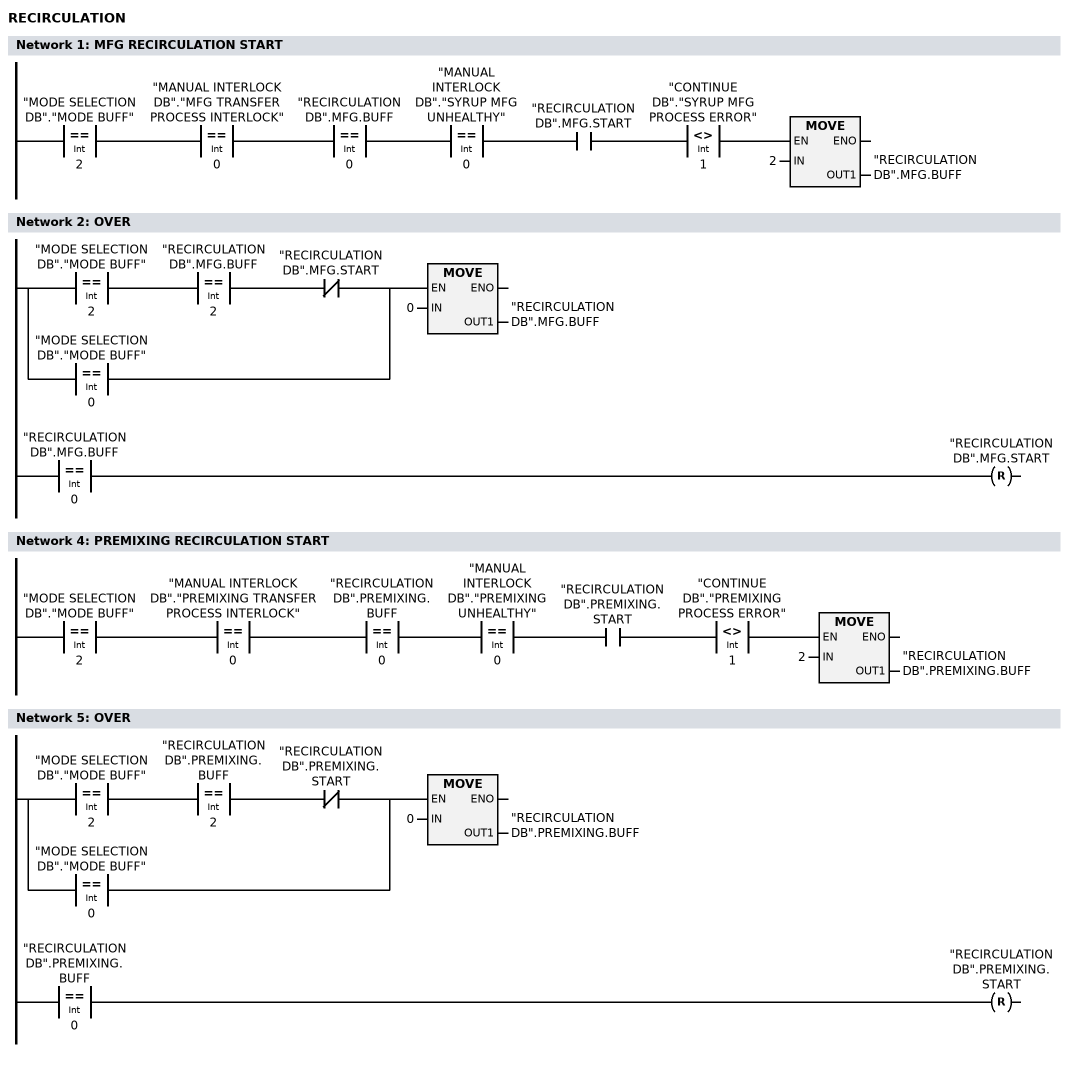
   RUNG wire#powerrail
      { S7_Templates := "SrcType := Int" } EQ_Contact(in1 := "MODE SELECTION DB"."MODE BUFF", in2 := 2)
      { S7_Templates := "SrcType := Int" } EQ_Contact(in1 := "MANUAL INTERLOCK DB"."MFG TRANSFER PROCESS INTERLOCK", in2 := 0)
      { S7_Templates := "SrcType := Int" } EQ_Contact(in1 := "RECIRCULATION DB".MFG.BUFF, in2 := 0)
      { S7_Templates := "SrcType := Int" } EQ_Contact(in1 := "MANUAL INTERLOCK DB"."SYRUP MFG UNHEALTHY", in2 := 0)
      Contact( "RECIRCULATION DB".MFG.START )
      { S7_Templates := "SrcType := Int" } NE_Contact(in1 := "CONTINUE DB"."SYRUP MFG PROCESS ERROR", in2 := 1)
      Move(in := 2, out1 => "RECIRCULATION DB".MFG.BUFF)
   END_RUNG
   // the same network as SCL:
   IF ("MODE SELECTION DB"."MODE BUFF" = 2) AND ("MANUAL INTERLOCK DB"."MFG TRANSFER PROCESS INTERLOCK" = 0) AND ("RECIRCULATION DB".MFG.BUFF = 0) AND ("MANUAL INTERLOCK DB"."SYRUP MFG UNHEALTHY" = 0) AND "RECIRCULATION DB".MFG.START AND ("CONTINUE DB"."SYRUP MFG PROCESS ERROR" <> 1) THEN
       "RECIRCULATION DB".MFG.BUFF := 2;
   END_IF;
END_REGION

REGION Network 2: OVER
   RUNG wire#powerrail
      { S7_Templates := "SrcType := Int" } EQ_Contact(in1 := "MODE SELECTION DB"."MODE BUFF", in2 := 2)
      { S7_Templates := "SrcType := Int" } EQ_Contact(in1 := "RECIRCULATION DB".MFG.BUFF, in2 := 2)
      I_Contact( "RECIRCULATION DB".MFG.START )
      wire#w1
      Move(in := 0, out1 => "RECIRCULATION DB".MFG.BUFF)
   END_RUNG
   RUNG wire#powerrail
      { S7_Templates := "SrcType := Int" } EQ_Contact(in1 := "MODE SELECTION DB"."MODE BUFF", in2 := 0)
   END_RUNG wire#w1
   RUNG wire#powerrail
      { S7_Templates := "SrcType := Int" } EQ_Contact(in1 := "RECIRCULATION DB".MFG.BUFF, in2 := 0)
      R_Coil( "RECIRCULATION DB".MFG.START )
   END_RUNG
   // the same network as SCL:
   IF (("MODE SELECTION DB"."MODE BUFF" = 2) AND ("RECIRCULATION DB".MFG.BUFF = 2) AND NOT "RECIRCULATION DB".MFG.START) OR ("MODE SELECTION DB"."MODE BUFF" = 0) THEN
       "RECIRCULATION DB".MFG.BUFF := 0;
   END_IF;
   IF "RECIRCULATION DB".MFG.BUFF = 0 THEN "RECIRCULATION DB".MFG.START := FALSE; END_IF;
END_REGION

REGION Network 4: PREMIXING RECIRCULATION START
   RUNG wire#powerrail
      { S7_Templates := "SrcType := Int" } EQ_Contact(in1 := "MODE SELECTION DB"."MODE BUFF", in2 := 2)
      { S7_Templates := "SrcType := Int" } EQ_Contact(in1 := "MANUAL INTERLOCK DB"."PREMIXING TRANSFER PROCESS INTERLOCK", in2 := 0)
      { S7_Templates := "SrcType := Int" } EQ_Contact(in1 := "RECIRCULATION DB".PREMIXING.BUFF, in2 := 0)
      { S7_Templates := "SrcType := Int" } EQ_Contact(in1 := "MANUAL INTERLOCK DB"."PREMIXING UNHEALTHY", in2 := 0)
      Contact( "RECIRCULATION DB".PREMIXING.START )
      { S7_Templates := "SrcType := Int" } NE_Contact(in1 := "CONTINUE DB"."PREMIXING PROCESS ERROR", in2 := 1)
      Move(in := 2, out1 => "RECIRCULATION DB".PREMIXING.BUFF)
   END_RUNG
   // the same network as SCL:
   IF ("MODE SELECTION DB"."MODE BUFF" = 2) AND ("MANUAL INTERLOCK DB"."PREMIXING TRANSFER PROCESS INTERLOCK" = 0) AND ("RECIRCULATION DB".PREMIXING.BUFF = 0) AND ("MANUAL INTERLOCK DB"."PREMIXING UNHEALTHY" = 0) AND "RECIRCULATION DB".PREMIXING.START AND ("CONTINUE DB"."PREMIXING PROCESS ERROR" <> 1) THEN
       "RECIRCULATION DB".PREMIXING.BUFF := 2;
   END_IF;
END_REGION

REGION Network 5: OVER
   RUNG wire#powerrail
      { S7_Templates := "SrcType := Int" } EQ_Contact(in1 := "MODE SELECTION DB"."MODE BUFF", in2 := 2)
      { S7_Templates := "SrcType := Int" } EQ_Contact(in1 := "RECIRCULATION DB".PREMIXING.BUFF, in2 := 2)
      I_Contact( "RECIRCULATION DB".PREMIXING.START )
      wire#w1
      Move(in := 0, out1 => "RECIRCULATION DB".PREMIXING.BUFF)
   END_RUNG
   RUNG wire#powerrail
      { S7_Templates := "SrcType := Int" } EQ_Contact(in1 := "MODE SELECTION DB"."MODE BUFF", in2 := 0)
   END_RUNG wire#w1
   RUNG wire#powerrail
      { S7_Templates := "SrcType := Int" } EQ_Contact(in1 := "RECIRCULATION DB".PREMIXING.BUFF, in2 := 0)
      R_Coil( "RECIRCULATION DB".PREMIXING.START )
   END_RUNG
   // the same network as SCL:
   IF (("MODE SELECTION DB"."MODE BUFF" = 2) AND ("RECIRCULATION DB".PREMIXING.BUFF = 2) AND NOT "RECIRCULATION DB".PREMIXING.START) OR ("MODE SELECTION DB"."MODE BUFF" = 0) THEN
       "RECIRCULATION DB".PREMIXING.BUFF := 0;
   END_IF;
   IF "RECIRCULATION DB".PREMIXING.BUFF = 0 THEN "RECIRCULATION DB".PREMIXING.START := FALSE; END_IF;
END_REGION
END_FUNCTION

FUNCTION "TEMP CUTOFF LOGIC" : Void   // FC11, LAD
{ S7_Optimized_Access := 'TRUE' }
// stored: SetENOAutomatically false
   VAR_TEMP   // added for the SCL form of the ladder/FBD networks
      _w1 : Bool;
      _w2 : Bool;
   END_VAR
BEGIN

REGION Network 1: MFG_TEMP. VALUE ///////////////////////////////////////////////////////////////
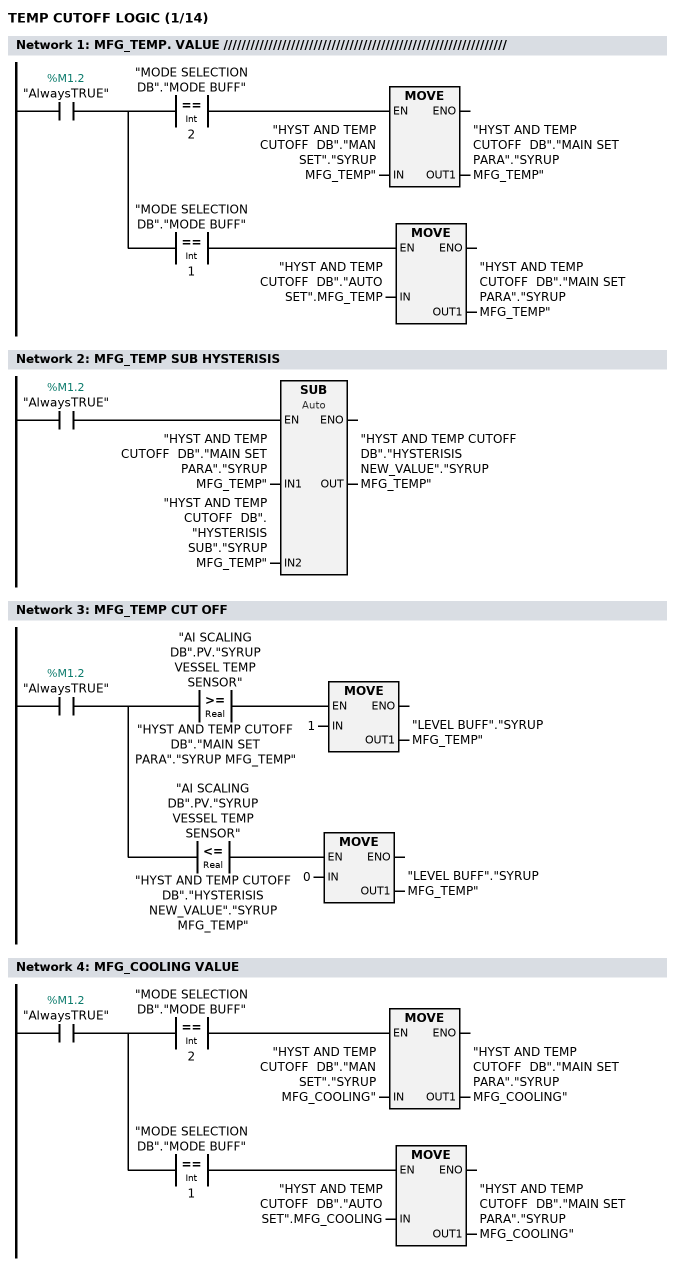
   RUNG wire#powerrail
      Contact( "AlwaysTRUE" )
      wire#w1
      { S7_Templates := "SrcType := Int" } EQ_Contact(in1 := "MODE SELECTION DB"."MODE BUFF", in2 := 2)
      Move(in := "HYST AND TEMP CUTOFF  DB"."MAN SET"."SYRUP MFG_TEMP", out1 => "HYST AND TEMP CUTOFF  DB"."MAIN SET PARA"."SYRUP MFG_TEMP")
   END_RUNG
   RUNG wire#w1
      { S7_Templates := "SrcType := Int" } EQ_Contact(in1 := "MODE SELECTION DB"."MODE BUFF", in2 := 1)
      Move(in := "HYST AND TEMP CUTOFF  DB"."AUTO SET".MFG_TEMP, out1 => "HYST AND TEMP CUTOFF  DB"."MAIN SET PARA"."SYRUP MFG_TEMP")
   END_RUNG
   // the same network as SCL:
   IF "AlwaysTRUE" AND ("MODE SELECTION DB"."MODE BUFF" = 2) THEN
       "HYST AND TEMP CUTOFF  DB"."MAIN SET PARA"."SYRUP MFG_TEMP" := "HYST AND TEMP CUTOFF  DB"."MAN SET"."SYRUP MFG_TEMP";
   END_IF;
   IF "AlwaysTRUE" AND ("MODE SELECTION DB"."MODE BUFF" = 1) THEN
       "HYST AND TEMP CUTOFF  DB"."MAIN SET PARA"."SYRUP MFG_TEMP" := "HYST AND TEMP CUTOFF  DB"."AUTO SET".MFG_TEMP;
   END_IF;
END_REGION

REGION Network 2: MFG_TEMP SUB HYSTERISIS
   RUNG wire#powerrail
      Contact( "AlwaysTRUE" )
      Sub(in1 := "HYST AND TEMP CUTOFF  DB"."MAIN SET PARA"."SYRUP MFG_TEMP", in2 := "HYST AND TEMP CUTOFF  DB"."HYSTERISIS SUB"."SYRUP MFG_TEMP", out => "HYST AND TEMP CUTOFF  DB"."HYSTERISIS NEW_VALUE"."SYRUP MFG_TEMP")
   END_RUNG
   // the same network as SCL:
   IF "AlwaysTRUE" THEN
       "HYST AND TEMP CUTOFF  DB"."HYSTERISIS NEW_VALUE"."SYRUP MFG_TEMP" := "HYST AND TEMP CUTOFF  DB"."MAIN SET PARA"."SYRUP MFG_TEMP" - "HYST AND TEMP CUTOFF  DB"."HYSTERISIS SUB"."SYRUP MFG_TEMP";
   END_IF;
END_REGION

REGION Network 3: MFG_TEMP CUT OFF
   RUNG wire#powerrail
      Contact( "AlwaysTRUE" )
      wire#w1
      { S7_Templates := "SrcType := Real" } GE_Contact(in1 := "AI SCALING DB".PV."SYRUP VESSEL TEMP SENSOR", in2 := "HYST AND TEMP CUTOFF  DB"."MAIN SET PARA"."SYRUP MFG_TEMP")
      Move(in := 1, out1 => "LEVEL BUFF"."SYRUP MFG_TEMP")
   END_RUNG
   RUNG wire#w1
      { S7_Templates := "SrcType := Real" } LE_Contact(in1 := "AI SCALING DB".PV."SYRUP VESSEL TEMP SENSOR", in2 := "HYST AND TEMP CUTOFF  DB"."HYSTERISIS NEW_VALUE"."SYRUP MFG_TEMP")
      Move(in := 0, out1 => "LEVEL BUFF"."SYRUP MFG_TEMP")
   END_RUNG
   // the same network as SCL:
   IF "AlwaysTRUE" AND ("AI SCALING DB".PV."SYRUP VESSEL TEMP SENSOR" >= "HYST AND TEMP CUTOFF  DB"."MAIN SET PARA"."SYRUP MFG_TEMP") THEN
       "LEVEL BUFF"."SYRUP MFG_TEMP" := 1;
   END_IF;
   IF "AlwaysTRUE" AND ("AI SCALING DB".PV."SYRUP VESSEL TEMP SENSOR" <= "HYST AND TEMP CUTOFF  DB"."HYSTERISIS NEW_VALUE"."SYRUP MFG_TEMP") THEN
       "LEVEL BUFF"."SYRUP MFG_TEMP" := 0;
   END_IF;
END_REGION

REGION Network 4: MFG_COOLING VALUE
   RUNG wire#powerrail
      Contact( "AlwaysTRUE" )
      wire#w1
      { S7_Templates := "SrcType := Int" } EQ_Contact(in1 := "MODE SELECTION DB"."MODE BUFF", in2 := 2)
      Move(in := "HYST AND TEMP CUTOFF  DB"."MAN SET"."SYRUP MFG_COOLING", out1 => "HYST AND TEMP CUTOFF  DB"."MAIN SET PARA"."SYRUP MFG_COOLING")
   END_RUNG
   RUNG wire#w1
      { S7_Templates := "SrcType := Int" } EQ_Contact(in1 := "MODE SELECTION DB"."MODE BUFF", in2 := 1)
      Move(in := "HYST AND TEMP CUTOFF  DB"."AUTO SET".MFG_COOLING, out1 => "HYST AND TEMP CUTOFF  DB"."MAIN SET PARA"."SYRUP MFG_COOLING")
   END_RUNG
   // the same network as SCL:
   IF "AlwaysTRUE" AND ("MODE SELECTION DB"."MODE BUFF" = 2) THEN
       "HYST AND TEMP CUTOFF  DB"."MAIN SET PARA"."SYRUP MFG_COOLING" := "HYST AND TEMP CUTOFF  DB"."MAN SET"."SYRUP MFG_COOLING";
   END_IF;
   IF "AlwaysTRUE" AND ("MODE SELECTION DB"."MODE BUFF" = 1) THEN
       "HYST AND TEMP CUTOFF  DB"."MAIN SET PARA"."SYRUP MFG_COOLING" := "HYST AND TEMP CUTOFF  DB"."AUTO SET".MFG_COOLING;
   END_IF;
END_REGION

REGION Network 5: MFG_COOLING SUB HYSTERISIS
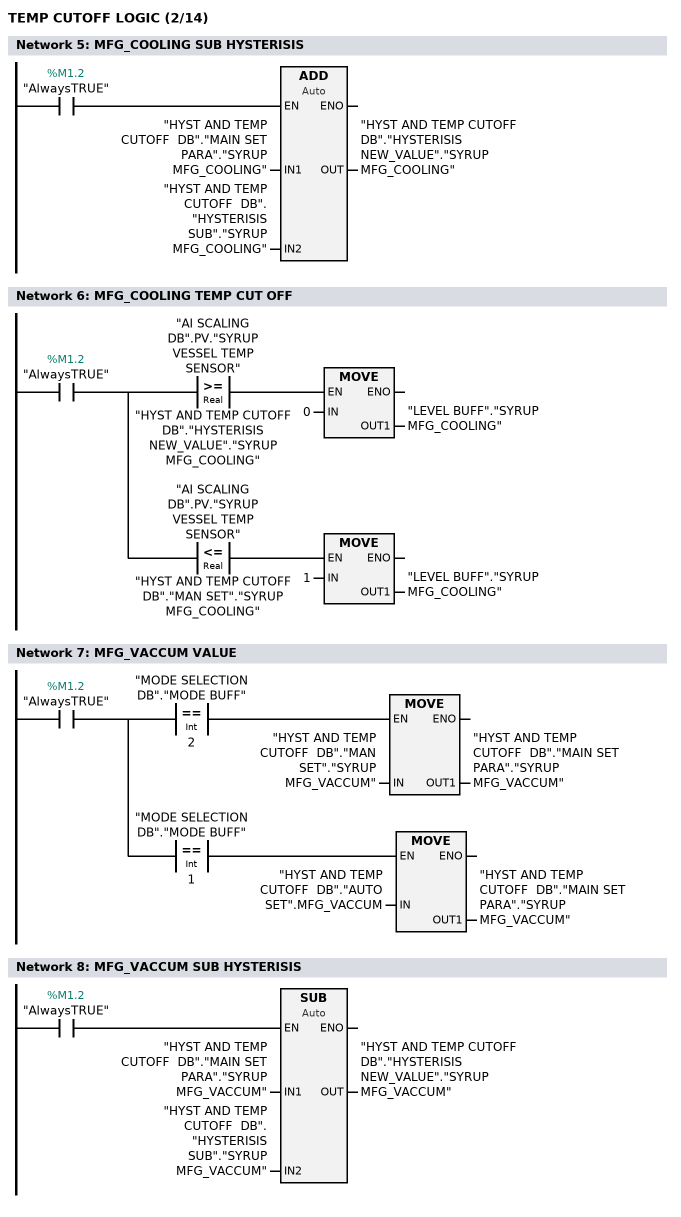
   RUNG wire#powerrail
      Contact( "AlwaysTRUE" )
      Add(in1 := "HYST AND TEMP CUTOFF  DB"."MAIN SET PARA"."SYRUP MFG_COOLING", in2 := "HYST AND TEMP CUTOFF  DB"."HYSTERISIS SUB"."SYRUP MFG_COOLING", out => "HYST AND TEMP CUTOFF  DB"."HYSTERISIS NEW_VALUE"."SYRUP MFG_COOLING")
   END_RUNG
   // the same network as SCL:
   IF "AlwaysTRUE" THEN
       "HYST AND TEMP CUTOFF  DB"."HYSTERISIS NEW_VALUE"."SYRUP MFG_COOLING" := "HYST AND TEMP CUTOFF  DB"."MAIN SET PARA"."SYRUP MFG_COOLING" + "HYST AND TEMP CUTOFF  DB"."HYSTERISIS SUB"."SYRUP MFG_COOLING";
   END_IF;
END_REGION

REGION Network 6: MFG_COOLING TEMP CUT OFF
   RUNG wire#powerrail
      Contact( "AlwaysTRUE" )
      wire#w1
      { S7_Templates := "SrcType := Real" } GE_Contact(in1 := "AI SCALING DB".PV."SYRUP VESSEL TEMP SENSOR", in2 := "HYST AND TEMP CUTOFF  DB"."HYSTERISIS NEW_VALUE"."SYRUP MFG_COOLING")
      Move(in := 0, out1 => "LEVEL BUFF"."SYRUP MFG_COOLING")
   END_RUNG
   RUNG wire#w1
      { S7_Templates := "SrcType := Real" } LE_Contact(in1 := "AI SCALING DB".PV."SYRUP VESSEL TEMP SENSOR", in2 := "HYST AND TEMP CUTOFF  DB"."MAN SET"."SYRUP MFG_COOLING")
      Move(in := 1, out1 => "LEVEL BUFF"."SYRUP MFG_COOLING")
   END_RUNG
   // the same network as SCL:
   IF "AlwaysTRUE" AND ("AI SCALING DB".PV."SYRUP VESSEL TEMP SENSOR" >= "HYST AND TEMP CUTOFF  DB"."HYSTERISIS NEW_VALUE"."SYRUP MFG_COOLING") THEN
       "LEVEL BUFF"."SYRUP MFG_COOLING" := 0;
   END_IF;
   IF "AlwaysTRUE" AND ("AI SCALING DB".PV."SYRUP VESSEL TEMP SENSOR" <= "HYST AND TEMP CUTOFF  DB"."MAN SET"."SYRUP MFG_COOLING") THEN
       "LEVEL BUFF"."SYRUP MFG_COOLING" := 1;
   END_IF;
END_REGION

REGION Network 7: MFG_VACCUM VALUE
   RUNG wire#powerrail
      Contact( "AlwaysTRUE" )
      wire#w1
      { S7_Templates := "SrcType := Int" } EQ_Contact(in1 := "MODE SELECTION DB"."MODE BUFF", in2 := 2)
      Move(in := "HYST AND TEMP CUTOFF  DB"."MAN SET"."SYRUP MFG_VACCUM", out1 => "HYST AND TEMP CUTOFF  DB"."MAIN SET PARA"."SYRUP MFG_VACCUM")
   END_RUNG
   RUNG wire#w1
      { S7_Templates := "SrcType := Int" } EQ_Contact(in1 := "MODE SELECTION DB"."MODE BUFF", in2 := 1)
      Move(in := "HYST AND TEMP CUTOFF  DB"."AUTO SET".MFG_VACCUM, out1 => "HYST AND TEMP CUTOFF  DB"."MAIN SET PARA"."SYRUP MFG_VACCUM")
   END_RUNG
   // the same network as SCL:
   IF "AlwaysTRUE" AND ("MODE SELECTION DB"."MODE BUFF" = 2) THEN
       "HYST AND TEMP CUTOFF  DB"."MAIN SET PARA"."SYRUP MFG_VACCUM" := "HYST AND TEMP CUTOFF  DB"."MAN SET"."SYRUP MFG_VACCUM";
   END_IF;
   IF "AlwaysTRUE" AND ("MODE SELECTION DB"."MODE BUFF" = 1) THEN
       "HYST AND TEMP CUTOFF  DB"."MAIN SET PARA"."SYRUP MFG_VACCUM" := "HYST AND TEMP CUTOFF  DB"."AUTO SET".MFG_VACCUM;
   END_IF;
END_REGION

REGION Network 8: MFG_VACCUM SUB HYSTERISIS
   RUNG wire#powerrail
      Contact( "AlwaysTRUE" )
      Sub(in1 := "HYST AND TEMP CUTOFF  DB"."MAIN SET PARA"."SYRUP MFG_VACCUM", in2 := "HYST AND TEMP CUTOFF  DB"."HYSTERISIS SUB"."SYRUP MFG_VACCUM", out => "HYST AND TEMP CUTOFF  DB"."HYSTERISIS NEW_VALUE"."SYRUP MFG_VACCUM")
   END_RUNG
   // the same network as SCL:
   IF "AlwaysTRUE" THEN
       "HYST AND TEMP CUTOFF  DB"."HYSTERISIS NEW_VALUE"."SYRUP MFG_VACCUM" := "HYST AND TEMP CUTOFF  DB"."MAIN SET PARA"."SYRUP MFG_VACCUM" - "HYST AND TEMP CUTOFF  DB"."HYSTERISIS SUB"."SYRUP MFG_VACCUM";
   END_IF;
END_REGION

REGION Network 9: MFG_VACCUM CUT OFF
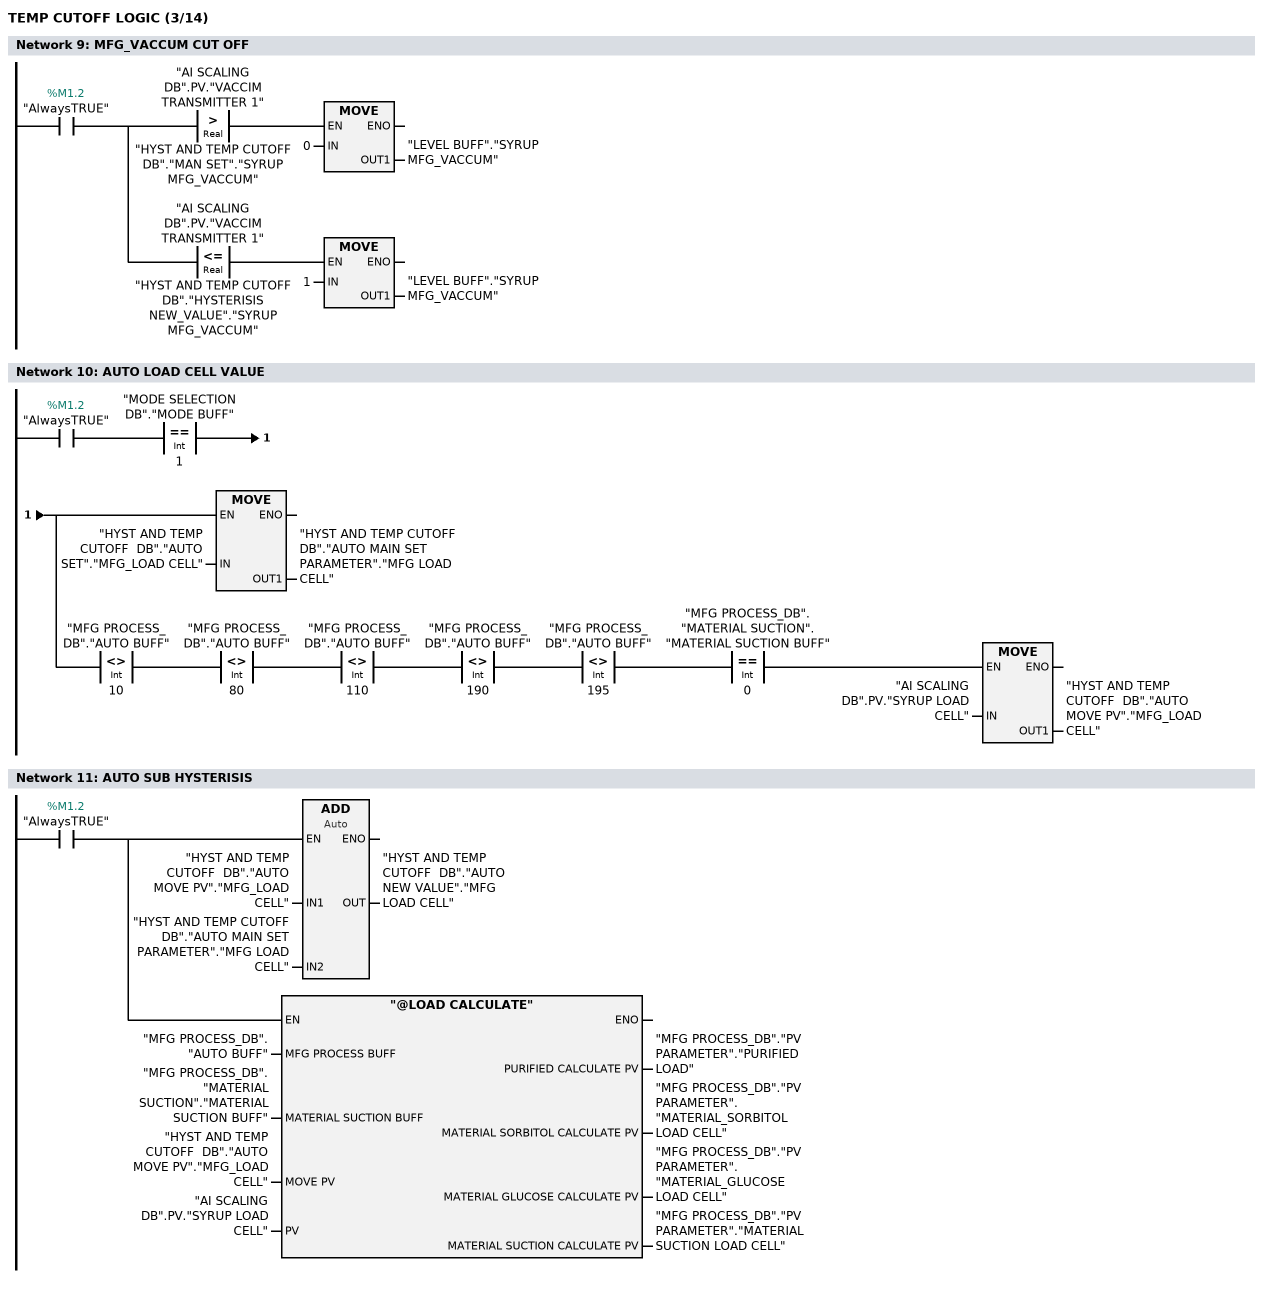
   RUNG wire#powerrail
      Contact( "AlwaysTRUE" )
      wire#w1
      { S7_Templates := "SrcType := Real" } GT_Contact(in1 := "AI SCALING DB".PV."VACCIM TRANSMITTER 1", in2 := "HYST AND TEMP CUTOFF  DB"."MAN SET"."SYRUP MFG_VACCUM")
      Move(in := 0, out1 => "LEVEL BUFF"."SYRUP MFG_VACCUM")
   END_RUNG
   RUNG wire#w1
      { S7_Templates := "SrcType := Real" } LE_Contact(in1 := "AI SCALING DB".PV."VACCIM TRANSMITTER 1", in2 := "HYST AND TEMP CUTOFF  DB"."HYSTERISIS NEW_VALUE"."SYRUP MFG_VACCUM")
      Move(in := 1, out1 => "LEVEL BUFF"."SYRUP MFG_VACCUM")
   END_RUNG
   // the same network as SCL:
   IF "AlwaysTRUE" AND ("AI SCALING DB".PV."VACCIM TRANSMITTER 1" > "HYST AND TEMP CUTOFF  DB"."MAN SET"."SYRUP MFG_VACCUM") THEN
       "LEVEL BUFF"."SYRUP MFG_VACCUM" := 0;
   END_IF;
   IF "AlwaysTRUE" AND ("AI SCALING DB".PV."VACCIM TRANSMITTER 1" <= "HYST AND TEMP CUTOFF  DB"."HYSTERISIS NEW_VALUE"."SYRUP MFG_VACCUM") THEN
       "LEVEL BUFF"."SYRUP MFG_VACCUM" := 1;
   END_IF;
END_REGION

REGION Network 10: AUTO LOAD CELL VALUE
   RUNG wire#powerrail
      Contact( "AlwaysTRUE" )
      { S7_Templates := "SrcType := Int" } EQ_Contact(in1 := "MODE SELECTION DB"."MODE BUFF", in2 := 1)
      wire#w1
      Move(in := "HYST AND TEMP CUTOFF  DB"."AUTO SET"."MFG_LOAD CELL", out1 => "HYST AND TEMP CUTOFF  DB"."AUTO MAIN SET PARAMETER"."MFG LOAD CELL")
   END_RUNG
   RUNG wire#w1
      { S7_Templates := "SrcType := Int" } NE_Contact(in1 := "MFG PROCESS_DB"."AUTO BUFF", in2 := 10)
      { S7_Templates := "SrcType := Int" } NE_Contact(in1 := "MFG PROCESS_DB"."AUTO BUFF", in2 := 80)
      { S7_Templates := "SrcType := Int" } NE_Contact(in1 := "MFG PROCESS_DB"."AUTO BUFF", in2 := 110)
      { S7_Templates := "SrcType := Int" } NE_Contact(in1 := "MFG PROCESS_DB"."AUTO BUFF", in2 := 190)
      { S7_Templates := "SrcType := Int" } NE_Contact(in1 := "MFG PROCESS_DB"."AUTO BUFF", in2 := 195)
      { S7_Templates := "SrcType := Int" } EQ_Contact(in1 := "MFG PROCESS_DB"."MATERIAL SUCTION"."MATERIAL SUCTION BUFF", in2 := 0)
      Move(in := "AI SCALING DB".PV."SYRUP LOAD CELL", out1 => "HYST AND TEMP CUTOFF  DB"."AUTO MOVE PV"."MFG_LOAD CELL")
   END_RUNG
   // the same network as SCL:
   #_w1 := "AlwaysTRUE" AND ("MODE SELECTION DB"."MODE BUFF" = 1);
   IF #_w1 THEN
       "HYST AND TEMP CUTOFF  DB"."AUTO MAIN SET PARAMETER"."MFG LOAD CELL" := "HYST AND TEMP CUTOFF  DB"."AUTO SET"."MFG_LOAD CELL";
   END_IF;
   IF #_w1 AND ("MFG PROCESS_DB"."AUTO BUFF" <> 10) AND ("MFG PROCESS_DB"."AUTO BUFF" <> 80) AND ("MFG PROCESS_DB"."AUTO BUFF" <> 110) AND ("MFG PROCESS_DB"."AUTO BUFF" <> 190) AND ("MFG PROCESS_DB"."AUTO BUFF" <> 195) AND ("MFG PROCESS_DB"."MATERIAL SUCTION"."MATERIAL SUCTION BUFF" = 0) THEN
       "HYST AND TEMP CUTOFF  DB"."AUTO MOVE PV"."MFG_LOAD CELL" := "AI SCALING DB".PV."SYRUP LOAD CELL";
   END_IF;
END_REGION

REGION Network 11: AUTO SUB HYSTERISIS
   RUNG wire#powerrail
      Contact( "AlwaysTRUE" )
      wire#w1
      Add(in1 := "HYST AND TEMP CUTOFF  DB"."AUTO MOVE PV"."MFG_LOAD CELL", in2 := "HYST AND TEMP CUTOFF  DB"."AUTO MAIN SET PARAMETER"."MFG LOAD CELL", out => "HYST AND TEMP CUTOFF  DB"."AUTO NEW VALUE"."MFG LOAD CELL")
   END_RUNG
   RUNG wire#w1
      "@LOAD CALCULATE"("MFG PROCESS BUFF" := "MFG PROCESS_DB"."AUTO BUFF", "MATERIAL SUCTION BUFF" := "MFG PROCESS_DB"."MATERIAL SUCTION"."MATERIAL SUCTION BUFF", "MOVE PV" := "HYST AND TEMP CUTOFF  DB"."AUTO MOVE PV"."MFG_LOAD CELL", PV := "AI SCALING DB".PV."SYRUP LOAD CELL", "PURIFIED CALCULATE PV" => "MFG PROCESS_DB"."PV PARAMETER"."PURIFIED LOAD", "MATERIAL SORBITOL CALCULATE PV" => "MFG PROCESS_DB"."PV PARAMETER"."MATERIAL_SORBITOL LOAD CELL", "MATERIAL GLUCOSE CALCULATE PV" => "MFG PROCESS_DB"."PV PARAMETER"."MATERIAL_GLUCOSE LOAD CELL", "MATERIAL SUCTION CALCULATE PV" => "MFG PROCESS_DB"."PV PARAMETER"."MATERIAL SUCTION LOAD CELL")
   END_RUNG
   // the same network as SCL:
   IF "AlwaysTRUE" THEN
       "HYST AND TEMP CUTOFF  DB"."AUTO NEW VALUE"."MFG LOAD CELL" := "HYST AND TEMP CUTOFF  DB"."AUTO MOVE PV"."MFG_LOAD CELL" + "HYST AND TEMP CUTOFF  DB"."AUTO MAIN SET PARAMETER"."MFG LOAD CELL";
       "@LOAD CALCULATE"("MFG PROCESS BUFF" := "MFG PROCESS_DB"."AUTO BUFF",
                         "MATERIAL SUCTION BUFF" := "MFG PROCESS_DB"."MATERIAL SUCTION"."MATERIAL SUCTION BUFF",
                         "MOVE PV" := "HYST AND TEMP CUTOFF  DB"."AUTO MOVE PV"."MFG_LOAD CELL",
                         PV := "AI SCALING DB".PV."SYRUP LOAD CELL",
                         "PURIFIED CALCULATE PV" => "MFG PROCESS_DB"."PV PARAMETER"."PURIFIED LOAD",
                         "MATERIAL SORBITOL CALCULATE PV" => "MFG PROCESS_DB"."PV PARAMETER"."MATERIAL_SORBITOL LOAD CELL",
                         "MATERIAL GLUCOSE CALCULATE PV" => "MFG PROCESS_DB"."PV PARAMETER"."MATERIAL_GLUCOSE LOAD CELL",
                         "MATERIAL SUCTION CALCULATE PV" => "MFG PROCESS_DB"."PV PARAMETER"."MATERIAL SUCTION LOAD CELL");
   END_IF;
END_REGION

REGION Network 12: AUTO LOAD CELL CUT OFF
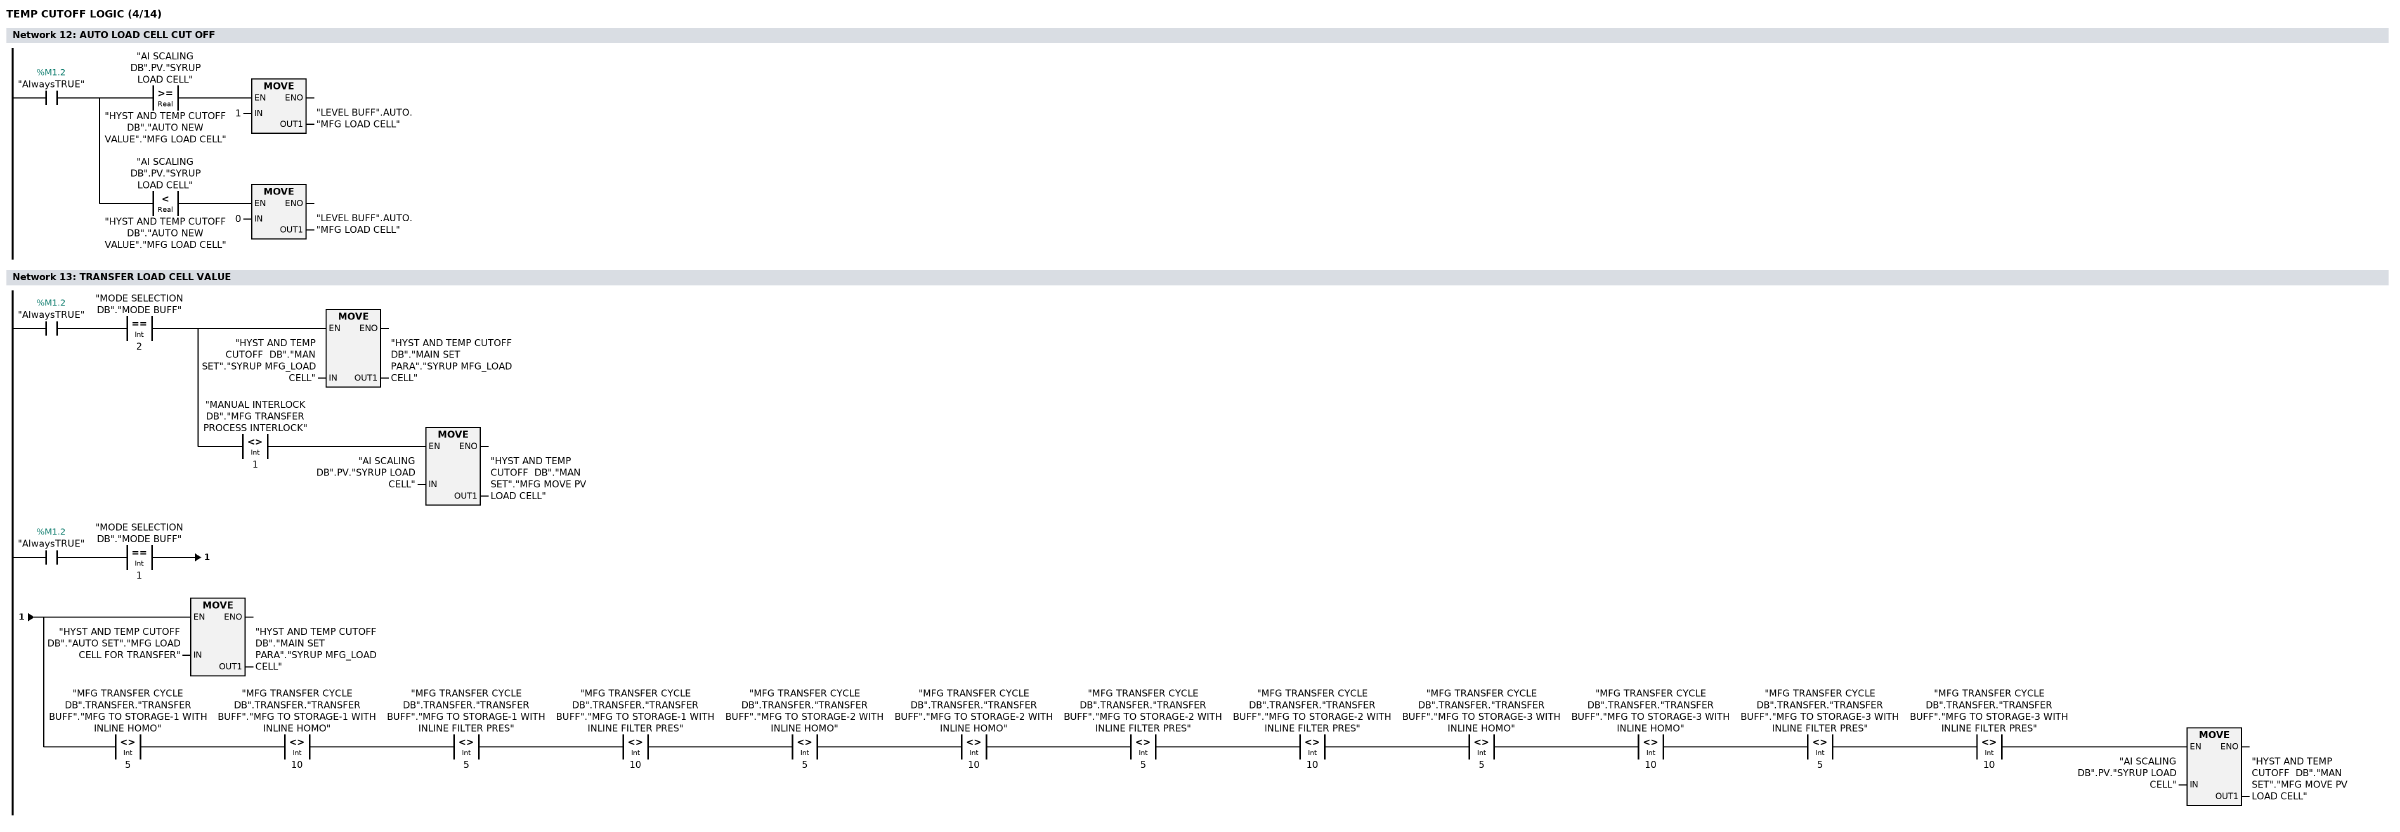
   RUNG wire#powerrail
      Contact( "AlwaysTRUE" )
      wire#w1
      { S7_Templates := "SrcType := Real" } GE_Contact(in1 := "AI SCALING DB".PV."SYRUP LOAD CELL", in2 := "HYST AND TEMP CUTOFF  DB"."AUTO NEW VALUE"."MFG LOAD CELL")
      Move(in := 1, out1 => "LEVEL BUFF".AUTO."MFG LOAD CELL")
   END_RUNG
   RUNG wire#w1
      { S7_Templates := "SrcType := Real" } LT_Contact(in1 := "AI SCALING DB".PV."SYRUP LOAD CELL", in2 := "HYST AND TEMP CUTOFF  DB"."AUTO NEW VALUE"."MFG LOAD CELL")
      Move(in := 0, out1 => "LEVEL BUFF".AUTO."MFG LOAD CELL")
   END_RUNG
   // the same network as SCL:
   IF "AlwaysTRUE" AND ("AI SCALING DB".PV."SYRUP LOAD CELL" >= "HYST AND TEMP CUTOFF  DB"."AUTO NEW VALUE"."MFG LOAD CELL") THEN
       "LEVEL BUFF".AUTO."MFG LOAD CELL" := 1;
   END_IF;
   IF "AlwaysTRUE" AND ("AI SCALING DB".PV."SYRUP LOAD CELL" < "HYST AND TEMP CUTOFF  DB"."AUTO NEW VALUE"."MFG LOAD CELL") THEN
       "LEVEL BUFF".AUTO."MFG LOAD CELL" := 0;
   END_IF;
END_REGION

REGION Network 13: TRANSFER LOAD CELL VALUE
   RUNG wire#powerrail
      Contact( "AlwaysTRUE" )
      { S7_Templates := "SrcType := Int" } EQ_Contact(in1 := "MODE SELECTION DB"."MODE BUFF", in2 := 2)
      wire#w1
      Move(in := "HYST AND TEMP CUTOFF  DB"."MAN SET"."SYRUP MFG_LOAD CELL", out1 => "HYST AND TEMP CUTOFF  DB"."MAIN SET PARA"."SYRUP MFG_LOAD CELL")
   END_RUNG
   RUNG wire#w1
      { S7_Templates := "SrcType := Int" } NE_Contact(in1 := "MANUAL INTERLOCK DB"."MFG TRANSFER PROCESS INTERLOCK", in2 := 1)
      Move(in := "AI SCALING DB".PV."SYRUP LOAD CELL", out1 => "HYST AND TEMP CUTOFF  DB"."MAN SET"."MFG MOVE PV LOAD CELL")
   END_RUNG
   RUNG wire#powerrail
      Contact( "AlwaysTRUE" )
      { S7_Templates := "SrcType := Int" } EQ_Contact(in1 := "MODE SELECTION DB"."MODE BUFF", in2 := 1)
      wire#w2
      Move(in := "HYST AND TEMP CUTOFF  DB"."AUTO SET"."MFG LOAD CELL FOR TRANSFER", out1 => "HYST AND TEMP CUTOFF  DB"."MAIN SET PARA"."SYRUP MFG_LOAD CELL")
   END_RUNG
   RUNG wire#w2
      { S7_Templates := "SrcType := Int" } NE_Contact(in1 := "MFG TRANSFER CYCLE DB".TRANSFER."TRANSFER BUFF"."MFG TO STORAGE-1 WITH INLINE HOMO", in2 := 5)
      { S7_Templates := "SrcType := Int" } NE_Contact(in1 := "MFG TRANSFER CYCLE DB".TRANSFER."TRANSFER BUFF"."MFG TO STORAGE-1 WITH INLINE HOMO", in2 := 10)
      { S7_Templates := "SrcType := Int" } NE_Contact(in1 := "MFG TRANSFER CYCLE DB".TRANSFER."TRANSFER BUFF"."MFG TO STORAGE-1 WITH INLINE FILTER PRES", in2 := 5)
      { S7_Templates := "SrcType := Int" } NE_Contact(in1 := "MFG TRANSFER CYCLE DB".TRANSFER."TRANSFER BUFF"."MFG TO STORAGE-1 WITH INLINE FILTER PRES", in2 := 10)
      { S7_Templates := "SrcType := Int" } NE_Contact(in1 := "MFG TRANSFER CYCLE DB".TRANSFER."TRANSFER BUFF"."MFG TO STORAGE-2 WITH INLINE HOMO", in2 := 5)
      { S7_Templates := "SrcType := Int" } NE_Contact(in1 := "MFG TRANSFER CYCLE DB".TRANSFER."TRANSFER BUFF"."MFG TO STORAGE-2 WITH INLINE HOMO", in2 := 10)
      { S7_Templates := "SrcType := Int" } NE_Contact(in1 := "MFG TRANSFER CYCLE DB".TRANSFER."TRANSFER BUFF"."MFG TO STORAGE-2 WITH INLINE FILTER PRES", in2 := 5)
      { S7_Templates := "SrcType := Int" } NE_Contact(in1 := "MFG TRANSFER CYCLE DB".TRANSFER."TRANSFER BUFF"."MFG TO STORAGE-2 WITH INLINE FILTER PRES", in2 := 10)
      { S7_Templates := "SrcType := Int" } NE_Contact(in1 := "MFG TRANSFER CYCLE DB".TRANSFER."TRANSFER BUFF"."MFG TO STORAGE-3 WITH INLINE HOMO", in2 := 5)
      { S7_Templates := "SrcType := Int" } NE_Contact(in1 := "MFG TRANSFER CYCLE DB".TRANSFER."TRANSFER BUFF"."MFG TO STORAGE-3 WITH INLINE HOMO", in2 := 10)
      { S7_Templates := "SrcType := Int" } NE_Contact(in1 := "MFG TRANSFER CYCLE DB".TRANSFER."TRANSFER BUFF"."MFG TO STORAGE-3 WITH INLINE FILTER PRES", in2 := 5)
      { S7_Templates := "SrcType := Int" } NE_Contact(in1 := "MFG TRANSFER CYCLE DB".TRANSFER."TRANSFER BUFF"."MFG TO STORAGE-3 WITH INLINE FILTER PRES", in2 := 10)
      Move(in := "AI SCALING DB".PV."SYRUP LOAD CELL", out1 => "HYST AND TEMP CUTOFF  DB"."MAN SET"."MFG MOVE PV LOAD CELL")
   END_RUNG
   // the same network as SCL:
   #_w1 := "AlwaysTRUE" AND ("MODE SELECTION DB"."MODE BUFF" = 2);
   IF #_w1 THEN
       "HYST AND TEMP CUTOFF  DB"."MAIN SET PARA"."SYRUP MFG_LOAD CELL" := "HYST AND TEMP CUTOFF  DB"."MAN SET"."SYRUP MFG_LOAD CELL";
   END_IF;
   IF #_w1 AND ("MANUAL INTERLOCK DB"."MFG TRANSFER PROCESS INTERLOCK" <> 1) THEN
       "HYST AND TEMP CUTOFF  DB"."MAN SET"."MFG MOVE PV LOAD CELL" := "AI SCALING DB".PV."SYRUP LOAD CELL";
   END_IF;
   #_w2 := "AlwaysTRUE" AND ("MODE SELECTION DB"."MODE BUFF" = 1);
   IF #_w2 THEN
       "HYST AND TEMP CUTOFF  DB"."MAIN SET PARA"."SYRUP MFG_LOAD CELL" := "HYST AND TEMP CUTOFF  DB"."AUTO SET"."MFG LOAD CELL FOR TRANSFER";
   END_IF;
   IF #_w2 AND ("MFG TRANSFER CYCLE DB".TRANSFER."TRANSFER BUFF"."MFG TO STORAGE-1 WITH INLINE HOMO" <> 5) AND ("MFG TRANSFER CYCLE DB".TRANSFER."TRANSFER BUFF"."MFG TO STORAGE-1 WITH INLINE HOMO" <> 10) AND ("MFG TRANSFER CYCLE DB".TRANSFER."TRANSFER BUFF"."MFG TO STORAGE-1 WITH INLINE FILTER PRES" <> 5) AND ("MFG TRANSFER CYCLE DB".TRANSFER."TRANSFER BUFF"."MFG TO STORAGE-1 WITH INLINE FILTER PRES" <> 10) AND ("MFG TRANSFER CYCLE DB".TRANSFER."TRANSFER BUFF"."MFG TO STORAGE-2 WITH INLINE HOMO" <> 5) AND ("MFG TRANSFER CYCLE DB".TRANSFER."TRANSFER BUFF"."MFG TO STORAGE-2 WITH INLINE HOMO" <> 10) AND ("MFG TRANSFER CYCLE DB".TRANSFER."TRANSFER BUFF"."MFG TO STORAGE-2 WITH INLINE FILTER PRES" <> 5) AND ("MFG TRANSFER CYCLE DB".TRANSFER."TRANSFER BUFF"."MFG TO STORAGE-2 WITH INLINE FILTER PRES" <> 10) AND ("MFG TRANSFER CYCLE DB".TRANSFER."TRANSFER BUFF"."MFG TO STORAGE-3 WITH INLINE HOMO" <> 5) AND ("MFG TRANSFER CYCLE DB".TRANSFER."TRANSFER BUFF"."MFG TO STORAGE-3 WITH INLINE HOMO" <> 10) AND ("MFG TRANSFER CYCLE DB".TRANSFER."TRANSFER BUFF"."MFG TO STORAGE-3 WITH INLINE FILTER PRES" <> 5) AND ("MFG TRANSFER CYCLE DB".TRANSFER."TRANSFER BUFF"."MFG TO STORAGE-3 WITH INLINE FILTER PRES" <> 10) THEN
       "HYST AND TEMP CUTOFF  DB"."MAN SET"."MFG MOVE PV LOAD CELL" := "AI SCALING DB".PV."SYRUP LOAD CELL";
   END_IF;
END_REGION

REGION Network 14: TRANSFER CALCULATE
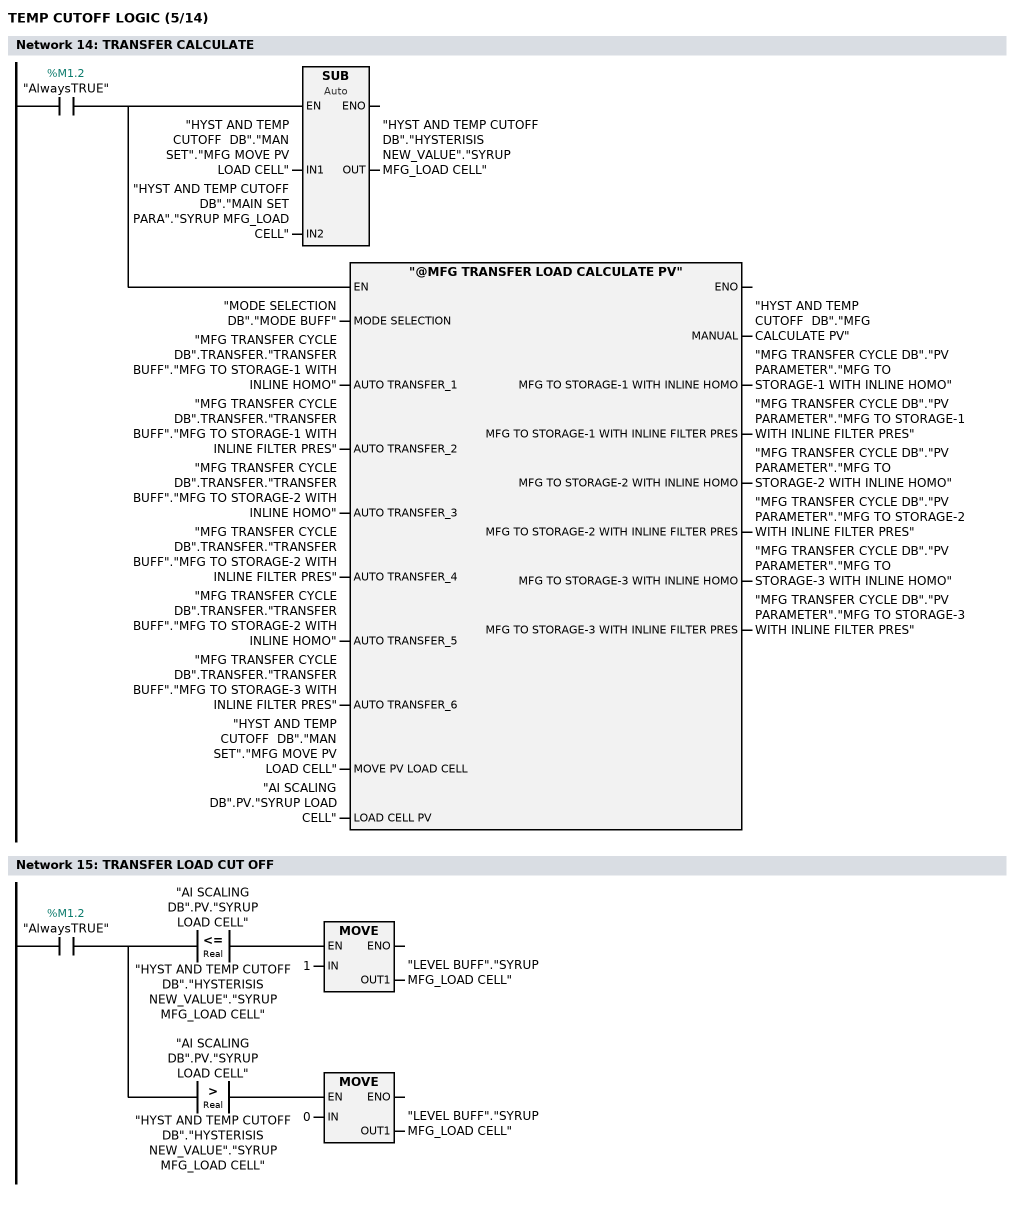
   RUNG wire#powerrail
      Contact( "AlwaysTRUE" )
      wire#w1
      Sub(in1 := "HYST AND TEMP CUTOFF  DB"."MAN SET"."MFG MOVE PV LOAD CELL", in2 := "HYST AND TEMP CUTOFF  DB"."MAIN SET PARA"."SYRUP MFG_LOAD CELL", out => "HYST AND TEMP CUTOFF  DB"."HYSTERISIS NEW_VALUE"."SYRUP MFG_LOAD CELL")
   END_RUNG
   RUNG wire#w1
      "@MFG TRANSFER LOAD CALCULATE PV"("MODE SELECTION" := "MODE SELECTION DB"."MODE BUFF", "AUTO TRANSFER_1" := "MFG TRANSFER CYCLE DB".TRANSFER."TRANSFER BUFF"."MFG TO STORAGE-1 WITH INLINE HOMO", "AUTO TRANSFER_2" := "MFG TRANSFER CYCLE DB".TRANSFER."TRANSFER BUFF"."MFG TO STORAGE-1 WITH INLINE FILTER PRES", "AUTO TRANSFER_3" := "MFG TRANSFER CYCLE DB".TRANSFER."TRANSFER BUFF"."MFG TO STORAGE-2 WITH INLINE HOMO", "AUTO TRANSFER_4" := "MFG TRANSFER CYCLE DB".TRANSFER."TRANSFER BUFF"."MFG TO STORAGE-2 WITH INLINE FILTER PRES", "AUTO TRANSFER_5" := "MFG TRANSFER CYCLE DB".TRANSFER."TRANSFER BUFF"."MFG TO STORAGE-2 WITH INLINE HOMO", "AUTO TRANSFER_6" := "MFG TRANSFER CYCLE DB".TRANSFER."TRANSFER BUFF"."MFG TO STORAGE-3 WITH INLINE FILTER PRES", "MOVE PV LOAD CELL" := "HYST AND TEMP CUTOFF  DB"."MAN SET"."MFG MOVE PV LOAD CELL", "LOAD CELL PV" := "AI SCALING DB".PV."SYRUP LOAD CELL", MANUAL => "HYST AND TEMP CUTOFF  DB"."MFG CALCULATE PV", "MFG TO STORAGE-1 WITH INLINE HOMO" => "MFG TRANSFER CYCLE DB"."PV PARAMETER"."MFG TO STORAGE-1 WITH INLINE HOMO", "MFG TO STORAGE-1 WITH INLINE FILTER PRES" => "MFG TRANSFER CYCLE DB"."PV PARAMETER"."MFG TO STORAGE-1 WITH INLINE FILTER PRES", "MFG TO STORAGE-2 WITH INLINE HOMO" => "MFG TRANSFER CYCLE DB"."PV PARAMETER"."MFG TO STORAGE-2 WITH INLINE HOMO", "MFG TO STORAGE-2 WITH INLINE FILTER PRES" => "MFG TRANSFER CYCLE DB"."PV PARAMETER"."MFG TO STORAGE-2 WITH INLINE FILTER PRES", "MFG TO STORAGE-3 WITH INLINE HOMO" => "MFG TRANSFER CYCLE DB"."PV PARAMETER"."MFG TO STORAGE-3 WITH INLINE HOMO", "MFG TO STORAGE-3 WITH INLINE FILTER PRES" => "MFG TRANSFER CYCLE DB"."PV PARAMETER"."MFG TO STORAGE-3 WITH INLINE FILTER PRES")
   END_RUNG
   // the same network as SCL:
   IF "AlwaysTRUE" THEN
       "HYST AND TEMP CUTOFF  DB"."HYSTERISIS NEW_VALUE"."SYRUP MFG_LOAD CELL" := "HYST AND TEMP CUTOFF  DB"."MAN SET"."MFG MOVE PV LOAD CELL" - "HYST AND TEMP CUTOFF  DB"."MAIN SET PARA"."SYRUP MFG_LOAD CELL";
       "@MFG TRANSFER LOAD CALCULATE PV"("MODE SELECTION" := "MODE SELECTION DB"."MODE BUFF",
                               "AUTO TRANSFER_1" := "MFG TRANSFER CYCLE DB".TRANSFER."TRANSFER BUFF"."MFG TO STORAGE-1 WITH INLINE HOMO",
                               "AUTO TRANSFER_2" := "MFG TRANSFER CYCLE DB".TRANSFER."TRANSFER BUFF"."MFG TO STORAGE-1 WITH INLINE FILTER PRES",
                               "AUTO TRANSFER_3" := "MFG TRANSFER CYCLE DB".TRANSFER."TRANSFER BUFF"."MFG TO STORAGE-2 WITH INLINE HOMO",
                               "AUTO TRANSFER_4" := "MFG TRANSFER CYCLE DB".TRANSFER."TRANSFER BUFF"."MFG TO STORAGE-2 WITH INLINE FILTER PRES",
                               "AUTO TRANSFER_5" := "MFG TRANSFER CYCLE DB".TRANSFER."TRANSFER BUFF"."MFG TO STORAGE-2 WITH INLINE HOMO",
                               "AUTO TRANSFER_6" := "MFG TRANSFER CYCLE DB".TRANSFER."TRANSFER BUFF"."MFG TO STORAGE-3 WITH INLINE FILTER PRES",
                               "MOVE PV LOAD CELL" := "HYST AND TEMP CUTOFF  DB"."MAN SET"."MFG MOVE PV LOAD CELL",
                               "LOAD CELL PV" := "AI SCALING DB".PV."SYRUP LOAD CELL",
                               MANUAL => "HYST AND TEMP CUTOFF  DB"."MFG CALCULATE PV",
                               "MFG TO STORAGE-1 WITH INLINE HOMO" => "MFG TRANSFER CYCLE DB"."PV PARAMETER"."MFG TO STORAGE-1 WITH INLINE HOMO",
                               "MFG TO STORAGE-1 WITH INLINE FILTER PRES" => "MFG TRANSFER CYCLE DB"."PV PARAMETER"."MFG TO STORAGE-1 WITH INLINE FILTER PRES",
                               "MFG TO STORAGE-2 WITH INLINE HOMO" => "MFG TRANSFER CYCLE DB"."PV PARAMETER"."MFG TO STORAGE-2 WITH INLINE HOMO",
                               "MFG TO STORAGE-2 WITH INLINE FILTER PRES" => "MFG TRANSFER CYCLE DB"."PV PARAMETER"."MFG TO STORAGE-2 WITH INLINE FILTER PRES",
                               "MFG TO STORAGE-3 WITH INLINE HOMO" => "MFG TRANSFER CYCLE DB"."PV PARAMETER"."MFG TO STORAGE-3 WITH INLINE HOMO",
                               "MFG TO STORAGE-3 WITH INLINE FILTER PRES" => "MFG TRANSFER CYCLE DB"."PV PARAMETER"."MFG TO STORAGE-3 WITH INLINE FILTER PRES");
   END_IF;
END_REGION

REGION Network 15: TRANSFER LOAD CUT OFF
   RUNG wire#powerrail
      Contact( "AlwaysTRUE" )
      wire#w1
      { S7_Templates := "SrcType := Real" } LE_Contact(in1 := "AI SCALING DB".PV."SYRUP LOAD CELL", in2 := "HYST AND TEMP CUTOFF  DB"."HYSTERISIS NEW_VALUE"."SYRUP MFG_LOAD CELL")
      Move(in := 1, out1 => "LEVEL BUFF"."SYRUP MFG_LOAD CELL")
   END_RUNG
   RUNG wire#w1
      { S7_Templates := "SrcType := Real" } GT_Contact(in1 := "AI SCALING DB".PV."SYRUP LOAD CELL", in2 := "HYST AND TEMP CUTOFF  DB"."HYSTERISIS NEW_VALUE"."SYRUP MFG_LOAD CELL")
      Move(in := 0, out1 => "LEVEL BUFF"."SYRUP MFG_LOAD CELL")
   END_RUNG
   // the same network as SCL:
   IF "AlwaysTRUE" AND ("AI SCALING DB".PV."SYRUP LOAD CELL" <= "HYST AND TEMP CUTOFF  DB"."HYSTERISIS NEW_VALUE"."SYRUP MFG_LOAD CELL") THEN
       "LEVEL BUFF"."SYRUP MFG_LOAD CELL" := 1;
   END_IF;
   IF "AlwaysTRUE" AND ("AI SCALING DB".PV."SYRUP LOAD CELL" > "HYST AND TEMP CUTOFF  DB"."HYSTERISIS NEW_VALUE"."SYRUP MFG_LOAD CELL") THEN
       "LEVEL BUFF"."SYRUP MFG_LOAD CELL" := 0;
   END_IF;
END_REGION

REGION Network 17: MFG TEMP MIN_MAX BUFF
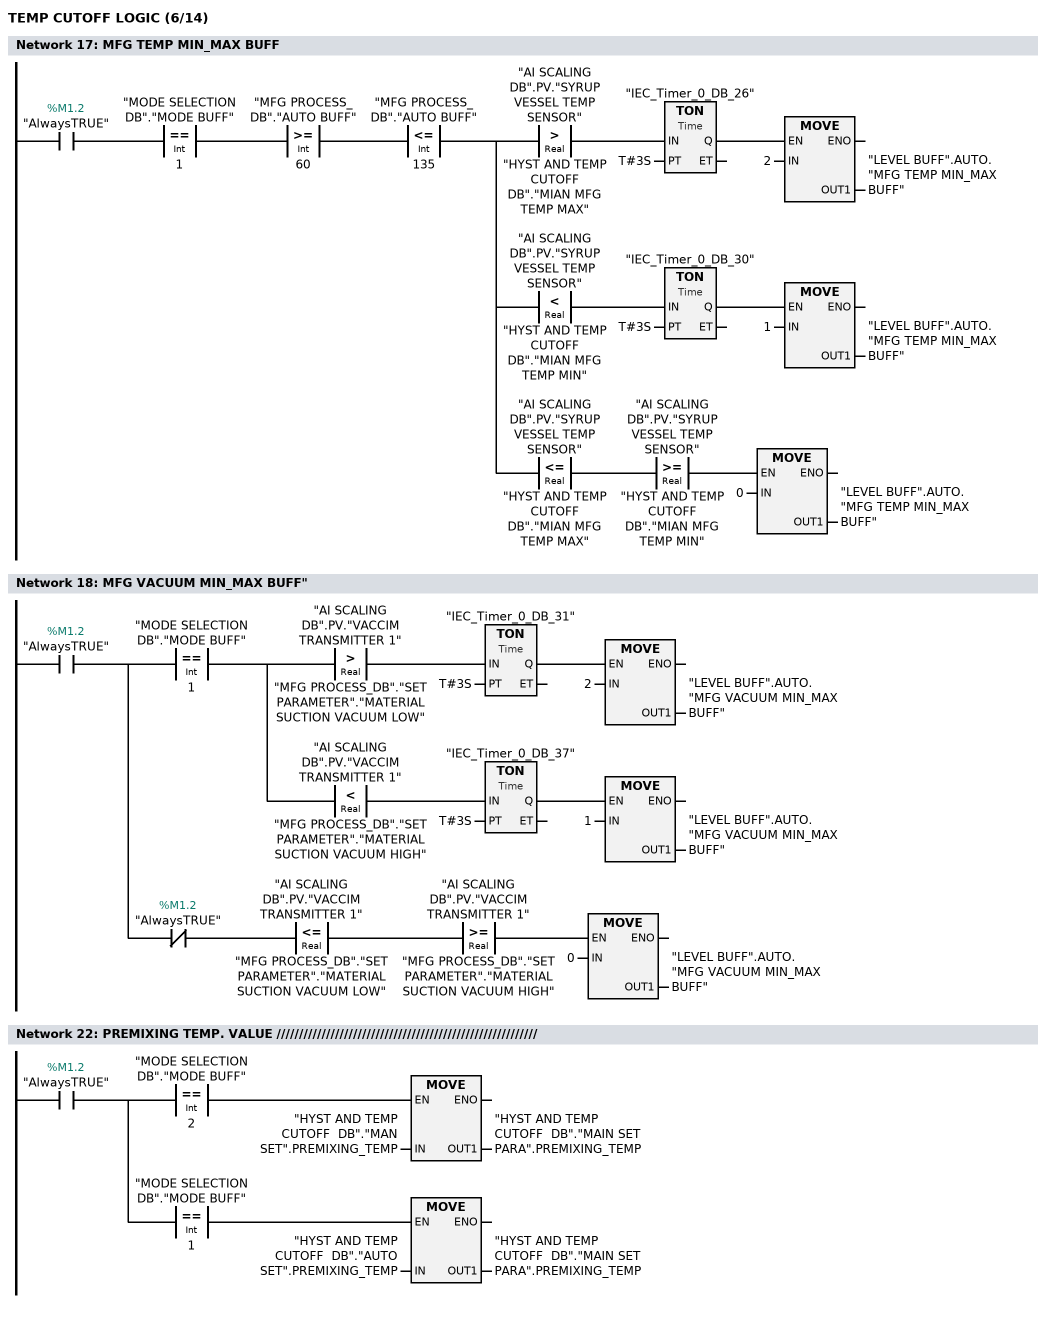
   RUNG wire#powerrail
      Contact( "AlwaysTRUE" )
      { S7_Templates := "SrcType := Int" } EQ_Contact(in1 := "MODE SELECTION DB"."MODE BUFF", in2 := 1)
      { S7_Templates := "SrcType := Int" } GE_Contact(in1 := "MFG PROCESS_DB"."AUTO BUFF", in2 := 60)
      { S7_Templates := "SrcType := Int" } LE_Contact(in1 := "MFG PROCESS_DB"."AUTO BUFF", in2 := 135)
      wire#w1
      { S7_Templates := "SrcType := Real" } GT_Contact(in1 := "AI SCALING DB".PV."SYRUP VESSEL TEMP SENSOR", in2 := "HYST AND TEMP CUTOFF  DB"."MIAN MFG TEMP MAX")
      { S7_Templates := "time_type := Time" } "IEC_Timer_0_DB_26".TON(pt := T#3S, et =>)
      Move(in := 2, out1 => "LEVEL BUFF".AUTO."MFG TEMP MIN_MAX BUFF")
   END_RUNG
   RUNG wire#w1
      { S7_Templates := "SrcType := Real" } LT_Contact(in1 := "AI SCALING DB".PV."SYRUP VESSEL TEMP SENSOR", in2 := "HYST AND TEMP CUTOFF  DB"."MIAN MFG TEMP MIN")
      { S7_Templates := "time_type := Time" } "IEC_Timer_0_DB_30".TON(pt := T#3S, et =>)
      Move(in := 1, out1 => "LEVEL BUFF".AUTO."MFG TEMP MIN_MAX BUFF")
   END_RUNG
   RUNG wire#w1
      { S7_Templates := "SrcType := Real" } LE_Contact(in1 := "AI SCALING DB".PV."SYRUP VESSEL TEMP SENSOR", in2 := "HYST AND TEMP CUTOFF  DB"."MIAN MFG TEMP MAX")
      { S7_Templates := "SrcType := Real" } GE_Contact(in1 := "AI SCALING DB".PV."SYRUP VESSEL TEMP SENSOR", in2 := "HYST AND TEMP CUTOFF  DB"."MIAN MFG TEMP MIN")
      Move(in := 0, out1 => "LEVEL BUFF".AUTO."MFG TEMP MIN_MAX BUFF")
   END_RUNG
   // the same network as SCL:
   #_w1 := "AlwaysTRUE" AND ("MODE SELECTION DB"."MODE BUFF" = 1) AND ("MFG PROCESS_DB"."AUTO BUFF" >= 60) AND ("MFG PROCESS_DB"."AUTO BUFF" <= 135);
   "IEC_Timer_0_DB_26".TON(IN := #_w1 AND ("AI SCALING DB".PV."SYRUP VESSEL TEMP SENSOR" > "HYST AND TEMP CUTOFF  DB"."MIAN MFG TEMP MAX"),
                           PT := T#3S);
   IF "IEC_Timer_0_DB_26".Q THEN "LEVEL BUFF".AUTO."MFG TEMP MIN_MAX BUFF" := 2; END_IF;
   "IEC_Timer_0_DB_30".TON(IN := #_w1 AND ("AI SCALING DB".PV."SYRUP VESSEL TEMP SENSOR" < "HYST AND TEMP CUTOFF  DB"."MIAN MFG TEMP MIN"),
                           PT := T#3S);
   IF "IEC_Timer_0_DB_30".Q THEN "LEVEL BUFF".AUTO."MFG TEMP MIN_MAX BUFF" := 1; END_IF;
   IF #_w1 AND ("AI SCALING DB".PV."SYRUP VESSEL TEMP SENSOR" <= "HYST AND TEMP CUTOFF  DB"."MIAN MFG TEMP MAX") AND ("AI SCALING DB".PV."SYRUP VESSEL TEMP SENSOR" >= "HYST AND TEMP CUTOFF  DB"."MIAN MFG TEMP MIN") THEN
       "LEVEL BUFF".AUTO."MFG TEMP MIN_MAX BUFF" := 0;
   END_IF;
END_REGION

REGION Network 18: MFG VACUUM MIN_MAX BUFF"
   RUNG wire#powerrail
      Contact( "AlwaysTRUE" )
      wire#w1
      { S7_Templates := "SrcType := Int" } EQ_Contact(in1 := "MODE SELECTION DB"."MODE BUFF", in2 := 1)
      wire#w2
      { S7_Templates := "SrcType := Real" } GT_Contact(in1 := "AI SCALING DB".PV."VACCIM TRANSMITTER 1", in2 := "MFG PROCESS_DB"."SET PARAMETER"."MATERIAL SUCTION VACUUM LOW")
      { S7_Templates := "time_type := Time" } "IEC_Timer_0_DB_31".TON(pt := T#3S, et =>)
      Move(in := 2, out1 => "LEVEL BUFF".AUTO."MFG VACUUM MIN_MAX BUFF")
   END_RUNG
   RUNG wire#w2
      { S7_Templates := "SrcType := Real" } LT_Contact(in1 := "AI SCALING DB".PV."VACCIM TRANSMITTER 1", in2 := "MFG PROCESS_DB"."SET PARAMETER"."MATERIAL SUCTION VACUUM HIGH")
      { S7_Templates := "time_type := Time" } "IEC_Timer_0_DB_37".TON(pt := T#3S, et =>)
      Move(in := 1, out1 => "LEVEL BUFF".AUTO."MFG VACUUM MIN_MAX BUFF")
   END_RUNG
   RUNG wire#w1
      I_Contact( "AlwaysTRUE" )
      { S7_Templates := "SrcType := Real" } LE_Contact(in1 := "AI SCALING DB".PV."VACCIM TRANSMITTER 1", in2 := "MFG PROCESS_DB"."SET PARAMETER"."MATERIAL SUCTION VACUUM LOW")
      { S7_Templates := "SrcType := Real" } GE_Contact(in1 := "AI SCALING DB".PV."VACCIM TRANSMITTER 1", in2 := "MFG PROCESS_DB"."SET PARAMETER"."MATERIAL SUCTION VACUUM HIGH")
      Move(in := 0, out1 => "LEVEL BUFF".AUTO."MFG VACUUM MIN_MAX BUFF")
   END_RUNG
   // the same network as SCL:
   #_w1 := "AlwaysTRUE" AND ("MODE SELECTION DB"."MODE BUFF" = 1);
   "IEC_Timer_0_DB_31".TON(IN := #_w1 AND ("AI SCALING DB".PV."VACCIM TRANSMITTER 1" > "MFG PROCESS_DB"."SET PARAMETER"."MATERIAL SUCTION VACUUM LOW"),
                           PT := T#3S);
   IF "IEC_Timer_0_DB_31".Q THEN "LEVEL BUFF".AUTO."MFG VACUUM MIN_MAX BUFF" := 2; END_IF;
   "IEC_Timer_0_DB_37".TON(IN := #_w1 AND ("AI SCALING DB".PV."VACCIM TRANSMITTER 1" < "MFG PROCESS_DB"."SET PARAMETER"."MATERIAL SUCTION VACUUM HIGH"),
                           PT := T#3S);
   IF "IEC_Timer_0_DB_37".Q THEN "LEVEL BUFF".AUTO."MFG VACUUM MIN_MAX BUFF" := 1; END_IF;
   IF "AlwaysTRUE" AND NOT "AlwaysTRUE" AND ("AI SCALING DB".PV."VACCIM TRANSMITTER 1" <= "MFG PROCESS_DB"."SET PARAMETER"."MATERIAL SUCTION VACUUM LOW") AND ("AI SCALING DB".PV."VACCIM TRANSMITTER 1" >= "MFG PROCESS_DB"."SET PARAMETER"."MATERIAL SUCTION VACUUM HIGH") THEN
       "LEVEL BUFF".AUTO."MFG VACUUM MIN_MAX BUFF" := 0;
   END_IF;
END_REGION

REGION Network 22: PREMIXING TEMP. VALUE //////////////////////////////////////////////////////////
   RUNG wire#powerrail
      Contact( "AlwaysTRUE" )
      wire#w1
      { S7_Templates := "SrcType := Int" } EQ_Contact(in1 := "MODE SELECTION DB"."MODE BUFF", in2 := 2)
      Move(in := "HYST AND TEMP CUTOFF  DB"."MAN SET".PREMIXING_TEMP, out1 => "HYST AND TEMP CUTOFF  DB"."MAIN SET PARA".PREMIXING_TEMP)
   END_RUNG
   RUNG wire#w1
      { S7_Templates := "SrcType := Int" } EQ_Contact(in1 := "MODE SELECTION DB"."MODE BUFF", in2 := 1)
      Move(in := "HYST AND TEMP CUTOFF  DB"."AUTO SET".PREMIXING_TEMP, out1 => "HYST AND TEMP CUTOFF  DB"."MAIN SET PARA".PREMIXING_TEMP)
   END_RUNG
   // the same network as SCL:
   IF "AlwaysTRUE" AND ("MODE SELECTION DB"."MODE BUFF" = 2) THEN
       "HYST AND TEMP CUTOFF  DB"."MAIN SET PARA".PREMIXING_TEMP := "HYST AND TEMP CUTOFF  DB"."MAN SET".PREMIXING_TEMP;
   END_IF;
   IF "AlwaysTRUE" AND ("MODE SELECTION DB"."MODE BUFF" = 1) THEN
       "HYST AND TEMP CUTOFF  DB"."MAIN SET PARA".PREMIXING_TEMP := "HYST AND TEMP CUTOFF  DB"."AUTO SET".PREMIXING_TEMP;
   END_IF;
END_REGION

REGION Network 23: SUB HYSTERISIS
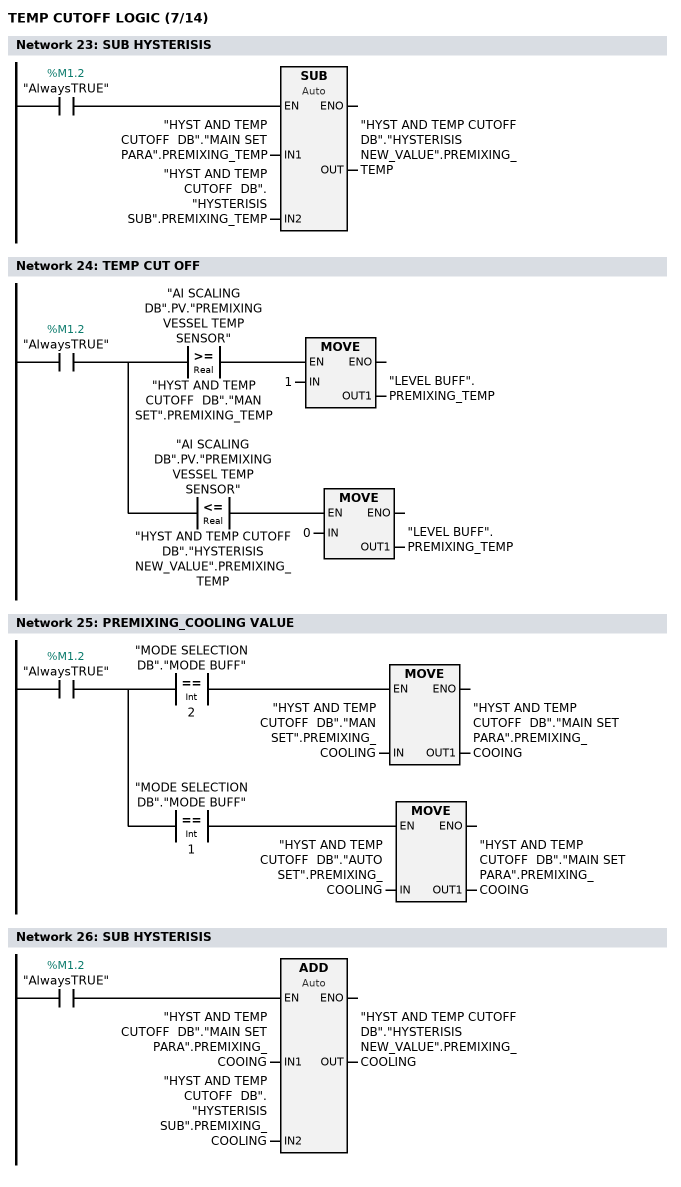
   RUNG wire#powerrail
      Contact( "AlwaysTRUE" )
      Sub(in1 := "HYST AND TEMP CUTOFF  DB"."MAIN SET PARA".PREMIXING_TEMP, in2 := "HYST AND TEMP CUTOFF  DB"."HYSTERISIS SUB".PREMIXING_TEMP, out => "HYST AND TEMP CUTOFF  DB"."HYSTERISIS NEW_VALUE".PREMIXING_TEMP)
   END_RUNG
   // the same network as SCL:
   IF "AlwaysTRUE" THEN
       "HYST AND TEMP CUTOFF  DB"."HYSTERISIS NEW_VALUE".PREMIXING_TEMP := "HYST AND TEMP CUTOFF  DB"."MAIN SET PARA".PREMIXING_TEMP - "HYST AND TEMP CUTOFF  DB"."HYSTERISIS SUB".PREMIXING_TEMP;
   END_IF;
END_REGION

REGION Network 24: TEMP CUT OFF
   RUNG wire#powerrail
      Contact( "AlwaysTRUE" )
      wire#w1
      { S7_Templates := "SrcType := Real" } GE_Contact(in1 := "AI SCALING DB".PV."PREMIXING VESSEL TEMP SENSOR", in2 := "HYST AND TEMP CUTOFF  DB"."MAN SET".PREMIXING_TEMP)
      Move(in := 1, out1 => "LEVEL BUFF".PREMIXING_TEMP)
   END_RUNG
   RUNG wire#w1
      { S7_Templates := "SrcType := Real" } LE_Contact(in1 := "AI SCALING DB".PV."PREMIXING VESSEL TEMP SENSOR", in2 := "HYST AND TEMP CUTOFF  DB"."HYSTERISIS NEW_VALUE".PREMIXING_TEMP)
      Move(in := 0, out1 => "LEVEL BUFF".PREMIXING_TEMP)
   END_RUNG
   // the same network as SCL:
   IF "AlwaysTRUE" AND ("AI SCALING DB".PV."PREMIXING VESSEL TEMP SENSOR" >= "HYST AND TEMP CUTOFF  DB"."MAN SET".PREMIXING_TEMP) THEN
       "LEVEL BUFF".PREMIXING_TEMP := 1;
   END_IF;
   IF "AlwaysTRUE" AND ("AI SCALING DB".PV."PREMIXING VESSEL TEMP SENSOR" <= "HYST AND TEMP CUTOFF  DB"."HYSTERISIS NEW_VALUE".PREMIXING_TEMP) THEN
       "LEVEL BUFF".PREMIXING_TEMP := 0;
   END_IF;
END_REGION

REGION Network 25: PREMIXING_COOLING VALUE
   RUNG wire#powerrail
      Contact( "AlwaysTRUE" )
      wire#w1
      { S7_Templates := "SrcType := Int" } EQ_Contact(in1 := "MODE SELECTION DB"."MODE BUFF", in2 := 2)
      Move(in := "HYST AND TEMP CUTOFF  DB"."MAN SET".PREMIXING_COOLING, out1 => "HYST AND TEMP CUTOFF  DB"."MAIN SET PARA".PREMIXING_COOING)
   END_RUNG
   RUNG wire#w1
      { S7_Templates := "SrcType := Int" } EQ_Contact(in1 := "MODE SELECTION DB"."MODE BUFF", in2 := 1)
      Move(in := "HYST AND TEMP CUTOFF  DB"."AUTO SET".PREMIXING_COOLING, out1 => "HYST AND TEMP CUTOFF  DB"."MAIN SET PARA".PREMIXING_COOING)
   END_RUNG
   // the same network as SCL:
   IF "AlwaysTRUE" AND ("MODE SELECTION DB"."MODE BUFF" = 2) THEN
       "HYST AND TEMP CUTOFF  DB"."MAIN SET PARA".PREMIXING_COOING := "HYST AND TEMP CUTOFF  DB"."MAN SET".PREMIXING_COOLING;
   END_IF;
   IF "AlwaysTRUE" AND ("MODE SELECTION DB"."MODE BUFF" = 1) THEN
       "HYST AND TEMP CUTOFF  DB"."MAIN SET PARA".PREMIXING_COOING := "HYST AND TEMP CUTOFF  DB"."AUTO SET".PREMIXING_COOLING;
   END_IF;
END_REGION

REGION Network 26: SUB HYSTERISIS
   RUNG wire#powerrail
      Contact( "AlwaysTRUE" )
      Add(in1 := "HYST AND TEMP CUTOFF  DB"."MAIN SET PARA".PREMIXING_COOING, in2 := "HYST AND TEMP CUTOFF  DB"."HYSTERISIS SUB".PREMIXING_COOLING, out => "HYST AND TEMP CUTOFF  DB"."HYSTERISIS NEW_VALUE".PREMIXING_COOLING)
   END_RUNG
   // the same network as SCL:
   IF "AlwaysTRUE" THEN
       "HYST AND TEMP CUTOFF  DB"."HYSTERISIS NEW_VALUE".PREMIXING_COOLING := "HYST AND TEMP CUTOFF  DB"."MAIN SET PARA".PREMIXING_COOING + "HYST AND TEMP CUTOFF  DB"."HYSTERISIS SUB".PREMIXING_COOLING;
   END_IF;
END_REGION

REGION Network 27: TEMP CUT OFF
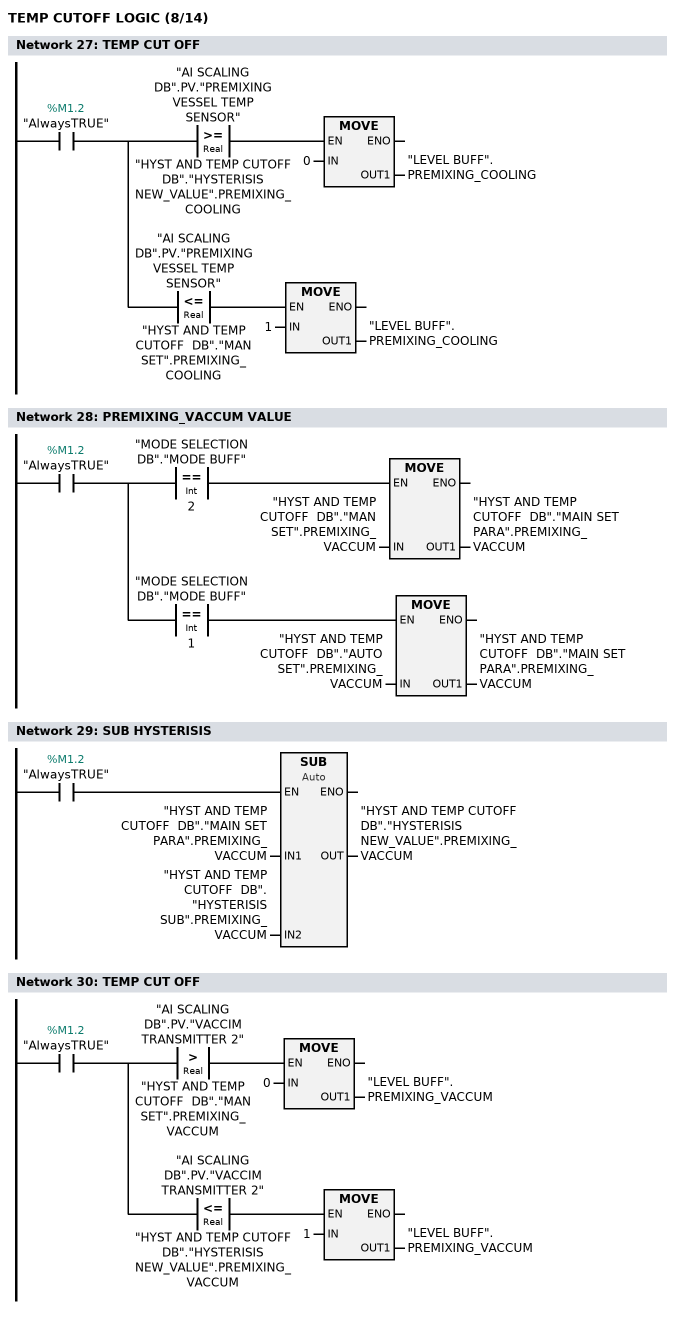
   RUNG wire#powerrail
      Contact( "AlwaysTRUE" )
      wire#w1
      { S7_Templates := "SrcType := Real" } GE_Contact(in1 := "AI SCALING DB".PV."PREMIXING VESSEL TEMP SENSOR", in2 := "HYST AND TEMP CUTOFF  DB"."HYSTERISIS NEW_VALUE".PREMIXING_COOLING)
      Move(in := 0, out1 => "LEVEL BUFF".PREMIXING_COOLING)
   END_RUNG
   RUNG wire#w1
      { S7_Templates := "SrcType := Real" } LE_Contact(in1 := "AI SCALING DB".PV."PREMIXING VESSEL TEMP SENSOR", in2 := "HYST AND TEMP CUTOFF  DB"."MAN SET".PREMIXING_COOLING)
      Move(in := 1, out1 => "LEVEL BUFF".PREMIXING_COOLING)
   END_RUNG
   // the same network as SCL:
   IF "AlwaysTRUE" AND ("AI SCALING DB".PV."PREMIXING VESSEL TEMP SENSOR" >= "HYST AND TEMP CUTOFF  DB"."HYSTERISIS NEW_VALUE".PREMIXING_COOLING) THEN
       "LEVEL BUFF".PREMIXING_COOLING := 0;
   END_IF;
   IF "AlwaysTRUE" AND ("AI SCALING DB".PV."PREMIXING VESSEL TEMP SENSOR" <= "HYST AND TEMP CUTOFF  DB"."MAN SET".PREMIXING_COOLING) THEN
       "LEVEL BUFF".PREMIXING_COOLING := 1;
   END_IF;
END_REGION

REGION Network 28: PREMIXING_VACCUM VALUE
   RUNG wire#powerrail
      Contact( "AlwaysTRUE" )
      wire#w1
      { S7_Templates := "SrcType := Int" } EQ_Contact(in1 := "MODE SELECTION DB"."MODE BUFF", in2 := 2)
      Move(in := "HYST AND TEMP CUTOFF  DB"."MAN SET".PREMIXING_VACCUM, out1 => "HYST AND TEMP CUTOFF  DB"."MAIN SET PARA".PREMIXING_VACCUM)
   END_RUNG
   RUNG wire#w1
      { S7_Templates := "SrcType := Int" } EQ_Contact(in1 := "MODE SELECTION DB"."MODE BUFF", in2 := 1)
      Move(in := "HYST AND TEMP CUTOFF  DB"."AUTO SET".PREMIXING_VACCUM, out1 => "HYST AND TEMP CUTOFF  DB"."MAIN SET PARA".PREMIXING_VACCUM)
   END_RUNG
   // the same network as SCL:
   IF "AlwaysTRUE" AND ("MODE SELECTION DB"."MODE BUFF" = 2) THEN
       "HYST AND TEMP CUTOFF  DB"."MAIN SET PARA".PREMIXING_VACCUM := "HYST AND TEMP CUTOFF  DB"."MAN SET".PREMIXING_VACCUM;
   END_IF;
   IF "AlwaysTRUE" AND ("MODE SELECTION DB"."MODE BUFF" = 1) THEN
       "HYST AND TEMP CUTOFF  DB"."MAIN SET PARA".PREMIXING_VACCUM := "HYST AND TEMP CUTOFF  DB"."AUTO SET".PREMIXING_VACCUM;
   END_IF;
END_REGION

REGION Network 29: SUB HYSTERISIS
   RUNG wire#powerrail
      Contact( "AlwaysTRUE" )
      Sub(in1 := "HYST AND TEMP CUTOFF  DB"."MAIN SET PARA".PREMIXING_VACCUM, in2 := "HYST AND TEMP CUTOFF  DB"."HYSTERISIS SUB".PREMIXING_VACCUM, out => "HYST AND TEMP CUTOFF  DB"."HYSTERISIS NEW_VALUE".PREMIXING_VACCUM)
   END_RUNG
   // the same network as SCL:
   IF "AlwaysTRUE" THEN
       "HYST AND TEMP CUTOFF  DB"."HYSTERISIS NEW_VALUE".PREMIXING_VACCUM := "HYST AND TEMP CUTOFF  DB"."MAIN SET PARA".PREMIXING_VACCUM - "HYST AND TEMP CUTOFF  DB"."HYSTERISIS SUB".PREMIXING_VACCUM;
   END_IF;
END_REGION

REGION Network 30: TEMP CUT OFF
   RUNG wire#powerrail
      Contact( "AlwaysTRUE" )
      wire#w1
      { S7_Templates := "SrcType := Real" } GT_Contact(in1 := "AI SCALING DB".PV."VACCIM TRANSMITTER 2", in2 := "HYST AND TEMP CUTOFF  DB"."MAN SET".PREMIXING_VACCUM)
      Move(in := 0, out1 => "LEVEL BUFF".PREMIXING_VACCUM)
   END_RUNG
   RUNG wire#w1
      { S7_Templates := "SrcType := Real" } LE_Contact(in1 := "AI SCALING DB".PV."VACCIM TRANSMITTER 2", in2 := "HYST AND TEMP CUTOFF  DB"."HYSTERISIS NEW_VALUE".PREMIXING_VACCUM)
      Move(in := 1, out1 => "LEVEL BUFF".PREMIXING_VACCUM)
   END_RUNG
   // the same network as SCL:
   IF "AlwaysTRUE" AND ("AI SCALING DB".PV."VACCIM TRANSMITTER 2" > "HYST AND TEMP CUTOFF  DB"."MAN SET".PREMIXING_VACCUM) THEN
       "LEVEL BUFF".PREMIXING_VACCUM := 0;
   END_IF;
   IF "AlwaysTRUE" AND ("AI SCALING DB".PV."VACCIM TRANSMITTER 2" <= "HYST AND TEMP CUTOFF  DB"."HYSTERISIS NEW_VALUE".PREMIXING_VACCUM) THEN
       "LEVEL BUFF".PREMIXING_VACCUM := 1;
   END_IF;
END_REGION

REGION Network 31: AUTO PREMIXING_LOAD CELL VALUE
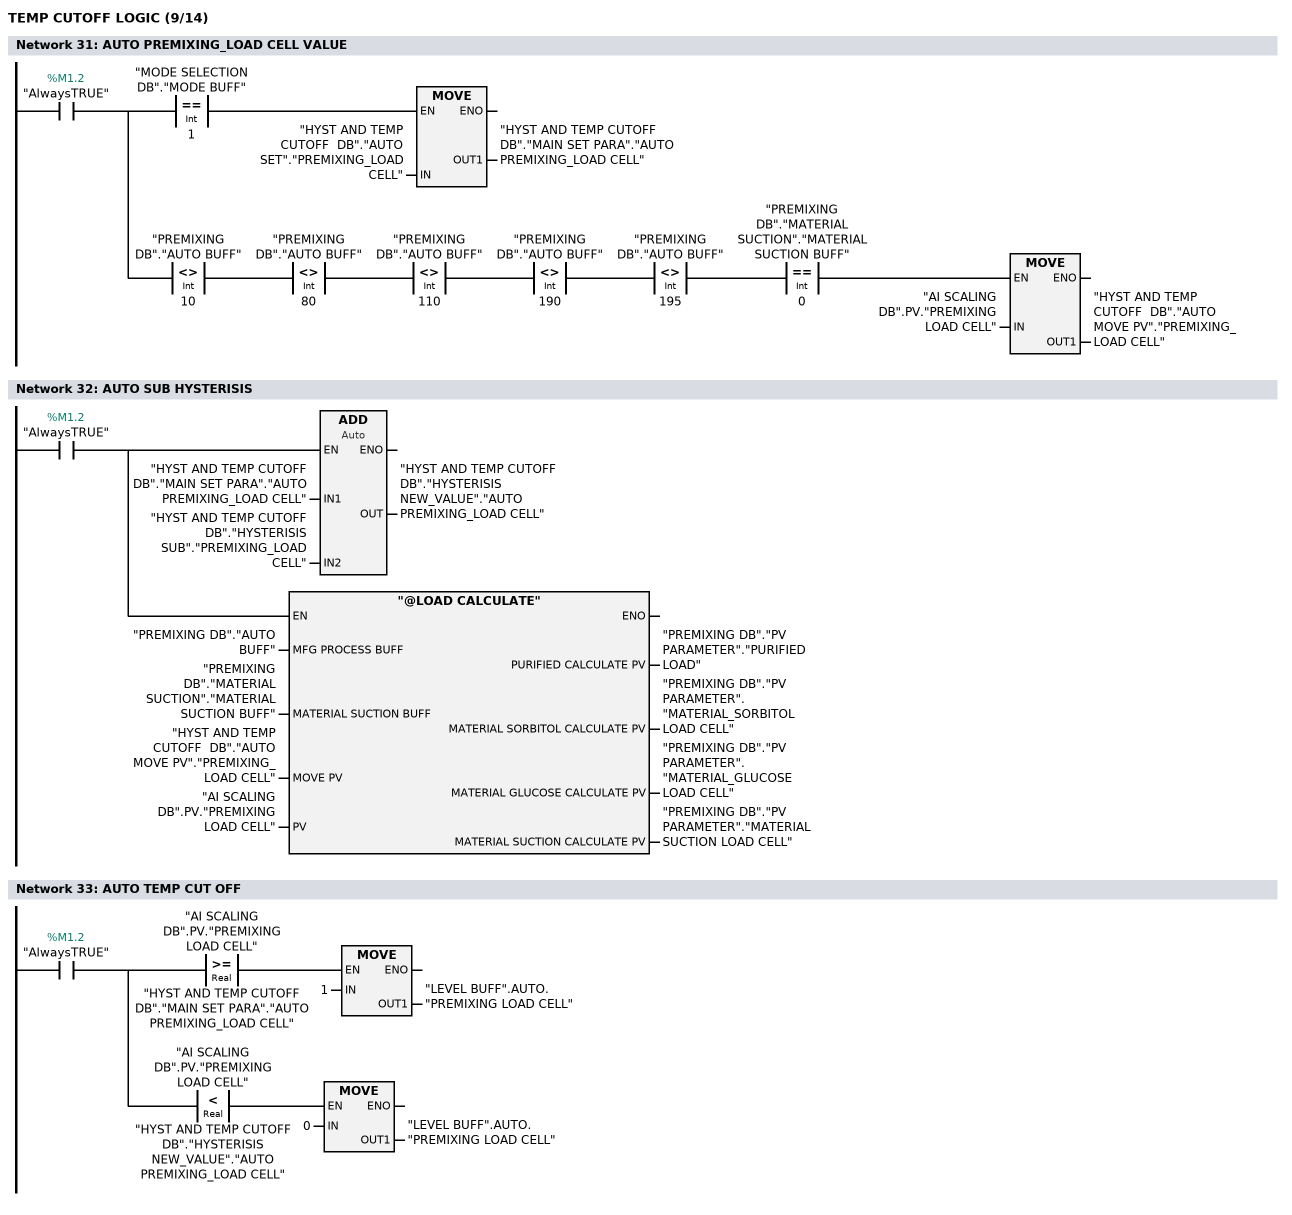
   RUNG wire#powerrail
      Contact( "AlwaysTRUE" )
      wire#w1
      { S7_Templates := "SrcType := Int" } EQ_Contact(in1 := "MODE SELECTION DB"."MODE BUFF", in2 := 1)
      Move(in := "HYST AND TEMP CUTOFF  DB"."AUTO SET"."PREMIXING_LOAD CELL", out1 => "HYST AND TEMP CUTOFF  DB"."MAIN SET PARA"."AUTO PREMIXING_LOAD CELL")
   END_RUNG
   RUNG wire#w1
      { S7_Templates := "SrcType := Int" } NE_Contact(in1 := "PREMIXING DB"."AUTO BUFF", in2 := 10)
      { S7_Templates := "SrcType := Int" } NE_Contact(in1 := "PREMIXING DB"."AUTO BUFF", in2 := 80)
      { S7_Templates := "SrcType := Int" } NE_Contact(in1 := "PREMIXING DB"."AUTO BUFF", in2 := 110)
      { S7_Templates := "SrcType := Int" } NE_Contact(in1 := "PREMIXING DB"."AUTO BUFF", in2 := 190)
      { S7_Templates := "SrcType := Int" } NE_Contact(in1 := "PREMIXING DB"."AUTO BUFF", in2 := 195)
      { S7_Templates := "SrcType := Int" } EQ_Contact(in1 := "PREMIXING DB"."MATERIAL SUCTION"."MATERIAL SUCTION BUFF", in2 := 0)
      Move(in := "AI SCALING DB".PV."PREMIXING LOAD CELL", out1 => "HYST AND TEMP CUTOFF  DB"."AUTO MOVE PV"."PREMIXING_LOAD CELL")
   END_RUNG
   // the same network as SCL:
   IF "AlwaysTRUE" AND ("MODE SELECTION DB"."MODE BUFF" = 1) THEN
       "HYST AND TEMP CUTOFF  DB"."MAIN SET PARA"."AUTO PREMIXING_LOAD CELL" := "HYST AND TEMP CUTOFF  DB"."AUTO SET"."PREMIXING_LOAD CELL";
   END_IF;
   IF "AlwaysTRUE" AND ("PREMIXING DB"."AUTO BUFF" <> 10) AND ("PREMIXING DB"."AUTO BUFF" <> 80) AND ("PREMIXING DB"."AUTO BUFF" <> 110) AND ("PREMIXING DB"."AUTO BUFF" <> 190) AND ("PREMIXING DB"."AUTO BUFF" <> 195) AND ("PREMIXING DB"."MATERIAL SUCTION"."MATERIAL SUCTION BUFF" = 0) THEN
       "HYST AND TEMP CUTOFF  DB"."AUTO MOVE PV"."PREMIXING_LOAD CELL" := "AI SCALING DB".PV."PREMIXING LOAD CELL";
   END_IF;
END_REGION

REGION Network 32: AUTO SUB HYSTERISIS
   RUNG wire#powerrail
      Contact( "AlwaysTRUE" )
      wire#w1
      Add(in1 := "HYST AND TEMP CUTOFF  DB"."MAIN SET PARA"."AUTO PREMIXING_LOAD CELL", in2 := "HYST AND TEMP CUTOFF  DB"."HYSTERISIS SUB"."PREMIXING_LOAD CELL", out => "HYST AND TEMP CUTOFF  DB"."HYSTERISIS NEW_VALUE"."AUTO PREMIXING_LOAD CELL")
   END_RUNG
   RUNG wire#w1
      "@LOAD CALCULATE"("MFG PROCESS BUFF" := "PREMIXING DB"."AUTO BUFF", "MATERIAL SUCTION BUFF" := "PREMIXING DB"."MATERIAL SUCTION"."MATERIAL SUCTION BUFF", "MOVE PV" := "HYST AND TEMP CUTOFF  DB"."AUTO MOVE PV"."PREMIXING_LOAD CELL", PV := "AI SCALING DB".PV."PREMIXING LOAD CELL", "PURIFIED CALCULATE PV" => "PREMIXING DB"."PV PARAMETER"."PURIFIED LOAD", "MATERIAL SORBITOL CALCULATE PV" => "PREMIXING DB"."PV PARAMETER"."MATERIAL_SORBITOL LOAD CELL", "MATERIAL GLUCOSE CALCULATE PV" => "PREMIXING DB"."PV PARAMETER"."MATERIAL_GLUCOSE LOAD CELL", "MATERIAL SUCTION CALCULATE PV" => "PREMIXING DB"."PV PARAMETER"."MATERIAL SUCTION LOAD CELL")
   END_RUNG
   // the same network as SCL:
   IF "AlwaysTRUE" THEN
       "HYST AND TEMP CUTOFF  DB"."HYSTERISIS NEW_VALUE"."AUTO PREMIXING_LOAD CELL" := "HYST AND TEMP CUTOFF  DB"."MAIN SET PARA"."AUTO PREMIXING_LOAD CELL" + "HYST AND TEMP CUTOFF  DB"."HYSTERISIS SUB"."PREMIXING_LOAD CELL";
       "@LOAD CALCULATE"("MFG PROCESS BUFF" := "PREMIXING DB"."AUTO BUFF",
                         "MATERIAL SUCTION BUFF" := "PREMIXING DB"."MATERIAL SUCTION"."MATERIAL SUCTION BUFF",
                         "MOVE PV" := "HYST AND TEMP CUTOFF  DB"."AUTO MOVE PV"."PREMIXING_LOAD CELL",
                         PV := "AI SCALING DB".PV."PREMIXING LOAD CELL",
                         "PURIFIED CALCULATE PV" => "PREMIXING DB"."PV PARAMETER"."PURIFIED LOAD",
                         "MATERIAL SORBITOL CALCULATE PV" => "PREMIXING DB"."PV PARAMETER"."MATERIAL_SORBITOL LOAD CELL",
                         "MATERIAL GLUCOSE CALCULATE PV" => "PREMIXING DB"."PV PARAMETER"."MATERIAL_GLUCOSE LOAD CELL",
                         "MATERIAL SUCTION CALCULATE PV" => "PREMIXING DB"."PV PARAMETER"."MATERIAL SUCTION LOAD CELL");
   END_IF;
END_REGION

REGION Network 33: AUTO TEMP CUT OFF
   RUNG wire#powerrail
      Contact( "AlwaysTRUE" )
      wire#w1
      { S7_Templates := "SrcType := Real" } GE_Contact(in1 := "AI SCALING DB".PV."PREMIXING LOAD CELL", in2 := "HYST AND TEMP CUTOFF  DB"."MAIN SET PARA"."AUTO PREMIXING_LOAD CELL")
      Move(in := 1, out1 => "LEVEL BUFF".AUTO."PREMIXING LOAD CELL")
   END_RUNG
   RUNG wire#w1
      { S7_Templates := "SrcType := Real" } LT_Contact(in1 := "AI SCALING DB".PV."PREMIXING LOAD CELL", in2 := "HYST AND TEMP CUTOFF  DB"."HYSTERISIS NEW_VALUE"."AUTO PREMIXING_LOAD CELL")
      Move(in := 0, out1 => "LEVEL BUFF".AUTO."PREMIXING LOAD CELL")
   END_RUNG
   // the same network as SCL:
   IF "AlwaysTRUE" AND ("AI SCALING DB".PV."PREMIXING LOAD CELL" >= "HYST AND TEMP CUTOFF  DB"."MAIN SET PARA"."AUTO PREMIXING_LOAD CELL") THEN
       "LEVEL BUFF".AUTO."PREMIXING LOAD CELL" := 1;
   END_IF;
   IF "AlwaysTRUE" AND ("AI SCALING DB".PV."PREMIXING LOAD CELL" < "HYST AND TEMP CUTOFF  DB"."HYSTERISIS NEW_VALUE"."AUTO PREMIXING_LOAD CELL") THEN
       "LEVEL BUFF".AUTO."PREMIXING LOAD CELL" := 0;
   END_IF;
END_REGION

REGION Network 34: TRANSFER PREMIXING_LOAD CELL
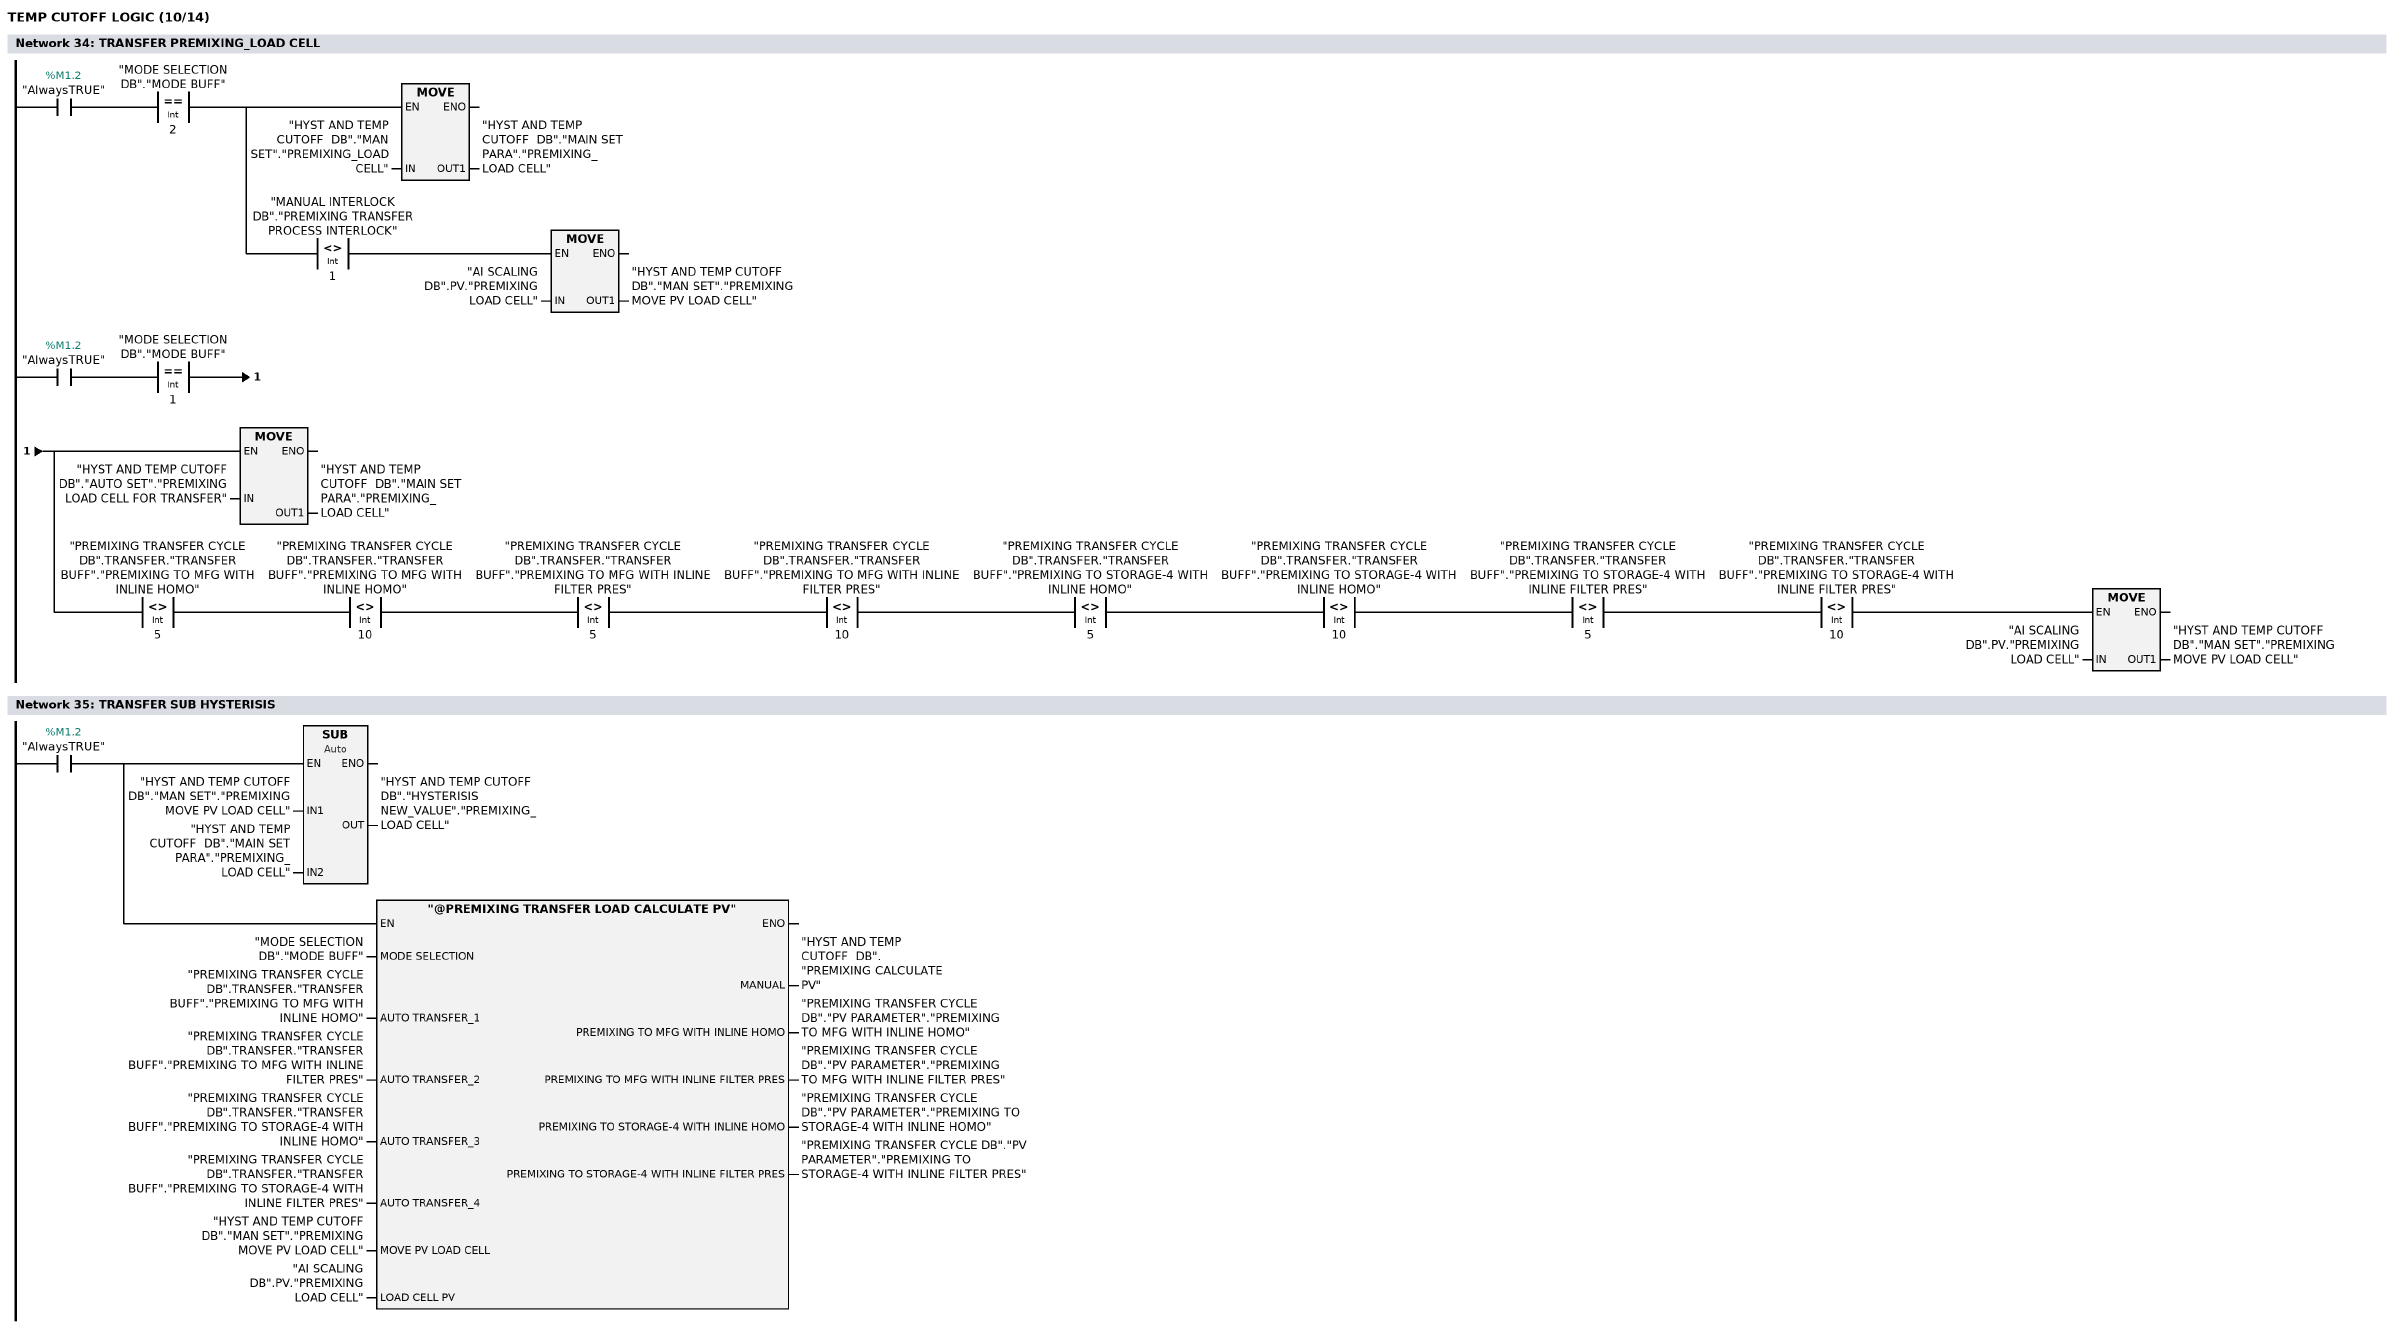
   RUNG wire#powerrail
      Contact( "AlwaysTRUE" )
      { S7_Templates := "SrcType := Int" } EQ_Contact(in1 := "MODE SELECTION DB"."MODE BUFF", in2 := 2)
      wire#w1
      Move(in := "HYST AND TEMP CUTOFF  DB"."MAN SET"."PREMIXING_LOAD CELL", out1 => "HYST AND TEMP CUTOFF  DB"."MAIN SET PARA"."PREMIXING_LOAD CELL")
   END_RUNG
   RUNG wire#w1
      { S7_Templates := "SrcType := Int" } NE_Contact(in1 := "MANUAL INTERLOCK DB"."PREMIXING TRANSFER PROCESS INTERLOCK", in2 := 1)
      Move(in := "AI SCALING DB".PV."PREMIXING LOAD CELL", out1 => "HYST AND TEMP CUTOFF  DB"."MAN SET"."PREMIXING MOVE PV LOAD CELL")
   END_RUNG
   RUNG wire#powerrail
      Contact( "AlwaysTRUE" )
      { S7_Templates := "SrcType := Int" } EQ_Contact(in1 := "MODE SELECTION DB"."MODE BUFF", in2 := 1)
      wire#w2
      Move(in := "HYST AND TEMP CUTOFF  DB"."AUTO SET"."PREMIXING LOAD CELL FOR TRANSFER", out1 => "HYST AND TEMP CUTOFF  DB"."MAIN SET PARA"."PREMIXING_LOAD CELL")
   END_RUNG
   RUNG wire#w2
      { S7_Templates := "SrcType := Int" } NE_Contact(in1 := "PREMIXING TRANSFER CYCLE DB".TRANSFER."TRANSFER BUFF"."PREMIXING TO MFG WITH INLINE HOMO", in2 := 5)
      { S7_Templates := "SrcType := Int" } NE_Contact(in1 := "PREMIXING TRANSFER CYCLE DB".TRANSFER."TRANSFER BUFF"."PREMIXING TO MFG WITH INLINE HOMO", in2 := 10)
      { S7_Templates := "SrcType := Int" } NE_Contact(in1 := "PREMIXING TRANSFER CYCLE DB".TRANSFER."TRANSFER BUFF"."PREMIXING TO MFG WITH INLINE FILTER PRES", in2 := 5)
      { S7_Templates := "SrcType := Int" } NE_Contact(in1 := "PREMIXING TRANSFER CYCLE DB".TRANSFER."TRANSFER BUFF"."PREMIXING TO MFG WITH INLINE FILTER PRES", in2 := 10)
      { S7_Templates := "SrcType := Int" } NE_Contact(in1 := "PREMIXING TRANSFER CYCLE DB".TRANSFER."TRANSFER BUFF"."PREMIXING TO STORAGE-4 WITH INLINE HOMO", in2 := 5)
      { S7_Templates := "SrcType := Int" } NE_Contact(in1 := "PREMIXING TRANSFER CYCLE DB".TRANSFER."TRANSFER BUFF"."PREMIXING TO STORAGE-4 WITH INLINE HOMO", in2 := 10)
      { S7_Templates := "SrcType := Int" } NE_Contact(in1 := "PREMIXING TRANSFER CYCLE DB".TRANSFER."TRANSFER BUFF"."PREMIXING TO STORAGE-4 WITH INLINE FILTER PRES", in2 := 5)
      { S7_Templates := "SrcType := Int" } NE_Contact(in1 := "PREMIXING TRANSFER CYCLE DB".TRANSFER."TRANSFER BUFF"."PREMIXING TO STORAGE-4 WITH INLINE FILTER PRES", in2 := 10)
      Move(in := "AI SCALING DB".PV."PREMIXING LOAD CELL", out1 => "HYST AND TEMP CUTOFF  DB"."MAN SET"."PREMIXING MOVE PV LOAD CELL")
   END_RUNG
   // the same network as SCL:
   #_w1 := "AlwaysTRUE" AND ("MODE SELECTION DB"."MODE BUFF" = 2);
   IF #_w1 THEN
       "HYST AND TEMP CUTOFF  DB"."MAIN SET PARA"."PREMIXING_LOAD CELL" := "HYST AND TEMP CUTOFF  DB"."MAN SET"."PREMIXING_LOAD CELL";
   END_IF;
   IF #_w1 AND ("MANUAL INTERLOCK DB"."PREMIXING TRANSFER PROCESS INTERLOCK" <> 1) THEN
       "HYST AND TEMP CUTOFF  DB"."MAN SET"."PREMIXING MOVE PV LOAD CELL" := "AI SCALING DB".PV."PREMIXING LOAD CELL";
   END_IF;
   #_w2 := "AlwaysTRUE" AND ("MODE SELECTION DB"."MODE BUFF" = 1);
   IF #_w2 THEN
       "HYST AND TEMP CUTOFF  DB"."MAIN SET PARA"."PREMIXING_LOAD CELL" := "HYST AND TEMP CUTOFF  DB"."AUTO SET"."PREMIXING LOAD CELL FOR TRANSFER";
   END_IF;
   IF #_w2 AND ("PREMIXING TRANSFER CYCLE DB".TRANSFER."TRANSFER BUFF"."PREMIXING TO MFG WITH INLINE HOMO" <> 5) AND ("PREMIXING TRANSFER CYCLE DB".TRANSFER."TRANSFER BUFF"."PREMIXING TO MFG WITH INLINE HOMO" <> 10) AND ("PREMIXING TRANSFER CYCLE DB".TRANSFER."TRANSFER BUFF"."PREMIXING TO MFG WITH INLINE FILTER PRES" <> 5) AND ("PREMIXING TRANSFER CYCLE DB".TRANSFER."TRANSFER BUFF"."PREMIXING TO MFG WITH INLINE FILTER PRES" <> 10) AND ("PREMIXING TRANSFER CYCLE DB".TRANSFER."TRANSFER BUFF"."PREMIXING TO STORAGE-4 WITH INLINE HOMO" <> 5) AND ("PREMIXING TRANSFER CYCLE DB".TRANSFER."TRANSFER BUFF"."PREMIXING TO STORAGE-4 WITH INLINE HOMO" <> 10) AND ("PREMIXING TRANSFER CYCLE DB".TRANSFER."TRANSFER BUFF"."PREMIXING TO STORAGE-4 WITH INLINE FILTER PRES" <> 5) AND ("PREMIXING TRANSFER CYCLE DB".TRANSFER."TRANSFER BUFF"."PREMIXING TO STORAGE-4 WITH INLINE FILTER PRES" <> 10) THEN
       "HYST AND TEMP CUTOFF  DB"."MAN SET"."PREMIXING MOVE PV LOAD CELL" := "AI SCALING DB".PV."PREMIXING LOAD CELL";
   END_IF;
END_REGION

REGION Network 35: TRANSFER SUB HYSTERISIS
   RUNG wire#powerrail
      Contact( "AlwaysTRUE" )
      wire#w1
      Sub(in1 := "HYST AND TEMP CUTOFF  DB"."MAN SET"."PREMIXING MOVE PV LOAD CELL", in2 := "HYST AND TEMP CUTOFF  DB"."MAIN SET PARA"."PREMIXING_LOAD CELL", out => "HYST AND TEMP CUTOFF  DB"."HYSTERISIS NEW_VALUE"."PREMIXING_LOAD CELL")
   END_RUNG
   RUNG wire#w1
      "@PREMIXING TRANSFER LOAD CALCULATE PV"("MODE SELECTION" := "MODE SELECTION DB"."MODE BUFF", "AUTO TRANSFER_1" := "PREMIXING TRANSFER CYCLE DB".TRANSFER."TRANSFER BUFF"."PREMIXING TO MFG WITH INLINE HOMO", "AUTO TRANSFER_2" := "PREMIXING TRANSFER CYCLE DB".TRANSFER."TRANSFER BUFF"."PREMIXING TO MFG WITH INLINE FILTER PRES", "AUTO TRANSFER_3" := "PREMIXING TRANSFER CYCLE DB".TRANSFER."TRANSFER BUFF"."PREMIXING TO STORAGE-4 WITH INLINE HOMO", "AUTO TRANSFER_4" := "PREMIXING TRANSFER CYCLE DB".TRANSFER."TRANSFER BUFF"."PREMIXING TO STORAGE-4 WITH INLINE FILTER PRES", "MOVE PV LOAD CELL" := "HYST AND TEMP CUTOFF  DB"."MAN SET"."PREMIXING MOVE PV LOAD CELL", "LOAD CELL PV" := "AI SCALING DB".PV."PREMIXING LOAD CELL", MANUAL => "HYST AND TEMP CUTOFF  DB"."PREMIXING CALCULATE PV", "PREMIXING TO MFG WITH INLINE HOMO" => "PREMIXING TRANSFER CYCLE DB"."PV PARAMETER"."PREMIXING TO MFG WITH INLINE HOMO", "PREMIXING TO MFG WITH INLINE FILTER PRES" => "PREMIXING TRANSFER CYCLE DB"."PV PARAMETER"."PREMIXING TO MFG WITH INLINE FILTER PRES", "PREMIXING TO STORAGE-4 WITH INLINE HOMO" => "PREMIXING TRANSFER CYCLE DB"."PV PARAMETER"."PREMIXING TO STORAGE-4 WITH INLINE HOMO", "PREMIXING TO STORAGE-4 WITH INLINE FILTER PRES" => "PREMIXING TRANSFER CYCLE DB"."PV PARAMETER"."PREMIXING TO STORAGE-4 WITH INLINE FILTER PRES")
   END_RUNG
   // the same network as SCL:
   IF "AlwaysTRUE" THEN
       "HYST AND TEMP CUTOFF  DB"."HYSTERISIS NEW_VALUE"."PREMIXING_LOAD CELL" := "HYST AND TEMP CUTOFF  DB"."MAN SET"."PREMIXING MOVE PV LOAD CELL" - "HYST AND TEMP CUTOFF  DB"."MAIN SET PARA"."PREMIXING_LOAD CELL";
       "@PREMIXING TRANSFER LOAD CALCULATE PV"("MODE SELECTION" := "MODE SELECTION DB"."MODE BUFF",
                               "AUTO TRANSFER_1" := "PREMIXING TRANSFER CYCLE DB".TRANSFER."TRANSFER BUFF"."PREMIXING TO MFG WITH INLINE HOMO",
                               "AUTO TRANSFER_2" := "PREMIXING TRANSFER CYCLE DB".TRANSFER."TRANSFER BUFF"."PREMIXING TO MFG WITH INLINE FILTER PRES",
                               "AUTO TRANSFER_3" := "PREMIXING TRANSFER CYCLE DB".TRANSFER."TRANSFER BUFF"."PREMIXING TO STORAGE-4 WITH INLINE HOMO",
                               "AUTO TRANSFER_4" := "PREMIXING TRANSFER CYCLE DB".TRANSFER."TRANSFER BUFF"."PREMIXING TO STORAGE-4 WITH INLINE FILTER PRES",
                               "MOVE PV LOAD CELL" := "HYST AND TEMP CUTOFF  DB"."MAN SET"."PREMIXING MOVE PV LOAD CELL",
                               "LOAD CELL PV" := "AI SCALING DB".PV."PREMIXING LOAD CELL",
                               MANUAL => "HYST AND TEMP CUTOFF  DB"."PREMIXING CALCULATE PV",
                               "PREMIXING TO MFG WITH INLINE HOMO" => "PREMIXING TRANSFER CYCLE DB"."PV PARAMETER"."PREMIXING TO MFG WITH INLINE HOMO",
                               "PREMIXING TO MFG WITH INLINE FILTER PRES" => "PREMIXING TRANSFER CYCLE DB"."PV PARAMETER"."PREMIXING TO MFG WITH INLINE FILTER PRES",
                               "PREMIXING TO STORAGE-4 WITH INLINE HOMO" => "PREMIXING TRANSFER CYCLE DB"."PV PARAMETER"."PREMIXING TO STORAGE-4 WITH INLINE HOMO",
                               "PREMIXING TO STORAGE-4 WITH INLINE FILTER PRES" => "PREMIXING TRANSFER CYCLE DB"."PV PARAMETER"."PREMIXING TO STORAGE-4 WITH INLINE FILTER PRES");
   END_IF;
END_REGION

REGION Network 36: TRANSFER TEMP CUT OFF
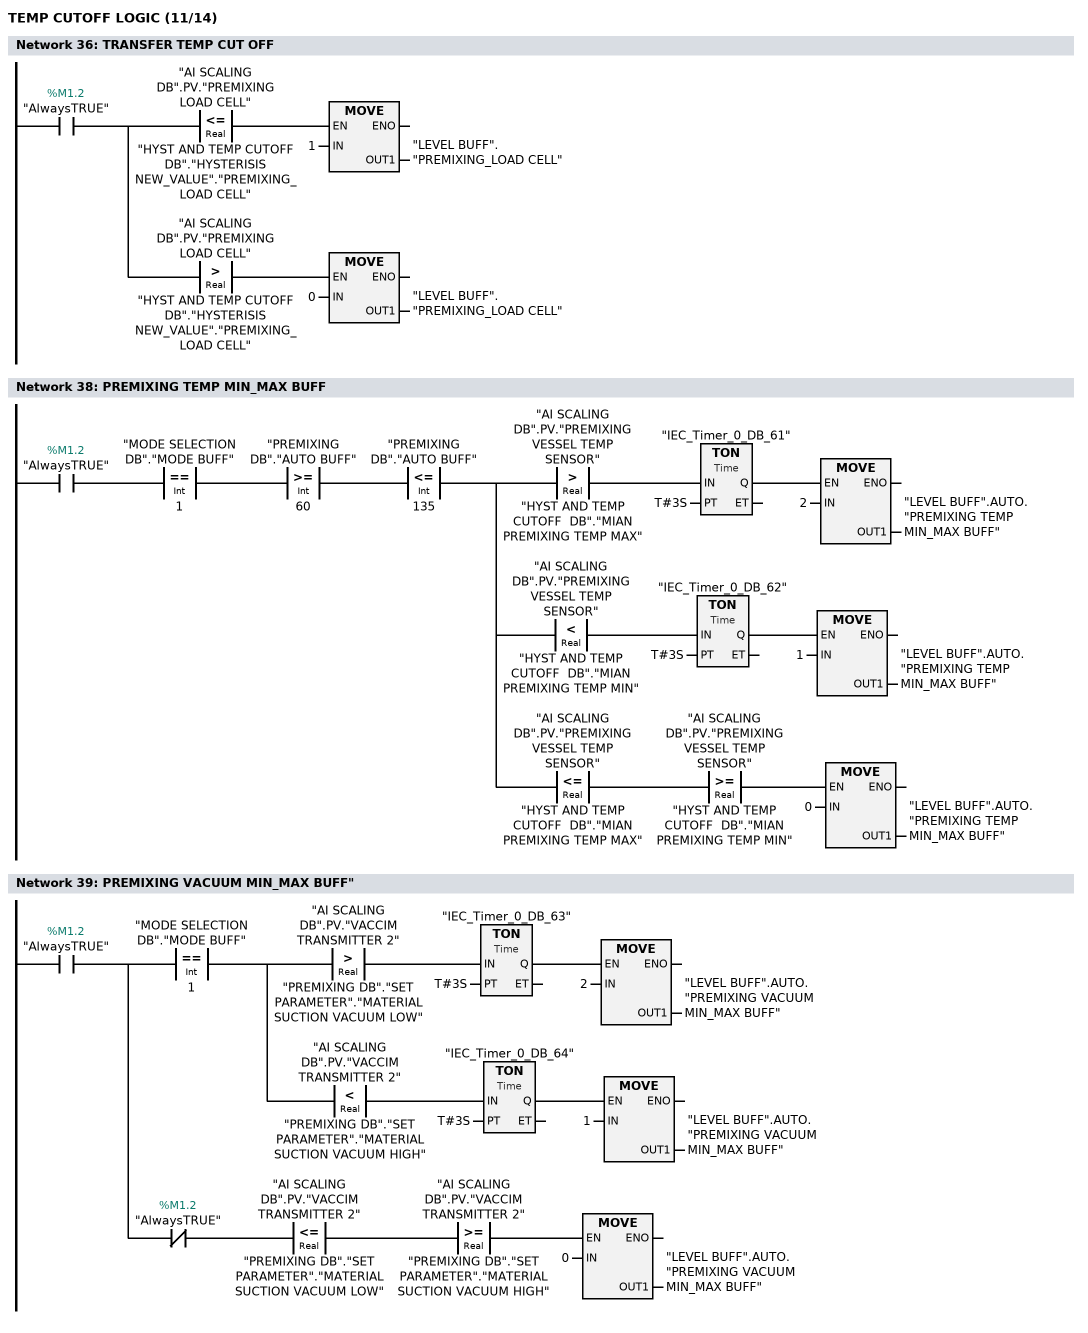
   RUNG wire#powerrail
      Contact( "AlwaysTRUE" )
      wire#w1
      { S7_Templates := "SrcType := Real" } LE_Contact(in1 := "AI SCALING DB".PV."PREMIXING LOAD CELL", in2 := "HYST AND TEMP CUTOFF  DB"."HYSTERISIS NEW_VALUE"."PREMIXING_LOAD CELL")
      Move(in := 1, out1 => "LEVEL BUFF"."PREMIXING_LOAD CELL")
   END_RUNG
   RUNG wire#w1
      { S7_Templates := "SrcType := Real" } GT_Contact(in1 := "AI SCALING DB".PV."PREMIXING LOAD CELL", in2 := "HYST AND TEMP CUTOFF  DB"."HYSTERISIS NEW_VALUE"."PREMIXING_LOAD CELL")
      Move(in := 0, out1 => "LEVEL BUFF"."PREMIXING_LOAD CELL")
   END_RUNG
   // the same network as SCL:
   IF "AlwaysTRUE" AND ("AI SCALING DB".PV."PREMIXING LOAD CELL" <= "HYST AND TEMP CUTOFF  DB"."HYSTERISIS NEW_VALUE"."PREMIXING_LOAD CELL") THEN
       "LEVEL BUFF"."PREMIXING_LOAD CELL" := 1;
   END_IF;
   IF "AlwaysTRUE" AND ("AI SCALING DB".PV."PREMIXING LOAD CELL" > "HYST AND TEMP CUTOFF  DB"."HYSTERISIS NEW_VALUE"."PREMIXING_LOAD CELL") THEN
       "LEVEL BUFF"."PREMIXING_LOAD CELL" := 0;
   END_IF;
END_REGION

REGION Network 38: PREMIXING TEMP MIN_MAX BUFF
   RUNG wire#powerrail
      Contact( "AlwaysTRUE" )
      { S7_Templates := "SrcType := Int" } EQ_Contact(in1 := "MODE SELECTION DB"."MODE BUFF", in2 := 1)
      { S7_Templates := "SrcType := Int" } GE_Contact(in1 := "PREMIXING DB"."AUTO BUFF", in2 := 60)
      { S7_Templates := "SrcType := Int" } LE_Contact(in1 := "PREMIXING DB"."AUTO BUFF", in2 := 135)
      wire#w1
      { S7_Templates := "SrcType := Real" } GT_Contact(in1 := "AI SCALING DB".PV."PREMIXING VESSEL TEMP SENSOR", in2 := "HYST AND TEMP CUTOFF  DB"."MIAN PREMIXING TEMP MAX")
      { S7_Templates := "time_type := Time" } "IEC_Timer_0_DB_61".TON(pt := T#3S, et =>)
      Move(in := 2, out1 => "LEVEL BUFF".AUTO."PREMIXING TEMP MIN_MAX BUFF")
   END_RUNG
   RUNG wire#w1
      { S7_Templates := "SrcType := Real" } LT_Contact(in1 := "AI SCALING DB".PV."PREMIXING VESSEL TEMP SENSOR", in2 := "HYST AND TEMP CUTOFF  DB"."MIAN PREMIXING TEMP MIN")
      { S7_Templates := "time_type := Time" } "IEC_Timer_0_DB_62".TON(pt := T#3S, et =>)
      Move(in := 1, out1 => "LEVEL BUFF".AUTO."PREMIXING TEMP MIN_MAX BUFF")
   END_RUNG
   RUNG wire#w1
      { S7_Templates := "SrcType := Real" } LE_Contact(in1 := "AI SCALING DB".PV."PREMIXING VESSEL TEMP SENSOR", in2 := "HYST AND TEMP CUTOFF  DB"."MIAN PREMIXING TEMP MAX")
      { S7_Templates := "SrcType := Real" } GE_Contact(in1 := "AI SCALING DB".PV."PREMIXING VESSEL TEMP SENSOR", in2 := "HYST AND TEMP CUTOFF  DB"."MIAN PREMIXING TEMP MIN")
      Move(in := 0, out1 => "LEVEL BUFF".AUTO."PREMIXING TEMP MIN_MAX BUFF")
   END_RUNG
   // the same network as SCL:
   #_w1 := "AlwaysTRUE" AND ("MODE SELECTION DB"."MODE BUFF" = 1) AND ("PREMIXING DB"."AUTO BUFF" >= 60) AND ("PREMIXING DB"."AUTO BUFF" <= 135);
   "IEC_Timer_0_DB_61".TON(IN := #_w1 AND ("AI SCALING DB".PV."PREMIXING VESSEL TEMP SENSOR" > "HYST AND TEMP CUTOFF  DB"."MIAN PREMIXING TEMP MAX"),
                           PT := T#3S);
   IF "IEC_Timer_0_DB_61".Q THEN "LEVEL BUFF".AUTO."PREMIXING TEMP MIN_MAX BUFF" := 2; END_IF;
   "IEC_Timer_0_DB_62".TON(IN := #_w1 AND ("AI SCALING DB".PV."PREMIXING VESSEL TEMP SENSOR" < "HYST AND TEMP CUTOFF  DB"."MIAN PREMIXING TEMP MIN"),
                           PT := T#3S);
   IF "IEC_Timer_0_DB_62".Q THEN "LEVEL BUFF".AUTO."PREMIXING TEMP MIN_MAX BUFF" := 1; END_IF;
   IF #_w1 AND ("AI SCALING DB".PV."PREMIXING VESSEL TEMP SENSOR" <= "HYST AND TEMP CUTOFF  DB"."MIAN PREMIXING TEMP MAX") AND ("AI SCALING DB".PV."PREMIXING VESSEL TEMP SENSOR" >= "HYST AND TEMP CUTOFF  DB"."MIAN PREMIXING TEMP MIN") THEN
       "LEVEL BUFF".AUTO."PREMIXING TEMP MIN_MAX BUFF" := 0;
   END_IF;
END_REGION

REGION Network 39: PREMIXING VACUUM MIN_MAX BUFF"
   RUNG wire#powerrail
      Contact( "AlwaysTRUE" )
      wire#w1
      { S7_Templates := "SrcType := Int" } EQ_Contact(in1 := "MODE SELECTION DB"."MODE BUFF", in2 := 1)
      wire#w2
      { S7_Templates := "SrcType := Real" } GT_Contact(in1 := "AI SCALING DB".PV."VACCIM TRANSMITTER 2", in2 := "PREMIXING DB"."SET PARAMETER"."MATERIAL SUCTION VACUUM LOW")
      { S7_Templates := "time_type := Time" } "IEC_Timer_0_DB_63".TON(pt := T#3S, et =>)
      Move(in := 2, out1 => "LEVEL BUFF".AUTO."PREMIXING VACUUM MIN_MAX BUFF")
   END_RUNG
   RUNG wire#w2
      { S7_Templates := "SrcType := Real" } LT_Contact(in1 := "AI SCALING DB".PV."VACCIM TRANSMITTER 2", in2 := "PREMIXING DB"."SET PARAMETER"."MATERIAL SUCTION VACUUM HIGH")
      { S7_Templates := "time_type := Time" } "IEC_Timer_0_DB_64".TON(pt := T#3S, et =>)
      Move(in := 1, out1 => "LEVEL BUFF".AUTO."PREMIXING VACUUM MIN_MAX BUFF")
   END_RUNG
   RUNG wire#w1
      I_Contact( "AlwaysTRUE" )
      { S7_Templates := "SrcType := Real" } LE_Contact(in1 := "AI SCALING DB".PV."VACCIM TRANSMITTER 2", in2 := "PREMIXING DB"."SET PARAMETER"."MATERIAL SUCTION VACUUM LOW")
      { S7_Templates := "SrcType := Real" } GE_Contact(in1 := "AI SCALING DB".PV."VACCIM TRANSMITTER 2", in2 := "PREMIXING DB"."SET PARAMETER"."MATERIAL SUCTION VACUUM HIGH")
      Move(in := 0, out1 => "LEVEL BUFF".AUTO."PREMIXING VACUUM MIN_MAX BUFF")
   END_RUNG
   // the same network as SCL:
   #_w1 := "AlwaysTRUE" AND ("MODE SELECTION DB"."MODE BUFF" = 1);
   "IEC_Timer_0_DB_63".TON(IN := #_w1 AND ("AI SCALING DB".PV."VACCIM TRANSMITTER 2" > "PREMIXING DB"."SET PARAMETER"."MATERIAL SUCTION VACUUM LOW"),
                           PT := T#3S);
   IF "IEC_Timer_0_DB_63".Q THEN "LEVEL BUFF".AUTO."PREMIXING VACUUM MIN_MAX BUFF" := 2; END_IF;
   "IEC_Timer_0_DB_64".TON(IN := #_w1 AND ("AI SCALING DB".PV."VACCIM TRANSMITTER 2" < "PREMIXING DB"."SET PARAMETER"."MATERIAL SUCTION VACUUM HIGH"),
                           PT := T#3S);
   IF "IEC_Timer_0_DB_64".Q THEN "LEVEL BUFF".AUTO."PREMIXING VACUUM MIN_MAX BUFF" := 1; END_IF;
   IF "AlwaysTRUE" AND NOT "AlwaysTRUE" AND ("AI SCALING DB".PV."VACCIM TRANSMITTER 2" <= "PREMIXING DB"."SET PARAMETER"."MATERIAL SUCTION VACUUM LOW") AND ("AI SCALING DB".PV."VACCIM TRANSMITTER 2" >= "PREMIXING DB"."SET PARAMETER"."MATERIAL SUCTION VACUUM HIGH") THEN
       "LEVEL BUFF".AUTO."PREMIXING VACUUM MIN_MAX BUFF" := 0;
   END_IF;
END_REGION

REGION Network 43: SUGAR TEMP. VALUE ///////////////////////////////////////////////////////////
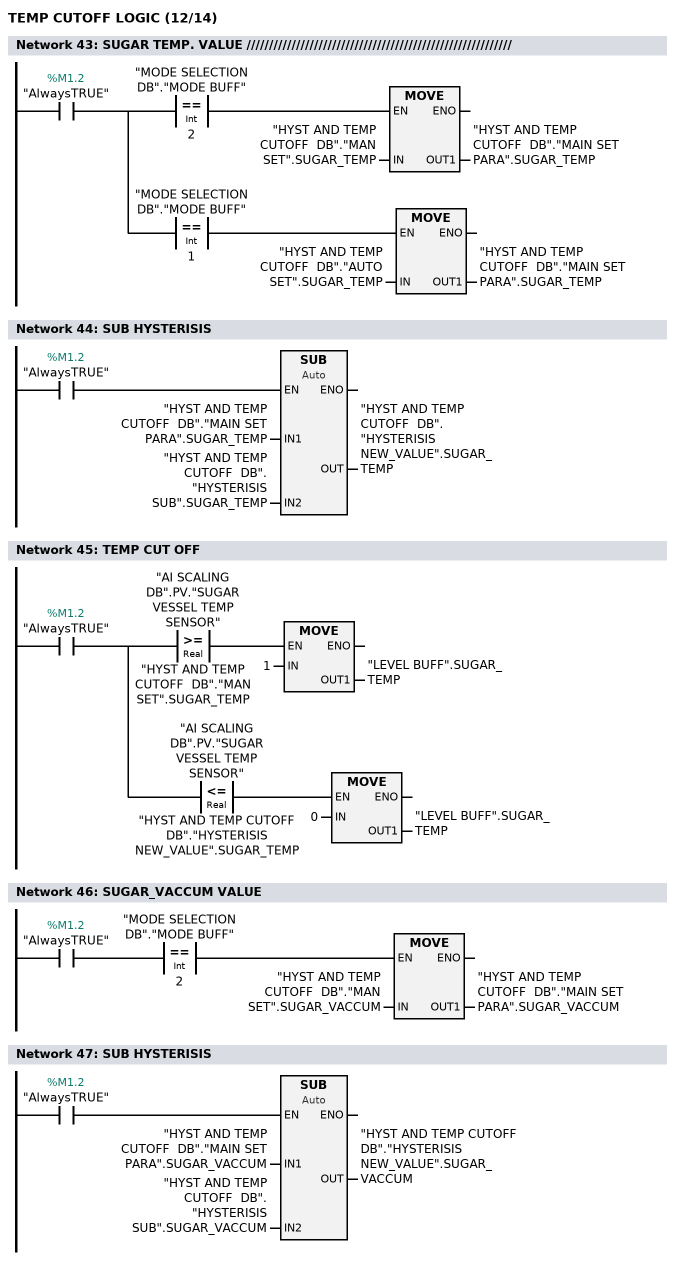
   RUNG wire#powerrail
      Contact( "AlwaysTRUE" )
      wire#w1
      { S7_Templates := "SrcType := Int" } EQ_Contact(in1 := "MODE SELECTION DB"."MODE BUFF", in2 := 2)
      Move(in := "HYST AND TEMP CUTOFF  DB"."MAN SET".SUGAR_TEMP, out1 => "HYST AND TEMP CUTOFF  DB"."MAIN SET PARA".SUGAR_TEMP)
   END_RUNG
   RUNG wire#w1
      { S7_Templates := "SrcType := Int" } EQ_Contact(in1 := "MODE SELECTION DB"."MODE BUFF", in2 := 1)
      Move(in := "HYST AND TEMP CUTOFF  DB"."AUTO SET".SUGAR_TEMP, out1 => "HYST AND TEMP CUTOFF  DB"."MAIN SET PARA".SUGAR_TEMP)
   END_RUNG
   // the same network as SCL:
   IF "AlwaysTRUE" AND ("MODE SELECTION DB"."MODE BUFF" = 2) THEN
       "HYST AND TEMP CUTOFF  DB"."MAIN SET PARA".SUGAR_TEMP := "HYST AND TEMP CUTOFF  DB"."MAN SET".SUGAR_TEMP;
   END_IF;
   IF "AlwaysTRUE" AND ("MODE SELECTION DB"."MODE BUFF" = 1) THEN
       "HYST AND TEMP CUTOFF  DB"."MAIN SET PARA".SUGAR_TEMP := "HYST AND TEMP CUTOFF  DB"."AUTO SET".SUGAR_TEMP;
   END_IF;
END_REGION

REGION Network 44: SUB HYSTERISIS
   RUNG wire#powerrail
      Contact( "AlwaysTRUE" )
      Sub(in1 := "HYST AND TEMP CUTOFF  DB"."MAIN SET PARA".SUGAR_TEMP, in2 := "HYST AND TEMP CUTOFF  DB"."HYSTERISIS SUB".SUGAR_TEMP, out => "HYST AND TEMP CUTOFF  DB"."HYSTERISIS NEW_VALUE".SUGAR_TEMP)
   END_RUNG
   // the same network as SCL:
   IF "AlwaysTRUE" THEN
       "HYST AND TEMP CUTOFF  DB"."HYSTERISIS NEW_VALUE".SUGAR_TEMP := "HYST AND TEMP CUTOFF  DB"."MAIN SET PARA".SUGAR_TEMP - "HYST AND TEMP CUTOFF  DB"."HYSTERISIS SUB".SUGAR_TEMP;
   END_IF;
END_REGION

REGION Network 45: TEMP CUT OFF
   RUNG wire#powerrail
      Contact( "AlwaysTRUE" )
      wire#w1
      { S7_Templates := "SrcType := Real" } GE_Contact(in1 := "AI SCALING DB".PV."SUGAR VESSEL TEMP SENSOR", in2 := "HYST AND TEMP CUTOFF  DB"."MAN SET".SUGAR_TEMP)
      Move(in := 1, out1 => "LEVEL BUFF".SUGAR_TEMP)
   END_RUNG
   RUNG wire#w1
      { S7_Templates := "SrcType := Real" } LE_Contact(in1 := "AI SCALING DB".PV."SUGAR VESSEL TEMP SENSOR", in2 := "HYST AND TEMP CUTOFF  DB"."HYSTERISIS NEW_VALUE".SUGAR_TEMP)
      Move(in := 0, out1 => "LEVEL BUFF".SUGAR_TEMP)
   END_RUNG
   // the same network as SCL:
   IF "AlwaysTRUE" AND ("AI SCALING DB".PV."SUGAR VESSEL TEMP SENSOR" >= "HYST AND TEMP CUTOFF  DB"."MAN SET".SUGAR_TEMP) THEN
       "LEVEL BUFF".SUGAR_TEMP := 1;
   END_IF;
   IF "AlwaysTRUE" AND ("AI SCALING DB".PV."SUGAR VESSEL TEMP SENSOR" <= "HYST AND TEMP CUTOFF  DB"."HYSTERISIS NEW_VALUE".SUGAR_TEMP) THEN
       "LEVEL BUFF".SUGAR_TEMP := 0;
   END_IF;
END_REGION

REGION Network 46: SUGAR_VACCUM VALUE
   RUNG wire#powerrail
      Contact( "AlwaysTRUE" )
      { S7_Templates := "SrcType := Int" } EQ_Contact(in1 := "MODE SELECTION DB"."MODE BUFF", in2 := 2)
      Move(in := "HYST AND TEMP CUTOFF  DB"."MAN SET".SUGAR_VACCUM, out1 => "HYST AND TEMP CUTOFF  DB"."MAIN SET PARA".SUGAR_VACCUM)
   END_RUNG
   // the same network as SCL:
   IF "AlwaysTRUE" AND ("MODE SELECTION DB"."MODE BUFF" = 2) THEN
       "HYST AND TEMP CUTOFF  DB"."MAIN SET PARA".SUGAR_VACCUM := "HYST AND TEMP CUTOFF  DB"."MAN SET".SUGAR_VACCUM;
   END_IF;
END_REGION

REGION Network 47: SUB HYSTERISIS
   RUNG wire#powerrail
      Contact( "AlwaysTRUE" )
      Sub(in1 := "HYST AND TEMP CUTOFF  DB"."MAIN SET PARA".SUGAR_VACCUM, in2 := "HYST AND TEMP CUTOFF  DB"."HYSTERISIS SUB".SUGAR_VACCUM, out => "HYST AND TEMP CUTOFF  DB"."HYSTERISIS NEW_VALUE".SUGAR_VACCUM)
   END_RUNG
   // the same network as SCL:
   IF "AlwaysTRUE" THEN
       "HYST AND TEMP CUTOFF  DB"."HYSTERISIS NEW_VALUE".SUGAR_VACCUM := "HYST AND TEMP CUTOFF  DB"."MAIN SET PARA".SUGAR_VACCUM - "HYST AND TEMP CUTOFF  DB"."HYSTERISIS SUB".SUGAR_VACCUM;
   END_IF;
END_REGION

REGION Network 48: VACCUM CUT OFF
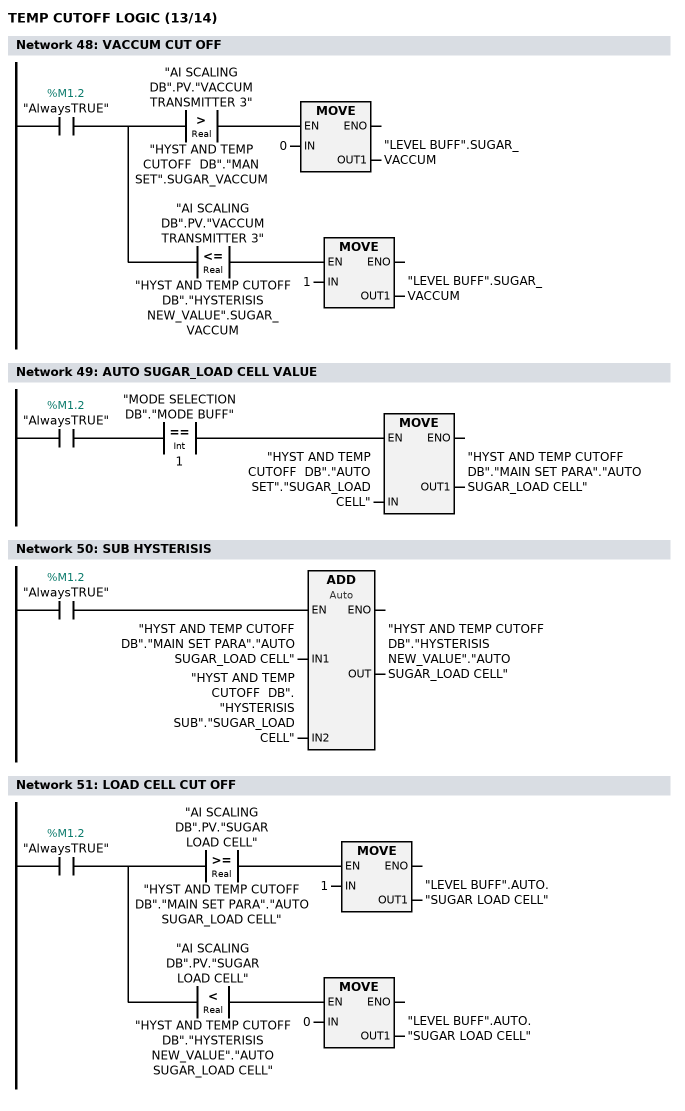
   RUNG wire#powerrail
      Contact( "AlwaysTRUE" )
      wire#w1
      { S7_Templates := "SrcType := Real" } GT_Contact(in1 := "AI SCALING DB".PV."VACCUM TRANSMITTER 3", in2 := "HYST AND TEMP CUTOFF  DB"."MAN SET".SUGAR_VACCUM)
      Move(in := 0, out1 => "LEVEL BUFF".SUGAR_VACCUM)
   END_RUNG
   RUNG wire#w1
      { S7_Templates := "SrcType := Real" } LE_Contact(in1 := "AI SCALING DB".PV."VACCUM TRANSMITTER 3", in2 := "HYST AND TEMP CUTOFF  DB"."HYSTERISIS NEW_VALUE".SUGAR_VACCUM)
      Move(in := 1, out1 => "LEVEL BUFF".SUGAR_VACCUM)
   END_RUNG
   // the same network as SCL:
   IF "AlwaysTRUE" AND ("AI SCALING DB".PV."VACCUM TRANSMITTER 3" > "HYST AND TEMP CUTOFF  DB"."MAN SET".SUGAR_VACCUM) THEN
       "LEVEL BUFF".SUGAR_VACCUM := 0;
   END_IF;
   IF "AlwaysTRUE" AND ("AI SCALING DB".PV."VACCUM TRANSMITTER 3" <= "HYST AND TEMP CUTOFF  DB"."HYSTERISIS NEW_VALUE".SUGAR_VACCUM) THEN
       "LEVEL BUFF".SUGAR_VACCUM := 1;
   END_IF;
END_REGION

REGION Network 49: AUTO SUGAR_LOAD CELL VALUE
   RUNG wire#powerrail
      Contact( "AlwaysTRUE" )
      { S7_Templates := "SrcType := Int" } EQ_Contact(in1 := "MODE SELECTION DB"."MODE BUFF", in2 := 1)
      Move(in := "HYST AND TEMP CUTOFF  DB"."AUTO SET"."SUGAR_LOAD CELL", out1 => "HYST AND TEMP CUTOFF  DB"."MAIN SET PARA"."AUTO SUGAR_LOAD CELL")
   END_RUNG
   // the same network as SCL:
   IF "AlwaysTRUE" AND ("MODE SELECTION DB"."MODE BUFF" = 1) THEN
       "HYST AND TEMP CUTOFF  DB"."MAIN SET PARA"."AUTO SUGAR_LOAD CELL" := "HYST AND TEMP CUTOFF  DB"."AUTO SET"."SUGAR_LOAD CELL";
   END_IF;
END_REGION

REGION Network 50: SUB HYSTERISIS
   RUNG wire#powerrail
      Contact( "AlwaysTRUE" )
      Add(in1 := "HYST AND TEMP CUTOFF  DB"."MAIN SET PARA"."AUTO SUGAR_LOAD CELL", in2 := "HYST AND TEMP CUTOFF  DB"."HYSTERISIS SUB"."SUGAR_LOAD CELL", out => "HYST AND TEMP CUTOFF  DB"."HYSTERISIS NEW_VALUE"."AUTO SUGAR_LOAD CELL")
   END_RUNG
   // the same network as SCL:
   IF "AlwaysTRUE" THEN
       "HYST AND TEMP CUTOFF  DB"."HYSTERISIS NEW_VALUE"."AUTO SUGAR_LOAD CELL" := "HYST AND TEMP CUTOFF  DB"."MAIN SET PARA"."AUTO SUGAR_LOAD CELL" + "HYST AND TEMP CUTOFF  DB"."HYSTERISIS SUB"."SUGAR_LOAD CELL";
   END_IF;
END_REGION

REGION Network 51: LOAD CELL CUT OFF
   RUNG wire#powerrail
      Contact( "AlwaysTRUE" )
      wire#w1
      { S7_Templates := "SrcType := Real" } GE_Contact(in1 := "AI SCALING DB".PV."SUGAR LOAD CELL", in2 := "HYST AND TEMP CUTOFF  DB"."MAIN SET PARA"."AUTO SUGAR_LOAD CELL")
      Move(in := 1, out1 => "LEVEL BUFF".AUTO."SUGAR LOAD CELL")
   END_RUNG
   RUNG wire#w1
      { S7_Templates := "SrcType := Real" } LT_Contact(in1 := "AI SCALING DB".PV."SUGAR LOAD CELL", in2 := "HYST AND TEMP CUTOFF  DB"."HYSTERISIS NEW_VALUE"."AUTO SUGAR_LOAD CELL")
      Move(in := 0, out1 => "LEVEL BUFF".AUTO."SUGAR LOAD CELL")
   END_RUNG
   // the same network as SCL:
   IF "AlwaysTRUE" AND ("AI SCALING DB".PV."SUGAR LOAD CELL" >= "HYST AND TEMP CUTOFF  DB"."MAIN SET PARA"."AUTO SUGAR_LOAD CELL") THEN
       "LEVEL BUFF".AUTO."SUGAR LOAD CELL" := 1;
   END_IF;
   IF "AlwaysTRUE" AND ("AI SCALING DB".PV."SUGAR LOAD CELL" < "HYST AND TEMP CUTOFF  DB"."HYSTERISIS NEW_VALUE"."AUTO SUGAR_LOAD CELL") THEN
       "LEVEL BUFF".AUTO."SUGAR LOAD CELL" := 0;
   END_IF;
END_REGION

REGION Network 53: SUGAR_LOAD CELL VALUE ONLY TRANSFER
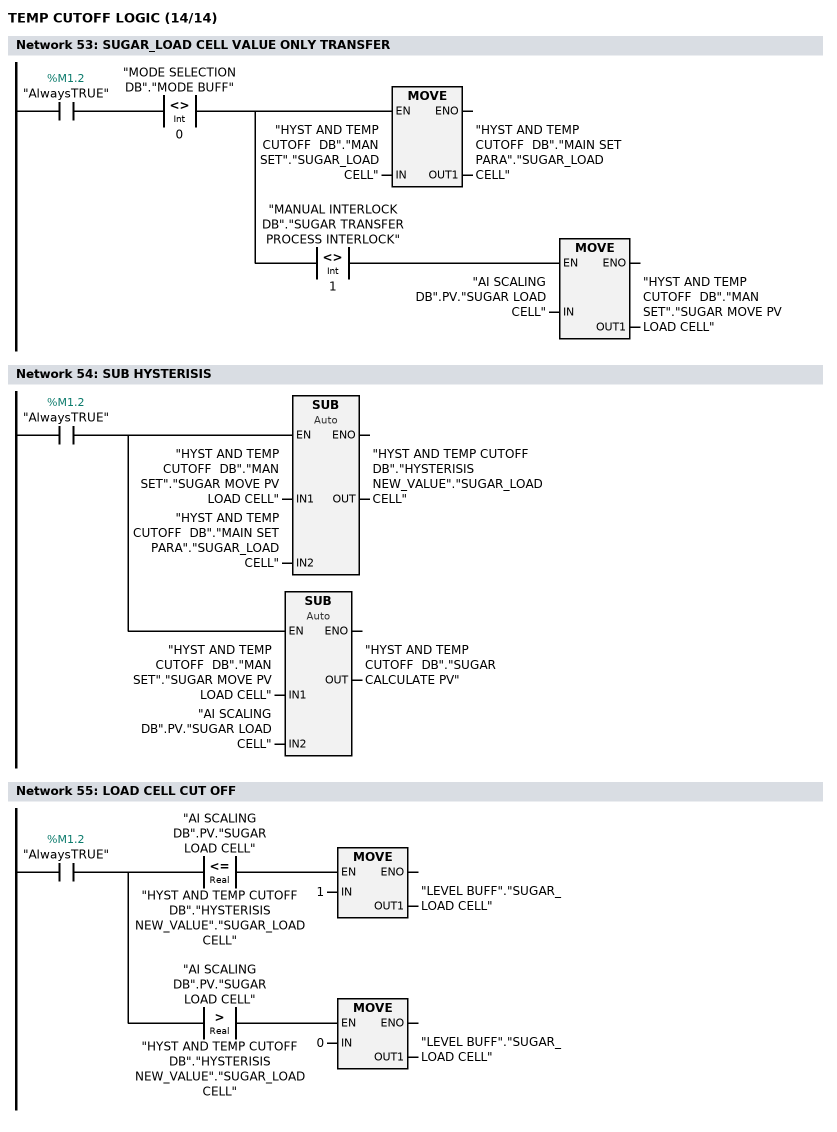
   RUNG wire#powerrail
      Contact( "AlwaysTRUE" )
      { S7_Templates := "SrcType := Int" } NE_Contact(in1 := "MODE SELECTION DB"."MODE BUFF", in2 := 0)
      wire#w1
      Move(in := "HYST AND TEMP CUTOFF  DB"."MAN SET"."SUGAR_LOAD CELL", out1 => "HYST AND TEMP CUTOFF  DB"."MAIN SET PARA"."SUGAR_LOAD CELL")
   END_RUNG
   RUNG wire#w1
      { S7_Templates := "SrcType := Int" } NE_Contact(in1 := "MANUAL INTERLOCK DB"."SUGAR TRANSFER PROCESS INTERLOCK", in2 := 1)
      Move(in := "AI SCALING DB".PV."SUGAR LOAD CELL", out1 => "HYST AND TEMP CUTOFF  DB"."MAN SET"."SUGAR MOVE PV LOAD CELL")
   END_RUNG
   // the same network as SCL:
   #_w1 := "AlwaysTRUE" AND ("MODE SELECTION DB"."MODE BUFF" <> 0);
   IF #_w1 THEN
       "HYST AND TEMP CUTOFF  DB"."MAIN SET PARA"."SUGAR_LOAD CELL" := "HYST AND TEMP CUTOFF  DB"."MAN SET"."SUGAR_LOAD CELL";
   END_IF;
   IF #_w1 AND ("MANUAL INTERLOCK DB"."SUGAR TRANSFER PROCESS INTERLOCK" <> 1) THEN
       "HYST AND TEMP CUTOFF  DB"."MAN SET"."SUGAR MOVE PV LOAD CELL" := "AI SCALING DB".PV."SUGAR LOAD CELL";
   END_IF;
END_REGION

REGION Network 54: SUB HYSTERISIS
   RUNG wire#powerrail
      Contact( "AlwaysTRUE" )
      wire#w1
      Sub(in1 := "HYST AND TEMP CUTOFF  DB"."MAN SET"."SUGAR MOVE PV LOAD CELL", in2 := "HYST AND TEMP CUTOFF  DB"."MAIN SET PARA"."SUGAR_LOAD CELL", out => "HYST AND TEMP CUTOFF  DB"."HYSTERISIS NEW_VALUE"."SUGAR_LOAD CELL")
   END_RUNG
   RUNG wire#w1
      Sub(in1 := "HYST AND TEMP CUTOFF  DB"."MAN SET"."SUGAR MOVE PV LOAD CELL", in2 := "AI SCALING DB".PV."SUGAR LOAD CELL", out => "HYST AND TEMP CUTOFF  DB"."SUGAR CALCULATE PV")
   END_RUNG
   // the same network as SCL:
   IF "AlwaysTRUE" THEN
       "HYST AND TEMP CUTOFF  DB"."HYSTERISIS NEW_VALUE"."SUGAR_LOAD CELL" := "HYST AND TEMP CUTOFF  DB"."MAN SET"."SUGAR MOVE PV LOAD CELL" - "HYST AND TEMP CUTOFF  DB"."MAIN SET PARA"."SUGAR_LOAD CELL";
       "HYST AND TEMP CUTOFF  DB"."SUGAR CALCULATE PV" := "HYST AND TEMP CUTOFF  DB"."MAN SET"."SUGAR MOVE PV LOAD CELL" - "AI SCALING DB".PV."SUGAR LOAD CELL";
   END_IF;
END_REGION

REGION Network 55: LOAD CELL CUT OFF
   RUNG wire#powerrail
      Contact( "AlwaysTRUE" )
      wire#w1
      { S7_Templates := "SrcType := Real" } LE_Contact(in1 := "AI SCALING DB".PV."SUGAR LOAD CELL", in2 := "HYST AND TEMP CUTOFF  DB"."HYSTERISIS NEW_VALUE"."SUGAR_LOAD CELL")
      Move(in := 1, out1 => "LEVEL BUFF"."SUGAR_LOAD CELL")
   END_RUNG
   RUNG wire#w1
      { S7_Templates := "SrcType := Real" } GT_Contact(in1 := "AI SCALING DB".PV."SUGAR LOAD CELL", in2 := "HYST AND TEMP CUTOFF  DB"."HYSTERISIS NEW_VALUE"."SUGAR_LOAD CELL")
      Move(in := 0, out1 => "LEVEL BUFF"."SUGAR_LOAD CELL")
   END_RUNG
   // the same network as SCL:
   IF "AlwaysTRUE" AND ("AI SCALING DB".PV."SUGAR LOAD CELL" <= "HYST AND TEMP CUTOFF  DB"."HYSTERISIS NEW_VALUE"."SUGAR_LOAD CELL") THEN
       "LEVEL BUFF"."SUGAR_LOAD CELL" := 1;
   END_IF;
   IF "AlwaysTRUE" AND ("AI SCALING DB".PV."SUGAR LOAD CELL" > "HYST AND TEMP CUTOFF  DB"."HYSTERISIS NEW_VALUE"."SUGAR_LOAD CELL") THEN
       "LEVEL BUFF"."SUGAR_LOAD CELL" := 0;
   END_IF;
END_REGION
END_FUNCTION

FUNCTION "@LOAD CALCULATE" : Void   // FC20, LAD
{ S7_Optimized_Access := 'TRUE' }
// stored: SetENOAutomatically false
   VAR_INPUT
      "MFG PROCESS BUFF" : Int;
      "MATERIAL SUCTION BUFF" : Int;
      "MOVE PV" : Real;
      PV : Real;
   END_VAR
   VAR_OUTPUT
      "PURIFIED CALCULATE PV" : Real;
      "MATERIAL SORBITOL CALCULATE PV" : Real;
      "MATERIAL GLUCOSE CALCULATE PV" : Real;
      "MATERIAL SUCTION CALCULATE PV" : Real;
   END_VAR
BEGIN

REGION Network 1
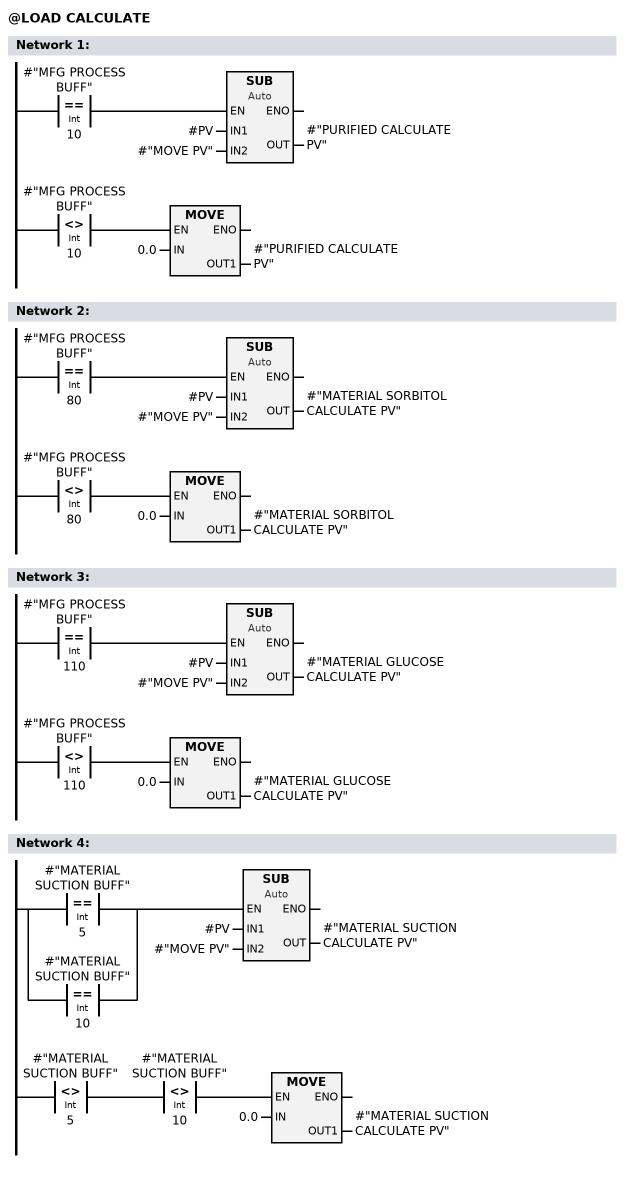
   RUNG wire#powerrail
      { S7_Templates := "SrcType := Int" } EQ_Contact(in1 := #"MFG PROCESS BUFF", in2 := 10)
      Sub(in1 := #PV, in2 := #"MOVE PV", out => #"PURIFIED CALCULATE PV")
   END_RUNG
   RUNG wire#powerrail
      { S7_Templates := "SrcType := Int" } NE_Contact(in1 := #"MFG PROCESS BUFF", in2 := 10)
      Move(in := 0.0, out1 => #"PURIFIED CALCULATE PV")
   END_RUNG
   // the same network as SCL:
   IF #"MFG PROCESS BUFF" = 10 THEN #"PURIFIED CALCULATE PV" := #PV - #"MOVE PV"; END_IF;
   IF #"MFG PROCESS BUFF" <> 10 THEN #"PURIFIED CALCULATE PV" := 0.0; END_IF;
END_REGION

REGION Network 2
   RUNG wire#powerrail
      { S7_Templates := "SrcType := Int" } EQ_Contact(in1 := #"MFG PROCESS BUFF", in2 := 80)
      Sub(in1 := #PV, in2 := #"MOVE PV", out => #"MATERIAL SORBITOL CALCULATE PV")
   END_RUNG
   RUNG wire#powerrail
      { S7_Templates := "SrcType := Int" } NE_Contact(in1 := #"MFG PROCESS BUFF", in2 := 80)
      Move(in := 0.0, out1 => #"MATERIAL SORBITOL CALCULATE PV")
   END_RUNG
   // the same network as SCL:
   IF #"MFG PROCESS BUFF" = 80 THEN #"MATERIAL SORBITOL CALCULATE PV" := #PV - #"MOVE PV"; END_IF;
   IF #"MFG PROCESS BUFF" <> 80 THEN #"MATERIAL SORBITOL CALCULATE PV" := 0.0; END_IF;
END_REGION

REGION Network 3
   RUNG wire#powerrail
      { S7_Templates := "SrcType := Int" } EQ_Contact(in1 := #"MFG PROCESS BUFF", in2 := 110)
      Sub(in1 := #PV, in2 := #"MOVE PV", out => #"MATERIAL GLUCOSE CALCULATE PV")
   END_RUNG
   RUNG wire#powerrail
      { S7_Templates := "SrcType := Int" } NE_Contact(in1 := #"MFG PROCESS BUFF", in2 := 110)
      Move(in := 0.0, out1 => #"MATERIAL GLUCOSE CALCULATE PV")
   END_RUNG
   // the same network as SCL:
   IF #"MFG PROCESS BUFF" = 110 THEN #"MATERIAL GLUCOSE CALCULATE PV" := #PV - #"MOVE PV"; END_IF;
   IF #"MFG PROCESS BUFF" <> 110 THEN #"MATERIAL GLUCOSE CALCULATE PV" := 0.0; END_IF;
END_REGION

REGION Network 4
   RUNG wire#powerrail
      { S7_Templates := "SrcType := Int" } EQ_Contact(in1 := #"MATERIAL SUCTION BUFF", in2 := 5)
      wire#w1
      Sub(in1 := #PV, in2 := #"MOVE PV", out => #"MATERIAL SUCTION CALCULATE PV")
   END_RUNG
   RUNG wire#powerrail
      { S7_Templates := "SrcType := Int" } EQ_Contact(in1 := #"MATERIAL SUCTION BUFF", in2 := 10)
   END_RUNG wire#w1
   RUNG wire#powerrail
      { S7_Templates := "SrcType := Int" } NE_Contact(in1 := #"MATERIAL SUCTION BUFF", in2 := 5)
      { S7_Templates := "SrcType := Int" } NE_Contact(in1 := #"MATERIAL SUCTION BUFF", in2 := 10)
      Move(in := 0.0, out1 => #"MATERIAL SUCTION CALCULATE PV")
   END_RUNG
   // the same network as SCL:
   IF (#"MATERIAL SUCTION BUFF" = 5) OR (#"MATERIAL SUCTION BUFF" = 10) THEN
       #"MATERIAL SUCTION CALCULATE PV" := #PV - #"MOVE PV";
   END_IF;
   IF (#"MATERIAL SUCTION BUFF" <> 5) AND (#"MATERIAL SUCTION BUFF" <> 10) THEN
       #"MATERIAL SUCTION CALCULATE PV" := 0.0;
   END_IF;
END_REGION
END_FUNCTION

FUNCTION "SET PARAMETER" : Void   // FC18, LAD
{ S7_Optimized_Access := 'TRUE' }
// stored: SetENOAutomatically false
   VAR_TEMP   // added for the SCL form of the ladder/FBD networks
      _w1 : Bool;
   END_VAR
BEGIN

REGION Network 1: MFG STIRRER MOTOR
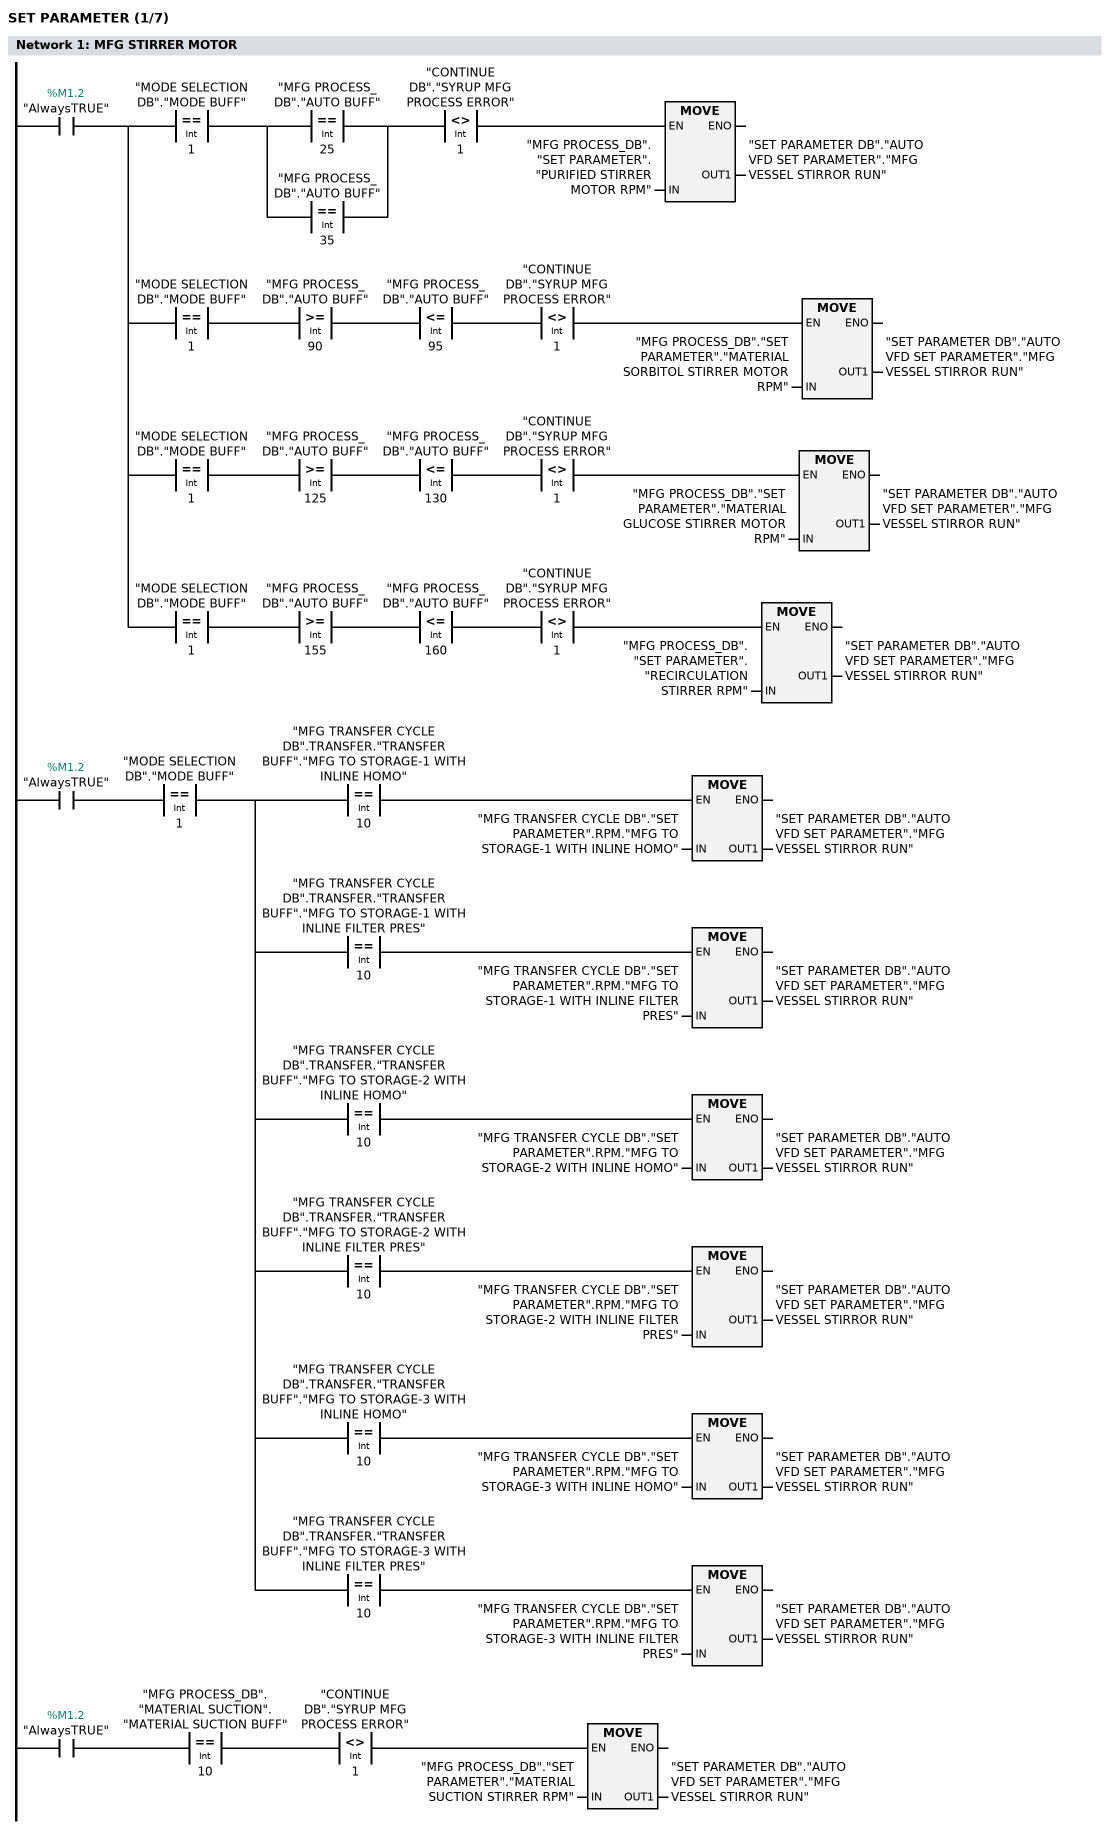
   RUNG wire#powerrail
      Contact( "AlwaysTRUE" )
      wire#w1
      { S7_Templates := "SrcType := Int" } EQ_Contact(in1 := "MODE SELECTION DB"."MODE BUFF", in2 := 1)
      wire#w2
      { S7_Templates := "SrcType := Int" } EQ_Contact(in1 := "MFG PROCESS_DB"."AUTO BUFF", in2 := 25)
      wire#w3
      { S7_Templates := "SrcType := Int" } NE_Contact(in1 := "CONTINUE DB"."SYRUP MFG PROCESS ERROR", in2 := 1)
      Move(in := "MFG PROCESS_DB"."SET PARAMETER"."PURIFIED STIRRER MOTOR RPM", out1 => "SET PARAMETER DB"."AUTO VFD SET PARAMETER"."MFG VESSEL STIRROR RUN")
   END_RUNG
   RUNG wire#w2
      { S7_Templates := "SrcType := Int" } EQ_Contact(in1 := "MFG PROCESS_DB"."AUTO BUFF", in2 := 35)
   END_RUNG wire#w3
   RUNG wire#w1
      { S7_Templates := "SrcType := Int" } EQ_Contact(in1 := "MODE SELECTION DB"."MODE BUFF", in2 := 1)
      { S7_Templates := "SrcType := Int" } GE_Contact(in1 := "MFG PROCESS_DB"."AUTO BUFF", in2 := 90)
      { S7_Templates := "SrcType := Int" } LE_Contact(in1 := "MFG PROCESS_DB"."AUTO BUFF", in2 := 95)
      { S7_Templates := "SrcType := Int" } NE_Contact(in1 := "CONTINUE DB"."SYRUP MFG PROCESS ERROR", in2 := 1)
      Move(in := "MFG PROCESS_DB"."SET PARAMETER"."MATERIAL SORBITOL STIRRER MOTOR RPM", out1 => "SET PARAMETER DB"."AUTO VFD SET PARAMETER"."MFG VESSEL STIRROR RUN")
   END_RUNG
   RUNG wire#w1
      { S7_Templates := "SrcType := Int" } EQ_Contact(in1 := "MODE SELECTION DB"."MODE BUFF", in2 := 1)
      { S7_Templates := "SrcType := Int" } GE_Contact(in1 := "MFG PROCESS_DB"."AUTO BUFF", in2 := 125)
      { S7_Templates := "SrcType := Int" } LE_Contact(in1 := "MFG PROCESS_DB"."AUTO BUFF", in2 := 130)
      { S7_Templates := "SrcType := Int" } NE_Contact(in1 := "CONTINUE DB"."SYRUP MFG PROCESS ERROR", in2 := 1)
      Move(in := "MFG PROCESS_DB"."SET PARAMETER"."MATERIAL GLUCOSE STIRRER MOTOR RPM", out1 => "SET PARAMETER DB"."AUTO VFD SET PARAMETER"."MFG VESSEL STIRROR RUN")
   END_RUNG
   RUNG wire#w1
      { S7_Templates := "SrcType := Int" } EQ_Contact(in1 := "MODE SELECTION DB"."MODE BUFF", in2 := 1)
      { S7_Templates := "SrcType := Int" } GE_Contact(in1 := "MFG PROCESS_DB"."AUTO BUFF", in2 := 155)
      { S7_Templates := "SrcType := Int" } LE_Contact(in1 := "MFG PROCESS_DB"."AUTO BUFF", in2 := 160)
      { S7_Templates := "SrcType := Int" } NE_Contact(in1 := "CONTINUE DB"."SYRUP MFG PROCESS ERROR", in2 := 1)
      Move(in := "MFG PROCESS_DB"."SET PARAMETER"."RECIRCULATION STIRRER RPM", out1 => "SET PARAMETER DB"."AUTO VFD SET PARAMETER"."MFG VESSEL STIRROR RUN")
   END_RUNG
   RUNG wire#powerrail
      Contact( "AlwaysTRUE" )
      { S7_Templates := "SrcType := Int" } EQ_Contact(in1 := "MODE SELECTION DB"."MODE BUFF", in2 := 1)
      wire#w4
      { S7_Templates := "SrcType := Int" } EQ_Contact(in1 := "MFG TRANSFER CYCLE DB".TRANSFER."TRANSFER BUFF"."MFG TO STORAGE-1 WITH INLINE HOMO", in2 := 10)
      Move(in := "MFG TRANSFER CYCLE DB"."SET PARAMETER".RPM."MFG TO STORAGE-1 WITH INLINE HOMO", out1 => "SET PARAMETER DB"."AUTO VFD SET PARAMETER"."MFG VESSEL STIRROR RUN")
   END_RUNG
   RUNG wire#w4
      { S7_Templates := "SrcType := Int" } EQ_Contact(in1 := "MFG TRANSFER CYCLE DB".TRANSFER."TRANSFER BUFF"."MFG TO STORAGE-1 WITH INLINE FILTER PRES", in2 := 10)
      Move(in := "MFG TRANSFER CYCLE DB"."SET PARAMETER".RPM."MFG TO STORAGE-1 WITH INLINE FILTER PRES", out1 => "SET PARAMETER DB"."AUTO VFD SET PARAMETER"."MFG VESSEL STIRROR RUN")
   END_RUNG
   RUNG wire#w4
      { S7_Templates := "SrcType := Int" } EQ_Contact(in1 := "MFG TRANSFER CYCLE DB".TRANSFER."TRANSFER BUFF"."MFG TO STORAGE-2 WITH INLINE HOMO", in2 := 10)
      Move(in := "MFG TRANSFER CYCLE DB"."SET PARAMETER".RPM."MFG TO STORAGE-2 WITH INLINE HOMO", out1 => "SET PARAMETER DB"."AUTO VFD SET PARAMETER"."MFG VESSEL STIRROR RUN")
   END_RUNG
   RUNG wire#w4
      { S7_Templates := "SrcType := Int" } EQ_Contact(in1 := "MFG TRANSFER CYCLE DB".TRANSFER."TRANSFER BUFF"."MFG TO STORAGE-2 WITH INLINE FILTER PRES", in2 := 10)
      Move(in := "MFG TRANSFER CYCLE DB"."SET PARAMETER".RPM."MFG TO STORAGE-2 WITH INLINE FILTER PRES", out1 => "SET PARAMETER DB"."AUTO VFD SET PARAMETER"."MFG VESSEL STIRROR RUN")
   END_RUNG
   RUNG wire#w4
      { S7_Templates := "SrcType := Int" } EQ_Contact(in1 := "MFG TRANSFER CYCLE DB".TRANSFER."TRANSFER BUFF"."MFG TO STORAGE-3 WITH INLINE HOMO", in2 := 10)
      Move(in := "MFG TRANSFER CYCLE DB"."SET PARAMETER".RPM."MFG TO STORAGE-3 WITH INLINE HOMO", out1 => "SET PARAMETER DB"."AUTO VFD SET PARAMETER"."MFG VESSEL STIRROR RUN")
   END_RUNG
   RUNG wire#w4
      { S7_Templates := "SrcType := Int" } EQ_Contact(in1 := "MFG TRANSFER CYCLE DB".TRANSFER."TRANSFER BUFF"."MFG TO STORAGE-3 WITH INLINE FILTER PRES", in2 := 10)
      Move(in := "MFG TRANSFER CYCLE DB"."SET PARAMETER".RPM."MFG TO STORAGE-3 WITH INLINE FILTER PRES", out1 => "SET PARAMETER DB"."AUTO VFD SET PARAMETER"."MFG VESSEL STIRROR RUN")
   END_RUNG
   RUNG wire#powerrail
      Contact( "AlwaysTRUE" )
      { S7_Templates := "SrcType := Int" } EQ_Contact(in1 := "MFG PROCESS_DB"."MATERIAL SUCTION"."MATERIAL SUCTION BUFF", in2 := 10)
      { S7_Templates := "SrcType := Int" } NE_Contact(in1 := "CONTINUE DB"."SYRUP MFG PROCESS ERROR", in2 := 1)
      Move(in := "MFG PROCESS_DB"."SET PARAMETER"."MATERIAL SUCTION STIRRER RPM", out1 => "SET PARAMETER DB"."AUTO VFD SET PARAMETER"."MFG VESSEL STIRROR RUN")
   END_RUNG
   // the same network as SCL:
   IF "AlwaysTRUE" AND ("MODE SELECTION DB"."MODE BUFF" = 1) AND (("MFG PROCESS_DB"."AUTO BUFF" = 25) OR ("MFG PROCESS_DB"."AUTO BUFF" = 35)) AND ("CONTINUE DB"."SYRUP MFG PROCESS ERROR" <> 1) THEN
       "SET PARAMETER DB"."AUTO VFD SET PARAMETER"."MFG VESSEL STIRROR RUN" := "MFG PROCESS_DB"."SET PARAMETER"."PURIFIED STIRRER MOTOR RPM";
   END_IF;
   IF "AlwaysTRUE" AND ("MODE SELECTION DB"."MODE BUFF" = 1) AND ("MFG PROCESS_DB"."AUTO BUFF" >= 90) AND ("MFG PROCESS_DB"."AUTO BUFF" <= 95) AND ("CONTINUE DB"."SYRUP MFG PROCESS ERROR" <> 1) THEN
       "SET PARAMETER DB"."AUTO VFD SET PARAMETER"."MFG VESSEL STIRROR RUN" := "MFG PROCESS_DB"."SET PARAMETER"."MATERIAL SORBITOL STIRRER MOTOR RPM";
   END_IF;
   IF "AlwaysTRUE" AND ("MODE SELECTION DB"."MODE BUFF" = 1) AND ("MFG PROCESS_DB"."AUTO BUFF" >= 125) AND ("MFG PROCESS_DB"."AUTO BUFF" <= 130) AND ("CONTINUE DB"."SYRUP MFG PROCESS ERROR" <> 1) THEN
       "SET PARAMETER DB"."AUTO VFD SET PARAMETER"."MFG VESSEL STIRROR RUN" := "MFG PROCESS_DB"."SET PARAMETER"."MATERIAL GLUCOSE STIRRER MOTOR RPM";
   END_IF;
   IF "AlwaysTRUE" AND ("MODE SELECTION DB"."MODE BUFF" = 1) AND ("MFG PROCESS_DB"."AUTO BUFF" >= 155) AND ("MFG PROCESS_DB"."AUTO BUFF" <= 160) AND ("CONTINUE DB"."SYRUP MFG PROCESS ERROR" <> 1) THEN
       "SET PARAMETER DB"."AUTO VFD SET PARAMETER"."MFG VESSEL STIRROR RUN" := "MFG PROCESS_DB"."SET PARAMETER"."RECIRCULATION STIRRER RPM";
   END_IF;
   #_w1 := "AlwaysTRUE" AND ("MODE SELECTION DB"."MODE BUFF" = 1);
   IF #_w1 AND ("MFG TRANSFER CYCLE DB".TRANSFER."TRANSFER BUFF"."MFG TO STORAGE-1 WITH INLINE HOMO" = 10) THEN
       "SET PARAMETER DB"."AUTO VFD SET PARAMETER"."MFG VESSEL STIRROR RUN" := "MFG TRANSFER CYCLE DB"."SET PARAMETER".RPM."MFG TO STORAGE-1 WITH INLINE HOMO";
   END_IF;
   IF #_w1 AND ("MFG TRANSFER CYCLE DB".TRANSFER."TRANSFER BUFF"."MFG TO STORAGE-1 WITH INLINE FILTER PRES" = 10) THEN
       "SET PARAMETER DB"."AUTO VFD SET PARAMETER"."MFG VESSEL STIRROR RUN" := "MFG TRANSFER CYCLE DB"."SET PARAMETER".RPM."MFG TO STORAGE-1 WITH INLINE FILTER PRES";
   END_IF;
   IF #_w1 AND ("MFG TRANSFER CYCLE DB".TRANSFER."TRANSFER BUFF"."MFG TO STORAGE-2 WITH INLINE HOMO" = 10) THEN
       "SET PARAMETER DB"."AUTO VFD SET PARAMETER"."MFG VESSEL STIRROR RUN" := "MFG TRANSFER CYCLE DB"."SET PARAMETER".RPM."MFG TO STORAGE-2 WITH INLINE HOMO";
   END_IF;
   IF #_w1 AND ("MFG TRANSFER CYCLE DB".TRANSFER."TRANSFER BUFF"."MFG TO STORAGE-2 WITH INLINE FILTER PRES" = 10) THEN
       "SET PARAMETER DB"."AUTO VFD SET PARAMETER"."MFG VESSEL STIRROR RUN" := "MFG TRANSFER CYCLE DB"."SET PARAMETER".RPM."MFG TO STORAGE-2 WITH INLINE FILTER PRES";
   END_IF;
   IF #_w1 AND ("MFG TRANSFER CYCLE DB".TRANSFER."TRANSFER BUFF"."MFG TO STORAGE-3 WITH INLINE HOMO" = 10) THEN
       "SET PARAMETER DB"."AUTO VFD SET PARAMETER"."MFG VESSEL STIRROR RUN" := "MFG TRANSFER CYCLE DB"."SET PARAMETER".RPM."MFG TO STORAGE-3 WITH INLINE HOMO";
   END_IF;
   IF #_w1 AND ("MFG TRANSFER CYCLE DB".TRANSFER."TRANSFER BUFF"."MFG TO STORAGE-3 WITH INLINE FILTER PRES" = 10) THEN
       "SET PARAMETER DB"."AUTO VFD SET PARAMETER"."MFG VESSEL STIRROR RUN" := "MFG TRANSFER CYCLE DB"."SET PARAMETER".RPM."MFG TO STORAGE-3 WITH INLINE FILTER PRES";
   END_IF;
   IF "AlwaysTRUE" AND ("MFG PROCESS_DB"."MATERIAL SUCTION"."MATERIAL SUCTION BUFF" = 10) AND ("CONTINUE DB"."SYRUP MFG PROCESS ERROR" <> 1) THEN
       "SET PARAMETER DB"."AUTO VFD SET PARAMETER"."MFG VESSEL STIRROR RUN" := "MFG PROCESS_DB"."SET PARAMETER"."MATERIAL SUCTION STIRRER RPM";
   END_IF;
END_REGION

REGION Network 2: PREMIXING STIRRER MOTOR
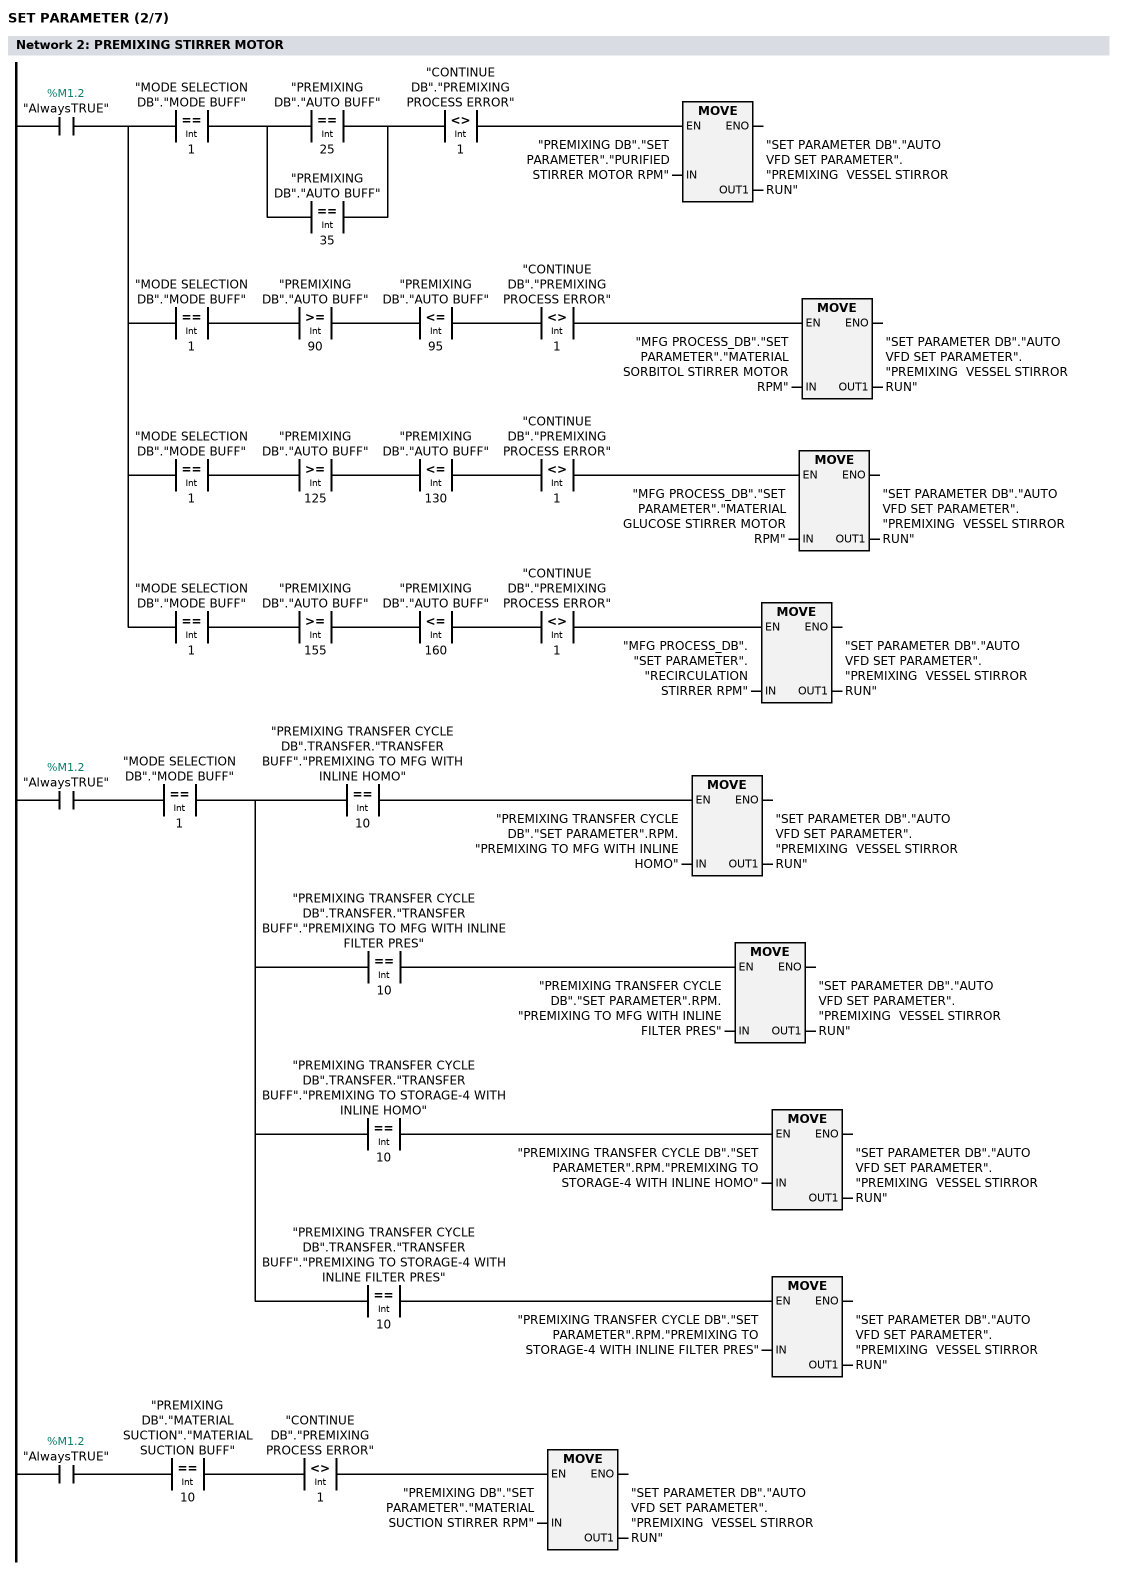
   RUNG wire#powerrail
      Contact( "AlwaysTRUE" )
      wire#w1
      { S7_Templates := "SrcType := Int" } EQ_Contact(in1 := "MODE SELECTION DB"."MODE BUFF", in2 := 1)
      wire#w2
      { S7_Templates := "SrcType := Int" } EQ_Contact(in1 := "PREMIXING DB"."AUTO BUFF", in2 := 25)
      wire#w3
      { S7_Templates := "SrcType := Int" } NE_Contact(in1 := "CONTINUE DB"."PREMIXING PROCESS ERROR", in2 := 1)
      Move(in := "PREMIXING DB"."SET PARAMETER"."PURIFIED STIRRER MOTOR RPM", out1 => "SET PARAMETER DB"."AUTO VFD SET PARAMETER"."PREMIXING  VESSEL STIRROR RUN")
   END_RUNG
   RUNG wire#w2
      { S7_Templates := "SrcType := Int" } EQ_Contact(in1 := "PREMIXING DB"."AUTO BUFF", in2 := 35)
   END_RUNG wire#w3
   RUNG wire#w1
      { S7_Templates := "SrcType := Int" } EQ_Contact(in1 := "MODE SELECTION DB"."MODE BUFF", in2 := 1)
      { S7_Templates := "SrcType := Int" } GE_Contact(in1 := "PREMIXING DB"."AUTO BUFF", in2 := 90)
      { S7_Templates := "SrcType := Int" } LE_Contact(in1 := "PREMIXING DB"."AUTO BUFF", in2 := 95)
      { S7_Templates := "SrcType := Int" } NE_Contact(in1 := "CONTINUE DB"."PREMIXING PROCESS ERROR", in2 := 1)
      Move(in := "MFG PROCESS_DB"."SET PARAMETER"."MATERIAL SORBITOL STIRRER MOTOR RPM", out1 => "SET PARAMETER DB"."AUTO VFD SET PARAMETER"."PREMIXING  VESSEL STIRROR RUN")
   END_RUNG
   RUNG wire#w1
      { S7_Templates := "SrcType := Int" } EQ_Contact(in1 := "MODE SELECTION DB"."MODE BUFF", in2 := 1)
      { S7_Templates := "SrcType := Int" } GE_Contact(in1 := "PREMIXING DB"."AUTO BUFF", in2 := 125)
      { S7_Templates := "SrcType := Int" } LE_Contact(in1 := "PREMIXING DB"."AUTO BUFF", in2 := 130)
      { S7_Templates := "SrcType := Int" } NE_Contact(in1 := "CONTINUE DB"."PREMIXING PROCESS ERROR", in2 := 1)
      Move(in := "MFG PROCESS_DB"."SET PARAMETER"."MATERIAL GLUCOSE STIRRER MOTOR RPM", out1 => "SET PARAMETER DB"."AUTO VFD SET PARAMETER"."PREMIXING  VESSEL STIRROR RUN")
   END_RUNG
   RUNG wire#w1
      { S7_Templates := "SrcType := Int" } EQ_Contact(in1 := "MODE SELECTION DB"."MODE BUFF", in2 := 1)
      { S7_Templates := "SrcType := Int" } GE_Contact(in1 := "PREMIXING DB"."AUTO BUFF", in2 := 155)
      { S7_Templates := "SrcType := Int" } LE_Contact(in1 := "PREMIXING DB"."AUTO BUFF", in2 := 160)
      { S7_Templates := "SrcType := Int" } NE_Contact(in1 := "CONTINUE DB"."PREMIXING PROCESS ERROR", in2 := 1)
      Move(in := "MFG PROCESS_DB"."SET PARAMETER"."RECIRCULATION STIRRER RPM", out1 => "SET PARAMETER DB"."AUTO VFD SET PARAMETER"."PREMIXING  VESSEL STIRROR RUN")
   END_RUNG
   RUNG wire#powerrail
      Contact( "AlwaysTRUE" )
      { S7_Templates := "SrcType := Int" } EQ_Contact(in1 := "MODE SELECTION DB"."MODE BUFF", in2 := 1)
      wire#w4
      { S7_Templates := "SrcType := Int" } EQ_Contact(in1 := "PREMIXING TRANSFER CYCLE DB".TRANSFER."TRANSFER BUFF"."PREMIXING TO MFG WITH INLINE HOMO", in2 := 10)
      Move(in := "PREMIXING TRANSFER CYCLE DB"."SET PARAMETER".RPM."PREMIXING TO MFG WITH INLINE HOMO", out1 => "SET PARAMETER DB"."AUTO VFD SET PARAMETER"."PREMIXING  VESSEL STIRROR RUN")
   END_RUNG
   RUNG wire#w4
      { S7_Templates := "SrcType := Int" } EQ_Contact(in1 := "PREMIXING TRANSFER CYCLE DB".TRANSFER."TRANSFER BUFF"."PREMIXING TO MFG WITH INLINE FILTER PRES", in2 := 10)
      Move(in := "PREMIXING TRANSFER CYCLE DB"."SET PARAMETER".RPM."PREMIXING TO MFG WITH INLINE FILTER PRES", out1 => "SET PARAMETER DB"."AUTO VFD SET PARAMETER"."PREMIXING  VESSEL STIRROR RUN")
   END_RUNG
   RUNG wire#w4
      { S7_Templates := "SrcType := Int" } EQ_Contact(in1 := "PREMIXING TRANSFER CYCLE DB".TRANSFER."TRANSFER BUFF"."PREMIXING TO STORAGE-4 WITH INLINE HOMO", in2 := 10)
      Move(in := "PREMIXING TRANSFER CYCLE DB"."SET PARAMETER".RPM."PREMIXING TO STORAGE-4 WITH INLINE HOMO", out1 => "SET PARAMETER DB"."AUTO VFD SET PARAMETER"."PREMIXING  VESSEL STIRROR RUN")
   END_RUNG
   RUNG wire#w4
      { S7_Templates := "SrcType := Int" } EQ_Contact(in1 := "PREMIXING TRANSFER CYCLE DB".TRANSFER."TRANSFER BUFF"."PREMIXING TO STORAGE-4 WITH INLINE FILTER PRES", in2 := 10)
      Move(in := "PREMIXING TRANSFER CYCLE DB"."SET PARAMETER".RPM."PREMIXING TO STORAGE-4 WITH INLINE FILTER PRES", out1 => "SET PARAMETER DB"."AUTO VFD SET PARAMETER"."PREMIXING  VESSEL STIRROR RUN")
   END_RUNG
   RUNG wire#powerrail
      Contact( "AlwaysTRUE" )
      { S7_Templates := "SrcType := Int" } EQ_Contact(in1 := "PREMIXING DB"."MATERIAL SUCTION"."MATERIAL SUCTION BUFF", in2 := 10)
      { S7_Templates := "SrcType := Int" } NE_Contact(in1 := "CONTINUE DB"."PREMIXING PROCESS ERROR", in2 := 1)
      Move(in := "PREMIXING DB"."SET PARAMETER"."MATERIAL SUCTION STIRRER RPM", out1 => "SET PARAMETER DB"."AUTO VFD SET PARAMETER"."PREMIXING  VESSEL STIRROR RUN")
   END_RUNG
   // the same network as SCL:
   IF "AlwaysTRUE" AND ("MODE SELECTION DB"."MODE BUFF" = 1) AND (("PREMIXING DB"."AUTO BUFF" = 25) OR ("PREMIXING DB"."AUTO BUFF" = 35)) AND ("CONTINUE DB"."PREMIXING PROCESS ERROR" <> 1) THEN
       "SET PARAMETER DB"."AUTO VFD SET PARAMETER"."PREMIXING  VESSEL STIRROR RUN" := "PREMIXING DB"."SET PARAMETER"."PURIFIED STIRRER MOTOR RPM";
   END_IF;
   IF "AlwaysTRUE" AND ("MODE SELECTION DB"."MODE BUFF" = 1) AND ("PREMIXING DB"."AUTO BUFF" >= 90) AND ("PREMIXING DB"."AUTO BUFF" <= 95) AND ("CONTINUE DB"."PREMIXING PROCESS ERROR" <> 1) THEN
       "SET PARAMETER DB"."AUTO VFD SET PARAMETER"."PREMIXING  VESSEL STIRROR RUN" := "MFG PROCESS_DB"."SET PARAMETER"."MATERIAL SORBITOL STIRRER MOTOR RPM";
   END_IF;
   IF "AlwaysTRUE" AND ("MODE SELECTION DB"."MODE BUFF" = 1) AND ("PREMIXING DB"."AUTO BUFF" >= 125) AND ("PREMIXING DB"."AUTO BUFF" <= 130) AND ("CONTINUE DB"."PREMIXING PROCESS ERROR" <> 1) THEN
       "SET PARAMETER DB"."AUTO VFD SET PARAMETER"."PREMIXING  VESSEL STIRROR RUN" := "MFG PROCESS_DB"."SET PARAMETER"."MATERIAL GLUCOSE STIRRER MOTOR RPM";
   END_IF;
   IF "AlwaysTRUE" AND ("MODE SELECTION DB"."MODE BUFF" = 1) AND ("PREMIXING DB"."AUTO BUFF" >= 155) AND ("PREMIXING DB"."AUTO BUFF" <= 160) AND ("CONTINUE DB"."PREMIXING PROCESS ERROR" <> 1) THEN
       "SET PARAMETER DB"."AUTO VFD SET PARAMETER"."PREMIXING  VESSEL STIRROR RUN" := "MFG PROCESS_DB"."SET PARAMETER"."RECIRCULATION STIRRER RPM";
   END_IF;
   #_w1 := "AlwaysTRUE" AND ("MODE SELECTION DB"."MODE BUFF" = 1);
   IF #_w1 AND ("PREMIXING TRANSFER CYCLE DB".TRANSFER."TRANSFER BUFF"."PREMIXING TO MFG WITH INLINE HOMO" = 10) THEN
       "SET PARAMETER DB"."AUTO VFD SET PARAMETER"."PREMIXING  VESSEL STIRROR RUN" := "PREMIXING TRANSFER CYCLE DB"."SET PARAMETER".RPM."PREMIXING TO MFG WITH INLINE HOMO";
   END_IF;
   IF #_w1 AND ("PREMIXING TRANSFER CYCLE DB".TRANSFER."TRANSFER BUFF"."PREMIXING TO MFG WITH INLINE FILTER PRES" = 10) THEN
       "SET PARAMETER DB"."AUTO VFD SET PARAMETER"."PREMIXING  VESSEL STIRROR RUN" := "PREMIXING TRANSFER CYCLE DB"."SET PARAMETER".RPM."PREMIXING TO MFG WITH INLINE FILTER PRES";
   END_IF;
   IF #_w1 AND ("PREMIXING TRANSFER CYCLE DB".TRANSFER."TRANSFER BUFF"."PREMIXING TO STORAGE-4 WITH INLINE HOMO" = 10) THEN
       "SET PARAMETER DB"."AUTO VFD SET PARAMETER"."PREMIXING  VESSEL STIRROR RUN" := "PREMIXING TRANSFER CYCLE DB"."SET PARAMETER".RPM."PREMIXING TO STORAGE-4 WITH INLINE HOMO";
   END_IF;
   IF #_w1 AND ("PREMIXING TRANSFER CYCLE DB".TRANSFER."TRANSFER BUFF"."PREMIXING TO STORAGE-4 WITH INLINE FILTER PRES" = 10) THEN
       "SET PARAMETER DB"."AUTO VFD SET PARAMETER"."PREMIXING  VESSEL STIRROR RUN" := "PREMIXING TRANSFER CYCLE DB"."SET PARAMETER".RPM."PREMIXING TO STORAGE-4 WITH INLINE FILTER PRES";
   END_IF;
   IF "AlwaysTRUE" AND ("PREMIXING DB"."MATERIAL SUCTION"."MATERIAL SUCTION BUFF" = 10) AND ("CONTINUE DB"."PREMIXING PROCESS ERROR" <> 1) THEN
       "SET PARAMETER DB"."AUTO VFD SET PARAMETER"."PREMIXING  VESSEL STIRROR RUN" := "PREMIXING DB"."SET PARAMETER"."MATERIAL SUCTION STIRRER RPM";
   END_IF;
END_REGION

REGION Network 3: SUGAR STIRRER MOTOR
END_REGION

REGION Network 5: MFG_TEMP
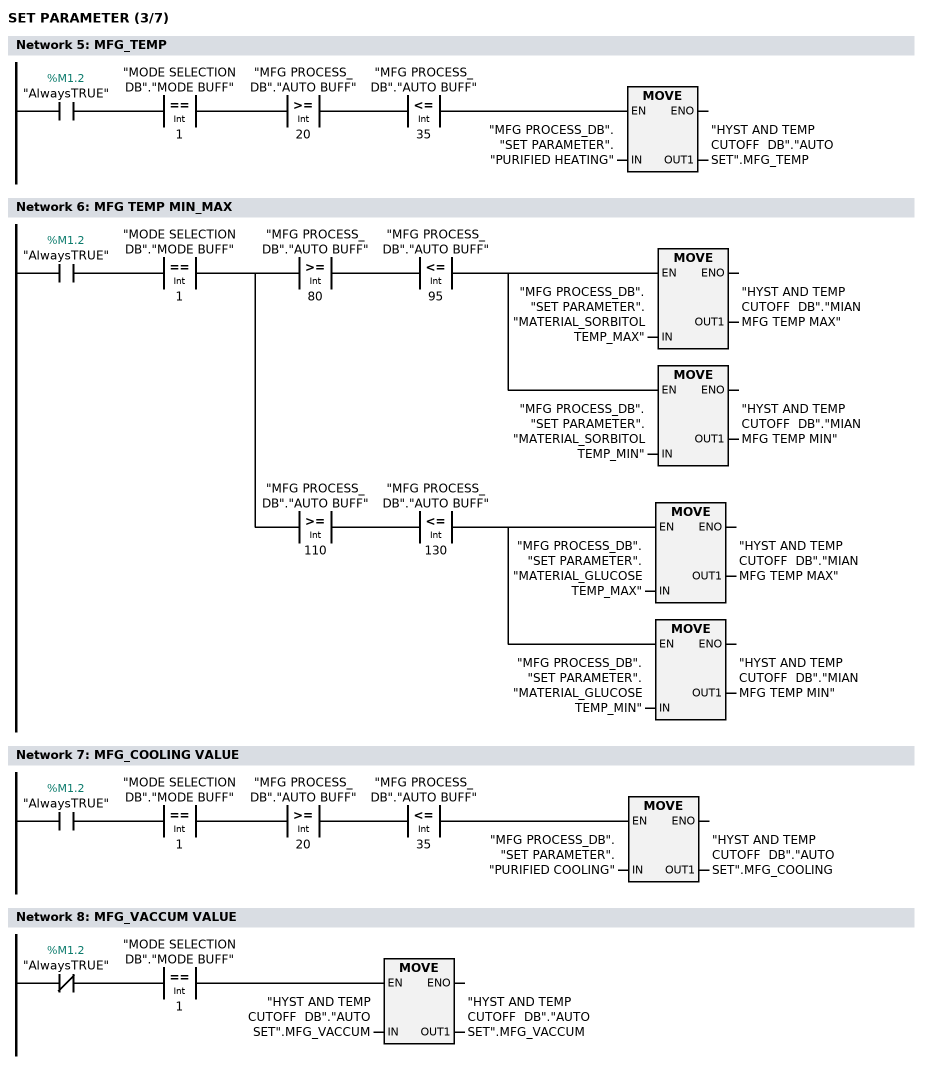
   RUNG wire#powerrail
      Contact( "AlwaysTRUE" )
      { S7_Templates := "SrcType := Int" } EQ_Contact(in1 := "MODE SELECTION DB"."MODE BUFF", in2 := 1)
      { S7_Templates := "SrcType := Int" } GE_Contact(in1 := "MFG PROCESS_DB"."AUTO BUFF", in2 := 20)
      { S7_Templates := "SrcType := Int" } LE_Contact(in1 := "MFG PROCESS_DB"."AUTO BUFF", in2 := 35)
      Move(in := "MFG PROCESS_DB"."SET PARAMETER"."PURIFIED HEATING", out1 => "HYST AND TEMP CUTOFF  DB"."AUTO SET".MFG_TEMP)
   END_RUNG
   // the same network as SCL:
   IF "AlwaysTRUE" AND ("MODE SELECTION DB"."MODE BUFF" = 1) AND ("MFG PROCESS_DB"."AUTO BUFF" >= 20) AND ("MFG PROCESS_DB"."AUTO BUFF" <= 35) THEN
       "HYST AND TEMP CUTOFF  DB"."AUTO SET".MFG_TEMP := "MFG PROCESS_DB"."SET PARAMETER"."PURIFIED HEATING";
   END_IF;
END_REGION

REGION Network 6: MFG TEMP MIN_MAX
   RUNG wire#powerrail
      Contact( "AlwaysTRUE" )
      { S7_Templates := "SrcType := Int" } EQ_Contact(in1 := "MODE SELECTION DB"."MODE BUFF", in2 := 1)
      wire#w1
      { S7_Templates := "SrcType := Int" } GE_Contact(in1 := "MFG PROCESS_DB"."AUTO BUFF", in2 := 80)
      { S7_Templates := "SrcType := Int" } LE_Contact(in1 := "MFG PROCESS_DB"."AUTO BUFF", in2 := 95)
      wire#w2
      Move(in := "MFG PROCESS_DB"."SET PARAMETER"."MATERIAL_SORBITOL TEMP_MAX", out1 => "HYST AND TEMP CUTOFF  DB"."MIAN MFG TEMP MAX")
   END_RUNG
   RUNG wire#w2
      Move(in := "MFG PROCESS_DB"."SET PARAMETER"."MATERIAL_SORBITOL TEMP_MIN", out1 => "HYST AND TEMP CUTOFF  DB"."MIAN MFG TEMP MIN")
   END_RUNG
   RUNG wire#w1
      { S7_Templates := "SrcType := Int" } GE_Contact(in1 := "MFG PROCESS_DB"."AUTO BUFF", in2 := 110)
      { S7_Templates := "SrcType := Int" } LE_Contact(in1 := "MFG PROCESS_DB"."AUTO BUFF", in2 := 130)
      wire#w3
      Move(in := "MFG PROCESS_DB"."SET PARAMETER"."MATERIAL_GLUCOSE TEMP_MAX", out1 => "HYST AND TEMP CUTOFF  DB"."MIAN MFG TEMP MAX")
   END_RUNG
   RUNG wire#w3
      Move(in := "MFG PROCESS_DB"."SET PARAMETER"."MATERIAL_GLUCOSE TEMP_MIN", out1 => "HYST AND TEMP CUTOFF  DB"."MIAN MFG TEMP MIN")
   END_RUNG
   // the same network as SCL:
   #_w1 := "AlwaysTRUE" AND ("MODE SELECTION DB"."MODE BUFF" = 1);
   IF #_w1 AND ("MFG PROCESS_DB"."AUTO BUFF" >= 80) AND ("MFG PROCESS_DB"."AUTO BUFF" <= 95) THEN
       "HYST AND TEMP CUTOFF  DB"."MIAN MFG TEMP MAX" := "MFG PROCESS_DB"."SET PARAMETER"."MATERIAL_SORBITOL TEMP_MAX";
       "HYST AND TEMP CUTOFF  DB"."MIAN MFG TEMP MIN" := "MFG PROCESS_DB"."SET PARAMETER"."MATERIAL_SORBITOL TEMP_MIN";
   END_IF;
   IF #_w1 AND ("MFG PROCESS_DB"."AUTO BUFF" >= 110) AND ("MFG PROCESS_DB"."AUTO BUFF" <= 130) THEN
       "HYST AND TEMP CUTOFF  DB"."MIAN MFG TEMP MAX" := "MFG PROCESS_DB"."SET PARAMETER"."MATERIAL_GLUCOSE TEMP_MAX";
       "HYST AND TEMP CUTOFF  DB"."MIAN MFG TEMP MIN" := "MFG PROCESS_DB"."SET PARAMETER"."MATERIAL_GLUCOSE TEMP_MIN";
   END_IF;
END_REGION

REGION Network 7: MFG_COOLING VALUE
   RUNG wire#powerrail
      Contact( "AlwaysTRUE" )
      { S7_Templates := "SrcType := Int" } EQ_Contact(in1 := "MODE SELECTION DB"."MODE BUFF", in2 := 1)
      { S7_Templates := "SrcType := Int" } GE_Contact(in1 := "MFG PROCESS_DB"."AUTO BUFF", in2 := 20)
      { S7_Templates := "SrcType := Int" } LE_Contact(in1 := "MFG PROCESS_DB"."AUTO BUFF", in2 := 35)
      Move(in := "MFG PROCESS_DB"."SET PARAMETER"."PURIFIED COOLING", out1 => "HYST AND TEMP CUTOFF  DB"."AUTO SET".MFG_COOLING)
   END_RUNG
   // the same network as SCL:
   IF "AlwaysTRUE" AND ("MODE SELECTION DB"."MODE BUFF" = 1) AND ("MFG PROCESS_DB"."AUTO BUFF" >= 20) AND ("MFG PROCESS_DB"."AUTO BUFF" <= 35) THEN
       "HYST AND TEMP CUTOFF  DB"."AUTO SET".MFG_COOLING := "MFG PROCESS_DB"."SET PARAMETER"."PURIFIED COOLING";
   END_IF;
END_REGION

REGION Network 8: MFG_VACCUM VALUE
   RUNG wire#powerrail
      I_Contact( "AlwaysTRUE" )
      { S7_Templates := "SrcType := Int" } EQ_Contact(in1 := "MODE SELECTION DB"."MODE BUFF", in2 := 1)
      Move(in := "HYST AND TEMP CUTOFF  DB"."AUTO SET".MFG_VACCUM, out1 => "HYST AND TEMP CUTOFF  DB"."AUTO SET".MFG_VACCUM)
   END_RUNG
   // the same network as SCL:
   IF NOT "AlwaysTRUE" AND ("MODE SELECTION DB"."MODE BUFF" = 1) THEN
       "HYST AND TEMP CUTOFF  DB"."AUTO SET".MFG_VACCUM := "HYST AND TEMP CUTOFF  DB"."AUTO SET".MFG_VACCUM;
   END_IF;
END_REGION

